REGION Network 12: HMI BA3 SET GOOD PART
   RUNG wire#powerrail
      Contact( "DB2001_MODES_GENERAL".BA.BA3_SELECTED )
      I_Contact( "DB1201_PART_CYCLE_UNIT_01".RUNNING )
      Contact( "DB1018_SAFETY_TAGS".ENABLE_DEVICE_FROM_UNIT_01_MAIN_SAFETY_DOOR_AREA )
      Contact( "DB7224_HMI_AXES".BA3.SOFTKEYS.SET_GOOD_PART )
      wire#w1
      Contact( "DB4000_FIX_TABLE_POSITIONS".UNIT_01.FIXTURE_1.IN_CLADDING_STATION_3 )
      wire#w2
      S_Coil( "DB8000_PART_STATUS".UNIT_01.FIXTURE_1.PART_A.STATUS.OK )
   END_RUNG
   RUNG wire#w2
      R_Coil( "DB8000_PART_STATUS".UNIT_01.FIXTURE_1.PART_A.STATUS.PART_REJECTED )
   END_RUNG
   RUNG wire#w1
      Contact( "DB4000_FIX_TABLE_POSITIONS".UNIT_01.FIXTURE_2.IN_CLADDING_STATION_3 )
      wire#w3
      S_Coil( "DB8000_PART_STATUS".UNIT_01.FIXTURE_2.PART_A.STATUS.OK )
   END_RUNG
   RUNG wire#w3
      R_Coil( "DB8000_PART_STATUS".UNIT_01.FIXTURE_2.PART_A.STATUS.PART_REJECTED )
   END_RUNG
   RUNG wire#w1
      Contact( "DB4000_FIX_TABLE_POSITIONS".UNIT_01.FIXTURE_3.IN_CLADDING_STATION_3 )
      wire#w4
      S_Coil( "DB8000_PART_STATUS".UNIT_01.FIXTURE_3.PART_A.STATUS.OK )
   END_RUNG
   RUNG wire#w4
      R_Coil( "DB8000_PART_STATUS".UNIT_01.FIXTURE_3.PART_A.STATUS.PART_REJECTED )
   END_RUNG
   RUNG wire#w1
      Contact( "DB4000_FIX_TABLE_POSITIONS".UNIT_01.FIXTURE_4.IN_CLADDING_STATION_3 )
      wire#w5
      S_Coil( "DB8000_PART_STATUS".UNIT_01.FIXTURE_4.PART_A.STATUS.OK )
   END_RUNG
   RUNG wire#w5
      R_Coil( "DB8000_PART_STATUS".UNIT_01.FIXTURE_4.PART_A.STATUS.PART_REJECTED )
   END_RUNG
   // the same network as SCL:
   #_w1 := "DB2001_MODES_GENERAL".BA.BA3_SELECTED AND NOT "DB1201_PART_CYCLE_UNIT_01".RUNNING AND "DB1018_SAFETY_TAGS".ENABLE_DEVICE_FROM_UNIT_01_MAIN_SAFETY_DOOR_AREA AND "DB7224_HMI_AXES".BA3.SOFTKEYS.SET_GOOD_PART;
   IF #_w1 AND "DB4000_FIX_TABLE_POSITIONS".UNIT_01.FIXTURE_1.IN_CLADDING_STATION_3 THEN
       "DB8000_PART_STATUS".UNIT_01.FIXTURE_1.PART_A.STATUS.OK := TRUE;
       "DB8000_PART_STATUS".UNIT_01.FIXTURE_1.PART_A.STATUS.PART_REJECTED := FALSE;
   END_IF;
   IF #_w1 AND "DB4000_FIX_TABLE_POSITIONS".UNIT_01.FIXTURE_2.IN_CLADDING_STATION_3 THEN
       "DB8000_PART_STATUS".UNIT_01.FIXTURE_2.PART_A.STATUS.OK := TRUE;
       "DB8000_PART_STATUS".UNIT_01.FIXTURE_2.PART_A.STATUS.PART_REJECTED := FALSE;
   END_IF;
   IF #_w1 AND "DB4000_FIX_TABLE_POSITIONS".UNIT_01.FIXTURE_3.IN_CLADDING_STATION_3 THEN
       "DB8000_PART_STATUS".UNIT_01.FIXTURE_3.PART_A.STATUS.OK := TRUE;
       "DB8000_PART_STATUS".UNIT_01.FIXTURE_3.PART_A.STATUS.PART_REJECTED := FALSE;
   END_IF;
   IF #_w1 AND "DB4000_FIX_TABLE_POSITIONS".UNIT_01.FIXTURE_4.IN_CLADDING_STATION_3 THEN
       "DB8000_PART_STATUS".UNIT_01.FIXTURE_4.PART_A.STATUS.OK := TRUE;
       "DB8000_PART_STATUS".UNIT_01.FIXTURE_4.PART_A.STATUS.PART_REJECTED := FALSE;
   END_IF;
END_REGION

REGION Network 13: UNIT 01 STATION 1 PART A PRESENT
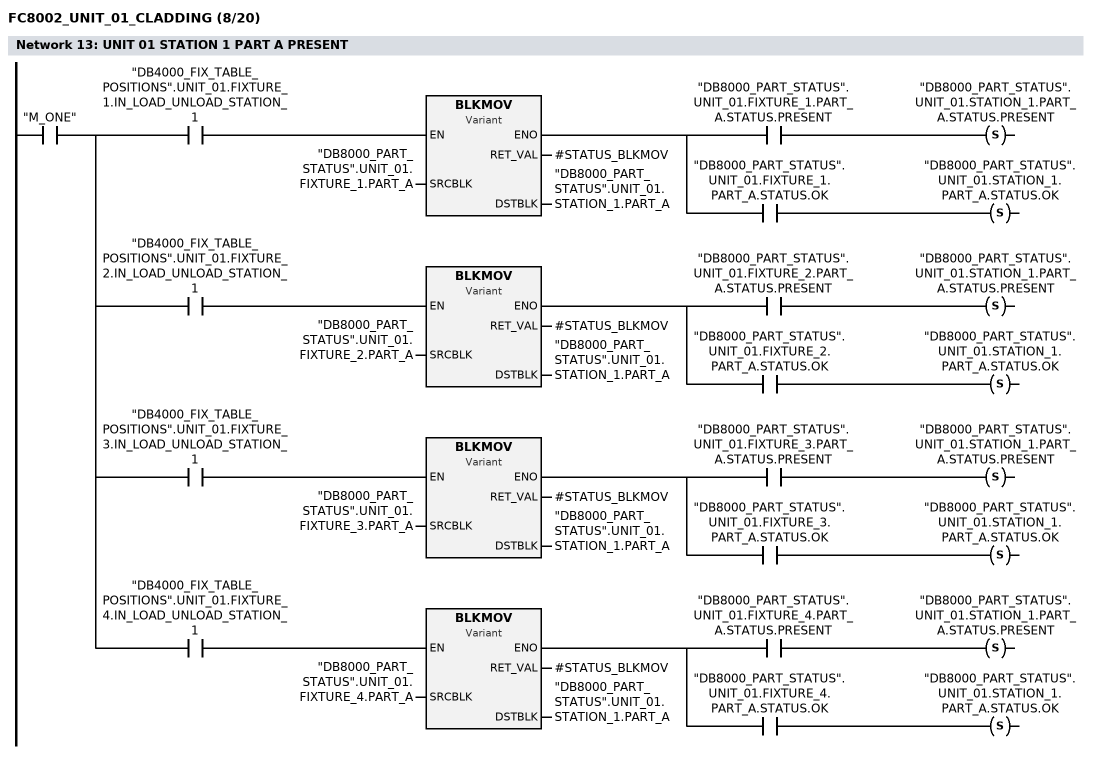
   RUNG wire#powerrail
      Contact( "M_ONE" )
      wire#w1
      Contact( "DB4000_FIX_TABLE_POSITIONS".UNIT_01.FIXTURE_1.IN_LOAD_UNLOAD_STATION_1 )
      { S7_Templates := "blk_type := Variant" } BLKMOV(SRCBLK := "DB8000_PART_STATUS".UNIT_01.FIXTURE_1.PART_A, RET_VAL => #STATUS_BLKMOV, DSTBLK => "DB8000_PART_STATUS".UNIT_01.STATION_1.PART_A)
      wire#w2
      Contact( "DB8000_PART_STATUS".UNIT_01.FIXTURE_1.PART_A.STATUS.PRESENT )
      S_Coil( "DB8000_PART_STATUS".UNIT_01.STATION_1.PART_A.STATUS.PRESENT )
   END_RUNG
   RUNG wire#w2
      Contact( "DB8000_PART_STATUS".UNIT_01.FIXTURE_1.PART_A.STATUS.OK )
      S_Coil( "DB8000_PART_STATUS".UNIT_01.STATION_1.PART_A.STATUS.OK )
   END_RUNG
   RUNG wire#w1
      Contact( "DB4000_FIX_TABLE_POSITIONS".UNIT_01.FIXTURE_2.IN_LOAD_UNLOAD_STATION_1 )
      { S7_Templates := "blk_type := Variant" } BLKMOV(SRCBLK := "DB8000_PART_STATUS".UNIT_01.FIXTURE_2.PART_A, RET_VAL => #STATUS_BLKMOV, DSTBLK => "DB8000_PART_STATUS".UNIT_01.STATION_1.PART_A)
      wire#w3
      Contact( "DB8000_PART_STATUS".UNIT_01.FIXTURE_2.PART_A.STATUS.PRESENT )
      S_Coil( "DB8000_PART_STATUS".UNIT_01.STATION_1.PART_A.STATUS.PRESENT )
   END_RUNG
   RUNG wire#w3
      Contact( "DB8000_PART_STATUS".UNIT_01.FIXTURE_2.PART_A.STATUS.OK )
      S_Coil( "DB8000_PART_STATUS".UNIT_01.STATION_1.PART_A.STATUS.OK )
   END_RUNG
   RUNG wire#w1
      Contact( "DB4000_FIX_TABLE_POSITIONS".UNIT_01.FIXTURE_3.IN_LOAD_UNLOAD_STATION_1 )
      { S7_Templates := "blk_type := Variant" } BLKMOV(SRCBLK := "DB8000_PART_STATUS".UNIT_01.FIXTURE_3.PART_A, RET_VAL => #STATUS_BLKMOV, DSTBLK => "DB8000_PART_STATUS".UNIT_01.STATION_1.PART_A)
      wire#w4
      Contact( "DB8000_PART_STATUS".UNIT_01.FIXTURE_3.PART_A.STATUS.PRESENT )
      S_Coil( "DB8000_PART_STATUS".UNIT_01.STATION_1.PART_A.STATUS.PRESENT )
   END_RUNG
   RUNG wire#w4
      Contact( "DB8000_PART_STATUS".UNIT_01.FIXTURE_3.PART_A.STATUS.OK )
      S_Coil( "DB8000_PART_STATUS".UNIT_01.STATION_1.PART_A.STATUS.OK )
   END_RUNG
   RUNG wire#w1
      Contact( "DB4000_FIX_TABLE_POSITIONS".UNIT_01.FIXTURE_4.IN_LOAD_UNLOAD_STATION_1 )
      { S7_Templates := "blk_type := Variant" } BLKMOV(SRCBLK := "DB8000_PART_STATUS".UNIT_01.FIXTURE_4.PART_A, RET_VAL => #STATUS_BLKMOV, DSTBLK => "DB8000_PART_STATUS".UNIT_01.STATION_1.PART_A)
      wire#w5
      Contact( "DB8000_PART_STATUS".UNIT_01.FIXTURE_4.PART_A.STATUS.PRESENT )
      S_Coil( "DB8000_PART_STATUS".UNIT_01.STATION_1.PART_A.STATUS.PRESENT )
   END_RUNG
   RUNG wire#w5
      Contact( "DB8000_PART_STATUS".UNIT_01.FIXTURE_4.PART_A.STATUS.OK )
      S_Coil( "DB8000_PART_STATUS".UNIT_01.STATION_1.PART_A.STATUS.OK )
   END_RUNG
   // the same network as SCL:
   #_w1 := "M_ONE" AND "DB4000_FIX_TABLE_POSITIONS".UNIT_01.FIXTURE_1.IN_LOAD_UNLOAD_STATION_1;
   #_w3 := "M_ONE";
   #STATUS_BLKMOV := BLKMOV(EN := #_w1,
                           SRCBLK := "DB8000_PART_STATUS".UNIT_01.FIXTURE_1.PART_A,
                           DSTBLK => "DB8000_PART_STATUS".UNIT_01.STATION_1.PART_A,
                           ENO => #_w2);
   IF #_w2 AND "DB8000_PART_STATUS".UNIT_01.FIXTURE_1.PART_A.STATUS.PRESENT THEN
       "DB8000_PART_STATUS".UNIT_01.STATION_1.PART_A.STATUS.PRESENT := TRUE;
   END_IF;
   IF #_w2 AND "DB8000_PART_STATUS".UNIT_01.FIXTURE_1.PART_A.STATUS.OK THEN
       "DB8000_PART_STATUS".UNIT_01.STATION_1.PART_A.STATUS.OK := TRUE;
   END_IF;
   #_w4 := #_w3 AND "DB4000_FIX_TABLE_POSITIONS".UNIT_01.FIXTURE_2.IN_LOAD_UNLOAD_STATION_1;
   #STATUS_BLKMOV := BLKMOV(EN := #_w4,
                           SRCBLK := "DB8000_PART_STATUS".UNIT_01.FIXTURE_2.PART_A,
                           DSTBLK => "DB8000_PART_STATUS".UNIT_01.STATION_1.PART_A,
                           ENO => #_w5);
   IF #_w5 AND "DB8000_PART_STATUS".UNIT_01.FIXTURE_2.PART_A.STATUS.PRESENT THEN
       "DB8000_PART_STATUS".UNIT_01.STATION_1.PART_A.STATUS.PRESENT := TRUE;
   END_IF;
   IF #_w5 AND "DB8000_PART_STATUS".UNIT_01.FIXTURE_2.PART_A.STATUS.OK THEN
       "DB8000_PART_STATUS".UNIT_01.STATION_1.PART_A.STATUS.OK := TRUE;
   END_IF;
   #_w6 := #_w3 AND "DB4000_FIX_TABLE_POSITIONS".UNIT_01.FIXTURE_3.IN_LOAD_UNLOAD_STATION_1;
   #STATUS_BLKMOV := BLKMOV(EN := #_w6,
                           SRCBLK := "DB8000_PART_STATUS".UNIT_01.FIXTURE_3.PART_A,
                           DSTBLK => "DB8000_PART_STATUS".UNIT_01.STATION_1.PART_A,
                           ENO => #_w7);
   IF #_w7 AND "DB8000_PART_STATUS".UNIT_01.FIXTURE_3.PART_A.STATUS.PRESENT THEN
       "DB8000_PART_STATUS".UNIT_01.STATION_1.PART_A.STATUS.PRESENT := TRUE;
   END_IF;
   IF #_w7 AND "DB8000_PART_STATUS".UNIT_01.FIXTURE_3.PART_A.STATUS.OK THEN
       "DB8000_PART_STATUS".UNIT_01.STATION_1.PART_A.STATUS.OK := TRUE;
   END_IF;
   #_w8 := #_w3 AND "DB4000_FIX_TABLE_POSITIONS".UNIT_01.FIXTURE_4.IN_LOAD_UNLOAD_STATION_1;
   #STATUS_BLKMOV := BLKMOV(EN := #_w8,
                           SRCBLK := "DB8000_PART_STATUS".UNIT_01.FIXTURE_4.PART_A,
                           DSTBLK => "DB8000_PART_STATUS".UNIT_01.STATION_1.PART_A,
                           ENO => #_w9);
   IF #_w9 AND "DB8000_PART_STATUS".UNIT_01.FIXTURE_4.PART_A.STATUS.PRESENT THEN
       "DB8000_PART_STATUS".UNIT_01.STATION_1.PART_A.STATUS.PRESENT := TRUE;
   END_IF;
   IF #_w9 AND "DB8000_PART_STATUS".UNIT_01.FIXTURE_4.PART_A.STATUS.OK THEN
       "DB8000_PART_STATUS".UNIT_01.STATION_1.PART_A.STATUS.OK := TRUE;
   END_IF;
END_REGION

REGION Network 14: UNIT 01 STATION 2 PART A PRESENT
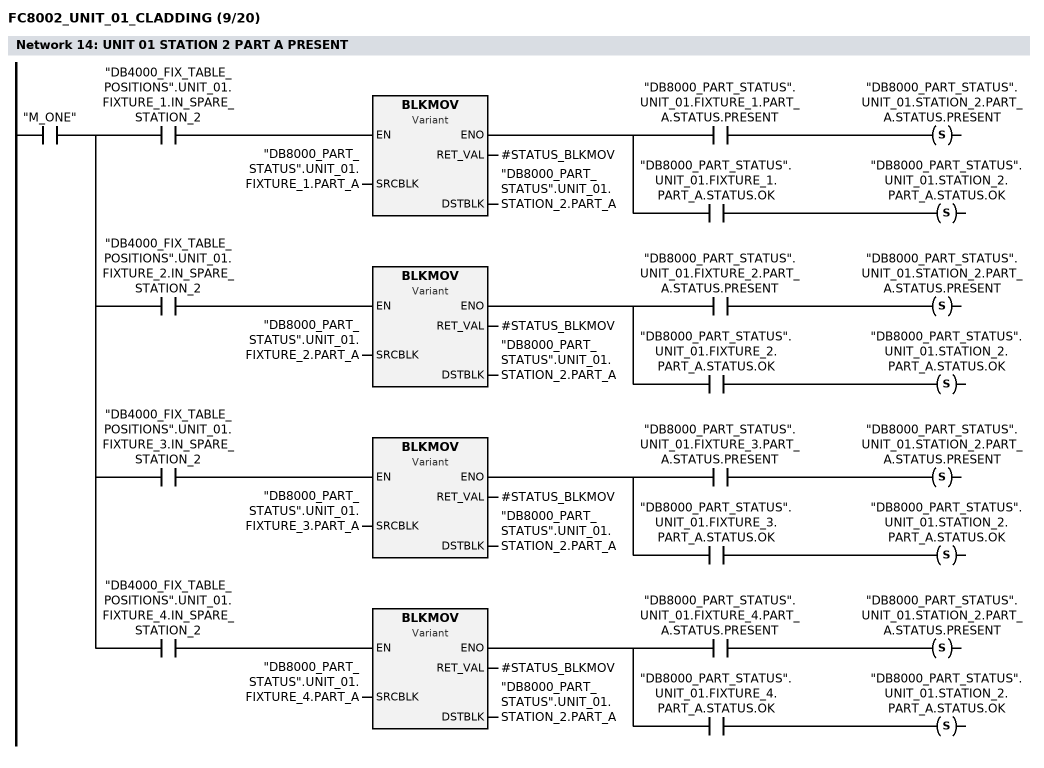
   RUNG wire#powerrail
      Contact( "M_ONE" )
      wire#w1
      Contact( "DB4000_FIX_TABLE_POSITIONS".UNIT_01.FIXTURE_1.IN_SPARE_STATION_2 )
      { S7_Templates := "blk_type := Variant" } BLKMOV(SRCBLK := "DB8000_PART_STATUS".UNIT_01.FIXTURE_1.PART_A, RET_VAL => #STATUS_BLKMOV, DSTBLK => "DB8000_PART_STATUS".UNIT_01.STATION_2.PART_A)
      wire#w2
      Contact( "DB8000_PART_STATUS".UNIT_01.FIXTURE_1.PART_A.STATUS.PRESENT )
      S_Coil( "DB8000_PART_STATUS".UNIT_01.STATION_2.PART_A.STATUS.PRESENT )
   END_RUNG
   RUNG wire#w2
      Contact( "DB8000_PART_STATUS".UNIT_01.FIXTURE_1.PART_A.STATUS.OK )
      S_Coil( "DB8000_PART_STATUS".UNIT_01.STATION_2.PART_A.STATUS.OK )
   END_RUNG
   RUNG wire#w1
      Contact( "DB4000_FIX_TABLE_POSITIONS".UNIT_01.FIXTURE_2.IN_SPARE_STATION_2 )
      { S7_Templates := "blk_type := Variant" } BLKMOV(SRCBLK := "DB8000_PART_STATUS".UNIT_01.FIXTURE_2.PART_A, RET_VAL => #STATUS_BLKMOV, DSTBLK => "DB8000_PART_STATUS".UNIT_01.STATION_2.PART_A)
      wire#w3
      Contact( "DB8000_PART_STATUS".UNIT_01.FIXTURE_2.PART_A.STATUS.PRESENT )
      S_Coil( "DB8000_PART_STATUS".UNIT_01.STATION_2.PART_A.STATUS.PRESENT )
   END_RUNG
   RUNG wire#w3
      Contact( "DB8000_PART_STATUS".UNIT_01.FIXTURE_2.PART_A.STATUS.OK )
      S_Coil( "DB8000_PART_STATUS".UNIT_01.STATION_2.PART_A.STATUS.OK )
   END_RUNG
   RUNG wire#w1
      Contact( "DB4000_FIX_TABLE_POSITIONS".UNIT_01.FIXTURE_3.IN_SPARE_STATION_2 )
      { S7_Templates := "blk_type := Variant" } BLKMOV(SRCBLK := "DB8000_PART_STATUS".UNIT_01.FIXTURE_3.PART_A, RET_VAL => #STATUS_BLKMOV, DSTBLK => "DB8000_PART_STATUS".UNIT_01.STATION_2.PART_A)
      wire#w4
      Contact( "DB8000_PART_STATUS".UNIT_01.FIXTURE_3.PART_A.STATUS.PRESENT )
      S_Coil( "DB8000_PART_STATUS".UNIT_01.STATION_2.PART_A.STATUS.PRESENT )
   END_RUNG
   RUNG wire#w4
      Contact( "DB8000_PART_STATUS".UNIT_01.FIXTURE_3.PART_A.STATUS.OK )
      S_Coil( "DB8000_PART_STATUS".UNIT_01.STATION_2.PART_A.STATUS.OK )
   END_RUNG
   RUNG wire#w1
      Contact( "DB4000_FIX_TABLE_POSITIONS".UNIT_01.FIXTURE_4.IN_SPARE_STATION_2 )
      { S7_Templates := "blk_type := Variant" } BLKMOV(SRCBLK := "DB8000_PART_STATUS".UNIT_01.FIXTURE_4.PART_A, RET_VAL => #STATUS_BLKMOV, DSTBLK => "DB8000_PART_STATUS".UNIT_01.STATION_2.PART_A)
      wire#w5
      Contact( "DB8000_PART_STATUS".UNIT_01.FIXTURE_4.PART_A.STATUS.PRESENT )
      S_Coil( "DB8000_PART_STATUS".UNIT_01.STATION_2.PART_A.STATUS.PRESENT )
   END_RUNG
   RUNG wire#w5
      Contact( "DB8000_PART_STATUS".UNIT_01.FIXTURE_4.PART_A.STATUS.OK )
      S_Coil( "DB8000_PART_STATUS".UNIT_01.STATION_2.PART_A.STATUS.OK )
   END_RUNG
   // the same network as SCL:
   #_w1 := "M_ONE" AND "DB4000_FIX_TABLE_POSITIONS".UNIT_01.FIXTURE_1.IN_SPARE_STATION_2;
   #_w3 := "M_ONE";
   #STATUS_BLKMOV := BLKMOV(EN := #_w1,
                           SRCBLK := "DB8000_PART_STATUS".UNIT_01.FIXTURE_1.PART_A,
                           DSTBLK => "DB8000_PART_STATUS".UNIT_01.STATION_2.PART_A,
                           ENO => #_w2);
   IF #_w2 AND "DB8000_PART_STATUS".UNIT_01.FIXTURE_1.PART_A.STATUS.PRESENT THEN
       "DB8000_PART_STATUS".UNIT_01.STATION_2.PART_A.STATUS.PRESENT := TRUE;
   END_IF;
   IF #_w2 AND "DB8000_PART_STATUS".UNIT_01.FIXTURE_1.PART_A.STATUS.OK THEN
       "DB8000_PART_STATUS".UNIT_01.STATION_2.PART_A.STATUS.OK := TRUE;
   END_IF;
   #_w4 := #_w3 AND "DB4000_FIX_TABLE_POSITIONS".UNIT_01.FIXTURE_2.IN_SPARE_STATION_2;
   #STATUS_BLKMOV := BLKMOV(EN := #_w4,
                           SRCBLK := "DB8000_PART_STATUS".UNIT_01.FIXTURE_2.PART_A,
                           DSTBLK => "DB8000_PART_STATUS".UNIT_01.STATION_2.PART_A,
                           ENO => #_w5);
   IF #_w5 AND "DB8000_PART_STATUS".UNIT_01.FIXTURE_2.PART_A.STATUS.PRESENT THEN
       "DB8000_PART_STATUS".UNIT_01.STATION_2.PART_A.STATUS.PRESENT := TRUE;
   END_IF;
   IF #_w5 AND "DB8000_PART_STATUS".UNIT_01.FIXTURE_2.PART_A.STATUS.OK THEN
       "DB8000_PART_STATUS".UNIT_01.STATION_2.PART_A.STATUS.OK := TRUE;
   END_IF;
   #_w6 := #_w3 AND "DB4000_FIX_TABLE_POSITIONS".UNIT_01.FIXTURE_3.IN_SPARE_STATION_2;
   #STATUS_BLKMOV := BLKMOV(EN := #_w6,
                           SRCBLK := "DB8000_PART_STATUS".UNIT_01.FIXTURE_3.PART_A,
                           DSTBLK => "DB8000_PART_STATUS".UNIT_01.STATION_2.PART_A,
                           ENO => #_w7);
   IF #_w7 AND "DB8000_PART_STATUS".UNIT_01.FIXTURE_3.PART_A.STATUS.PRESENT THEN
       "DB8000_PART_STATUS".UNIT_01.STATION_2.PART_A.STATUS.PRESENT := TRUE;
   END_IF;
   IF #_w7 AND "DB8000_PART_STATUS".UNIT_01.FIXTURE_3.PART_A.STATUS.OK THEN
       "DB8000_PART_STATUS".UNIT_01.STATION_2.PART_A.STATUS.OK := TRUE;
   END_IF;
   #_w8 := #_w3 AND "DB4000_FIX_TABLE_POSITIONS".UNIT_01.FIXTURE_4.IN_SPARE_STATION_2;
   #STATUS_BLKMOV := BLKMOV(EN := #_w8,
                           SRCBLK := "DB8000_PART_STATUS".UNIT_01.FIXTURE_4.PART_A,
                           DSTBLK => "DB8000_PART_STATUS".UNIT_01.STATION_2.PART_A,
                           ENO => #_w9);
   IF #_w9 AND "DB8000_PART_STATUS".UNIT_01.FIXTURE_4.PART_A.STATUS.PRESENT THEN
       "DB8000_PART_STATUS".UNIT_01.STATION_2.PART_A.STATUS.PRESENT := TRUE;
   END_IF;
   IF #_w9 AND "DB8000_PART_STATUS".UNIT_01.FIXTURE_4.PART_A.STATUS.OK THEN
       "DB8000_PART_STATUS".UNIT_01.STATION_2.PART_A.STATUS.OK := TRUE;
   END_IF;
END_REGION

REGION Network 15: UNIT 01 STATION 3 PART A PRESENT
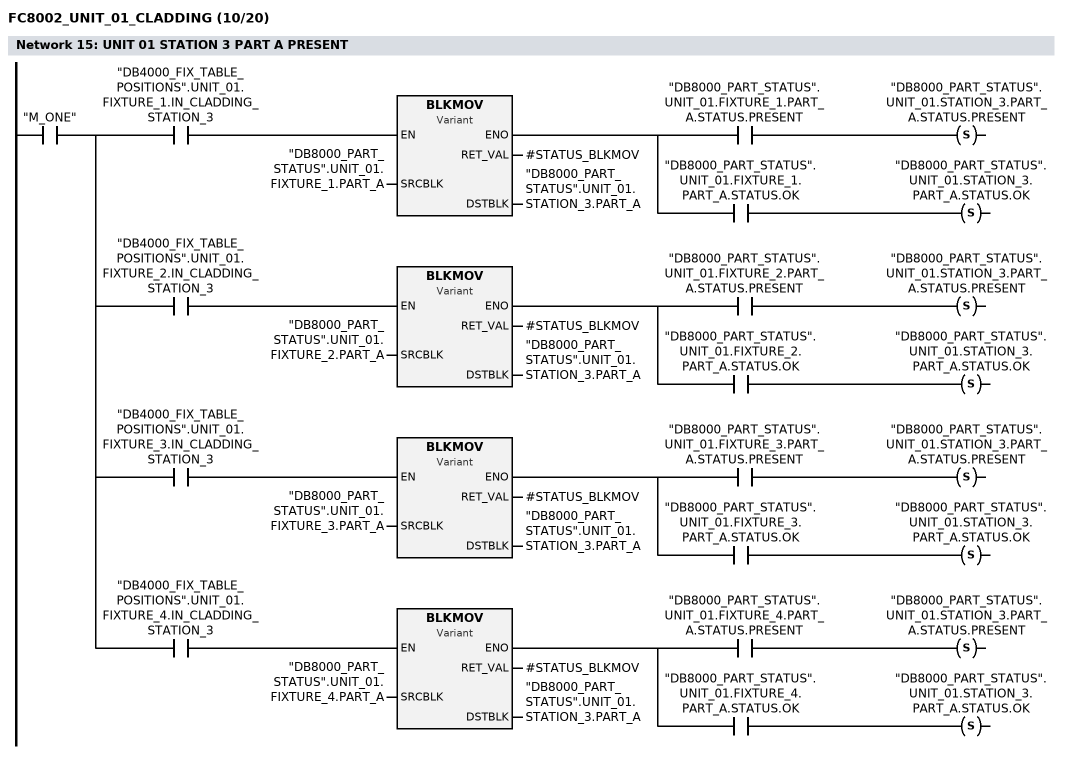
   RUNG wire#powerrail
      Contact( "M_ONE" )
      wire#w1
      Contact( "DB4000_FIX_TABLE_POSITIONS".UNIT_01.FIXTURE_1.IN_CLADDING_STATION_3 )
      { S7_Templates := "blk_type := Variant" } BLKMOV(SRCBLK := "DB8000_PART_STATUS".UNIT_01.FIXTURE_1.PART_A, RET_VAL => #STATUS_BLKMOV, DSTBLK => "DB8000_PART_STATUS".UNIT_01.STATION_3.PART_A)
      wire#w2
      Contact( "DB8000_PART_STATUS".UNIT_01.FIXTURE_1.PART_A.STATUS.PRESENT )
      S_Coil( "DB8000_PART_STATUS".UNIT_01.STATION_3.PART_A.STATUS.PRESENT )
   END_RUNG
   RUNG wire#w2
      Contact( "DB8000_PART_STATUS".UNIT_01.FIXTURE_1.PART_A.STATUS.OK )
      S_Coil( "DB8000_PART_STATUS".UNIT_01.STATION_3.PART_A.STATUS.OK )
   END_RUNG
   RUNG wire#w1
      Contact( "DB4000_FIX_TABLE_POSITIONS".UNIT_01.FIXTURE_2.IN_CLADDING_STATION_3 )
      { S7_Templates := "blk_type := Variant" } BLKMOV(SRCBLK := "DB8000_PART_STATUS".UNIT_01.FIXTURE_2.PART_A, RET_VAL => #STATUS_BLKMOV, DSTBLK => "DB8000_PART_STATUS".UNIT_01.STATION_3.PART_A)
      wire#w3
      Contact( "DB8000_PART_STATUS".UNIT_01.FIXTURE_2.PART_A.STATUS.PRESENT )
      S_Coil( "DB8000_PART_STATUS".UNIT_01.STATION_3.PART_A.STATUS.PRESENT )
   END_RUNG
   RUNG wire#w3
      Contact( "DB8000_PART_STATUS".UNIT_01.FIXTURE_2.PART_A.STATUS.OK )
      S_Coil( "DB8000_PART_STATUS".UNIT_01.STATION_3.PART_A.STATUS.OK )
   END_RUNG
   RUNG wire#w1
      Contact( "DB4000_FIX_TABLE_POSITIONS".UNIT_01.FIXTURE_3.IN_CLADDING_STATION_3 )
      { S7_Templates := "blk_type := Variant" } BLKMOV(SRCBLK := "DB8000_PART_STATUS".UNIT_01.FIXTURE_3.PART_A, RET_VAL => #STATUS_BLKMOV, DSTBLK => "DB8000_PART_STATUS".UNIT_01.STATION_3.PART_A)
      wire#w4
      Contact( "DB8000_PART_STATUS".UNIT_01.FIXTURE_3.PART_A.STATUS.PRESENT )
      S_Coil( "DB8000_PART_STATUS".UNIT_01.STATION_3.PART_A.STATUS.PRESENT )
   END_RUNG
   RUNG wire#w4
      Contact( "DB8000_PART_STATUS".UNIT_01.FIXTURE_3.PART_A.STATUS.OK )
      S_Coil( "DB8000_PART_STATUS".UNIT_01.STATION_3.PART_A.STATUS.OK )
   END_RUNG
   RUNG wire#w1
      Contact( "DB4000_FIX_TABLE_POSITIONS".UNIT_01.FIXTURE_4.IN_CLADDING_STATION_3 )
      { S7_Templates := "blk_type := Variant" } BLKMOV(SRCBLK := "DB8000_PART_STATUS".UNIT_01.FIXTURE_4.PART_A, RET_VAL => #STATUS_BLKMOV, DSTBLK => "DB8000_PART_STATUS".UNIT_01.STATION_3.PART_A)
      wire#w5
      Contact( "DB8000_PART_STATUS".UNIT_01.FIXTURE_4.PART_A.STATUS.PRESENT )
      S_Coil( "DB8000_PART_STATUS".UNIT_01.STATION_3.PART_A.STATUS.PRESENT )
   END_RUNG
   RUNG wire#w5
      Contact( "DB8000_PART_STATUS".UNIT_01.FIXTURE_4.PART_A.STATUS.OK )
      S_Coil( "DB8000_PART_STATUS".UNIT_01.STATION_3.PART_A.STATUS.OK )
   END_RUNG
   // the same network as SCL:
   #_w1 := "M_ONE" AND "DB4000_FIX_TABLE_POSITIONS".UNIT_01.FIXTURE_1.IN_CLADDING_STATION_3;
   #_w3 := "M_ONE";
   #STATUS_BLKMOV := BLKMOV(EN := #_w1,
                           SRCBLK := "DB8000_PART_STATUS".UNIT_01.FIXTURE_1.PART_A,
                           DSTBLK => "DB8000_PART_STATUS".UNIT_01.STATION_3.PART_A,
                           ENO => #_w2);
   IF #_w2 AND "DB8000_PART_STATUS".UNIT_01.FIXTURE_1.PART_A.STATUS.PRESENT THEN
       "DB8000_PART_STATUS".UNIT_01.STATION_3.PART_A.STATUS.PRESENT := TRUE;
   END_IF;
   IF #_w2 AND "DB8000_PART_STATUS".UNIT_01.FIXTURE_1.PART_A.STATUS.OK THEN
       "DB8000_PART_STATUS".UNIT_01.STATION_3.PART_A.STATUS.OK := TRUE;
   END_IF;
   #_w4 := #_w3 AND "DB4000_FIX_TABLE_POSITIONS".UNIT_01.FIXTURE_2.IN_CLADDING_STATION_3;
   #STATUS_BLKMOV := BLKMOV(EN := #_w4,
                           SRCBLK := "DB8000_PART_STATUS".UNIT_01.FIXTURE_2.PART_A,
                           DSTBLK => "DB8000_PART_STATUS".UNIT_01.STATION_3.PART_A,
                           ENO => #_w5);
   IF #_w5 AND "DB8000_PART_STATUS".UNIT_01.FIXTURE_2.PART_A.STATUS.PRESENT THEN
       "DB8000_PART_STATUS".UNIT_01.STATION_3.PART_A.STATUS.PRESENT := TRUE;
   END_IF;
   IF #_w5 AND "DB8000_PART_STATUS".UNIT_01.FIXTURE_2.PART_A.STATUS.OK THEN
       "DB8000_PART_STATUS".UNIT_01.STATION_3.PART_A.STATUS.OK := TRUE;
   END_IF;
   #_w6 := #_w3 AND "DB4000_FIX_TABLE_POSITIONS".UNIT_01.FIXTURE_3.IN_CLADDING_STATION_3;
   #STATUS_BLKMOV := BLKMOV(EN := #_w6,
                           SRCBLK := "DB8000_PART_STATUS".UNIT_01.FIXTURE_3.PART_A,
                           DSTBLK => "DB8000_PART_STATUS".UNIT_01.STATION_3.PART_A,
                           ENO => #_w7);
   IF #_w7 AND "DB8000_PART_STATUS".UNIT_01.FIXTURE_3.PART_A.STATUS.PRESENT THEN
       "DB8000_PART_STATUS".UNIT_01.STATION_3.PART_A.STATUS.PRESENT := TRUE;
   END_IF;
   IF #_w7 AND "DB8000_PART_STATUS".UNIT_01.FIXTURE_3.PART_A.STATUS.OK THEN
       "DB8000_PART_STATUS".UNIT_01.STATION_3.PART_A.STATUS.OK := TRUE;
   END_IF;
   #_w8 := #_w3 AND "DB4000_FIX_TABLE_POSITIONS".UNIT_01.FIXTURE_4.IN_CLADDING_STATION_3;
   #STATUS_BLKMOV := BLKMOV(EN := #_w8,
                           SRCBLK := "DB8000_PART_STATUS".UNIT_01.FIXTURE_4.PART_A,
                           DSTBLK => "DB8000_PART_STATUS".UNIT_01.STATION_3.PART_A,
                           ENO => #_w9);
   IF #_w9 AND "DB8000_PART_STATUS".UNIT_01.FIXTURE_4.PART_A.STATUS.PRESENT THEN
       "DB8000_PART_STATUS".UNIT_01.STATION_3.PART_A.STATUS.PRESENT := TRUE;
   END_IF;
   IF #_w9 AND "DB8000_PART_STATUS".UNIT_01.FIXTURE_4.PART_A.STATUS.OK THEN
       "DB8000_PART_STATUS".UNIT_01.STATION_3.PART_A.STATUS.OK := TRUE;
   END_IF;
END_REGION

REGION Network 16: UNIT 01 STATION 4 PART A PRESENT
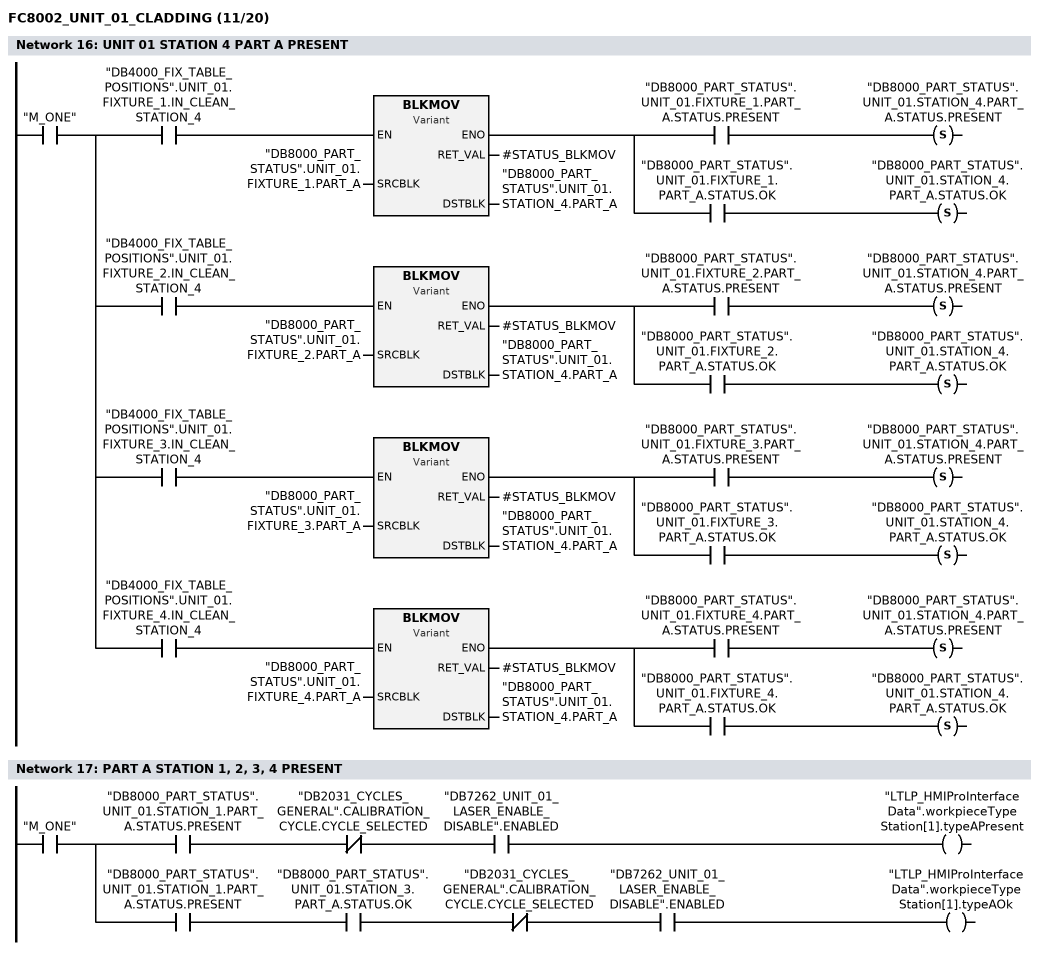
   RUNG wire#powerrail
      Contact( "M_ONE" )
      wire#w1
      Contact( "DB4000_FIX_TABLE_POSITIONS".UNIT_01.FIXTURE_1.IN_CLEAN_STATION_4 )
      { S7_Templates := "blk_type := Variant" } BLKMOV(SRCBLK := "DB8000_PART_STATUS".UNIT_01.FIXTURE_1.PART_A, RET_VAL => #STATUS_BLKMOV, DSTBLK => "DB8000_PART_STATUS".UNIT_01.STATION_4.PART_A)
      wire#w2
      Contact( "DB8000_PART_STATUS".UNIT_01.FIXTURE_1.PART_A.STATUS.PRESENT )
      S_Coil( "DB8000_PART_STATUS".UNIT_01.STATION_4.PART_A.STATUS.PRESENT )
   END_RUNG
   RUNG wire#w2
      Contact( "DB8000_PART_STATUS".UNIT_01.FIXTURE_1.PART_A.STATUS.OK )
      S_Coil( "DB8000_PART_STATUS".UNIT_01.STATION_4.PART_A.STATUS.OK )
   END_RUNG
   RUNG wire#w1
      Contact( "DB4000_FIX_TABLE_POSITIONS".UNIT_01.FIXTURE_2.IN_CLEAN_STATION_4 )
      { S7_Templates := "blk_type := Variant" } BLKMOV(SRCBLK := "DB8000_PART_STATUS".UNIT_01.FIXTURE_2.PART_A, RET_VAL => #STATUS_BLKMOV, DSTBLK => "DB8000_PART_STATUS".UNIT_01.STATION_4.PART_A)
      wire#w3
      Contact( "DB8000_PART_STATUS".UNIT_01.FIXTURE_2.PART_A.STATUS.PRESENT )
      S_Coil( "DB8000_PART_STATUS".UNIT_01.STATION_4.PART_A.STATUS.PRESENT )
   END_RUNG
   RUNG wire#w3
      Contact( "DB8000_PART_STATUS".UNIT_01.FIXTURE_2.PART_A.STATUS.OK )
      S_Coil( "DB8000_PART_STATUS".UNIT_01.STATION_4.PART_A.STATUS.OK )
   END_RUNG
   RUNG wire#w1
      Contact( "DB4000_FIX_TABLE_POSITIONS".UNIT_01.FIXTURE_3.IN_CLEAN_STATION_4 )
      { S7_Templates := "blk_type := Variant" } BLKMOV(SRCBLK := "DB8000_PART_STATUS".UNIT_01.FIXTURE_3.PART_A, RET_VAL => #STATUS_BLKMOV, DSTBLK => "DB8000_PART_STATUS".UNIT_01.STATION_4.PART_A)
      wire#w4
      Contact( "DB8000_PART_STATUS".UNIT_01.FIXTURE_3.PART_A.STATUS.PRESENT )
      S_Coil( "DB8000_PART_STATUS".UNIT_01.STATION_4.PART_A.STATUS.PRESENT )
   END_RUNG
   RUNG wire#w4
      Contact( "DB8000_PART_STATUS".UNIT_01.FIXTURE_3.PART_A.STATUS.OK )
      S_Coil( "DB8000_PART_STATUS".UNIT_01.STATION_4.PART_A.STATUS.OK )
   END_RUNG
   RUNG wire#w1
      Contact( "DB4000_FIX_TABLE_POSITIONS".UNIT_01.FIXTURE_4.IN_CLEAN_STATION_4 )
      { S7_Templates := "blk_type := Variant" } BLKMOV(SRCBLK := "DB8000_PART_STATUS".UNIT_01.FIXTURE_4.PART_A, RET_VAL => #STATUS_BLKMOV, DSTBLK => "DB8000_PART_STATUS".UNIT_01.STATION_4.PART_A)
      wire#w5
      Contact( "DB8000_PART_STATUS".UNIT_01.FIXTURE_4.PART_A.STATUS.PRESENT )
      S_Coil( "DB8000_PART_STATUS".UNIT_01.STATION_4.PART_A.STATUS.PRESENT )
   END_RUNG
   RUNG wire#w5
      Contact( "DB8000_PART_STATUS".UNIT_01.FIXTURE_4.PART_A.STATUS.OK )
      S_Coil( "DB8000_PART_STATUS".UNIT_01.STATION_4.PART_A.STATUS.OK )
   END_RUNG
   // the same network as SCL:
   #_w1 := "M_ONE" AND "DB4000_FIX_TABLE_POSITIONS".UNIT_01.FIXTURE_1.IN_CLEAN_STATION_4;
   #_w3 := "M_ONE";
   #STATUS_BLKMOV := BLKMOV(EN := #_w1,
                           SRCBLK := "DB8000_PART_STATUS".UNIT_01.FIXTURE_1.PART_A,
                           DSTBLK => "DB8000_PART_STATUS".UNIT_01.STATION_4.PART_A,
                           ENO => #_w2);
   IF #_w2 AND "DB8000_PART_STATUS".UNIT_01.FIXTURE_1.PART_A.STATUS.PRESENT THEN
       "DB8000_PART_STATUS".UNIT_01.STATION_4.PART_A.STATUS.PRESENT := TRUE;
   END_IF;
   IF #_w2 AND "DB8000_PART_STATUS".UNIT_01.FIXTURE_1.PART_A.STATUS.OK THEN
       "DB8000_PART_STATUS".UNIT_01.STATION_4.PART_A.STATUS.OK := TRUE;
   END_IF;
   #_w4 := #_w3 AND "DB4000_FIX_TABLE_POSITIONS".UNIT_01.FIXTURE_2.IN_CLEAN_STATION_4;
   #STATUS_BLKMOV := BLKMOV(EN := #_w4,
                           SRCBLK := "DB8000_PART_STATUS".UNIT_01.FIXTURE_2.PART_A,
                           DSTBLK => "DB8000_PART_STATUS".UNIT_01.STATION_4.PART_A,
                           ENO => #_w5);
   IF #_w5 AND "DB8000_PART_STATUS".UNIT_01.FIXTURE_2.PART_A.STATUS.PRESENT THEN
       "DB8000_PART_STATUS".UNIT_01.STATION_4.PART_A.STATUS.PRESENT := TRUE;
   END_IF;
   IF #_w5 AND "DB8000_PART_STATUS".UNIT_01.FIXTURE_2.PART_A.STATUS.OK THEN
       "DB8000_PART_STATUS".UNIT_01.STATION_4.PART_A.STATUS.OK := TRUE;
   END_IF;
   #_w6 := #_w3 AND "DB4000_FIX_TABLE_POSITIONS".UNIT_01.FIXTURE_3.IN_CLEAN_STATION_4;
   #STATUS_BLKMOV := BLKMOV(EN := #_w6,
                           SRCBLK := "DB8000_PART_STATUS".UNIT_01.FIXTURE_3.PART_A,
                           DSTBLK => "DB8000_PART_STATUS".UNIT_01.STATION_4.PART_A,
                           ENO => #_w7);
   IF #_w7 AND "DB8000_PART_STATUS".UNIT_01.FIXTURE_3.PART_A.STATUS.PRESENT THEN
       "DB8000_PART_STATUS".UNIT_01.STATION_4.PART_A.STATUS.PRESENT := TRUE;
   END_IF;
   IF #_w7 AND "DB8000_PART_STATUS".UNIT_01.FIXTURE_3.PART_A.STATUS.OK THEN
       "DB8000_PART_STATUS".UNIT_01.STATION_4.PART_A.STATUS.OK := TRUE;
   END_IF;
   #_w8 := #_w3 AND "DB4000_FIX_TABLE_POSITIONS".UNIT_01.FIXTURE_4.IN_CLEAN_STATION_4;
   #STATUS_BLKMOV := BLKMOV(EN := #_w8,
                           SRCBLK := "DB8000_PART_STATUS".UNIT_01.FIXTURE_4.PART_A,
                           DSTBLK => "DB8000_PART_STATUS".UNIT_01.STATION_4.PART_A,
                           ENO => #_w9);
   IF #_w9 AND "DB8000_PART_STATUS".UNIT_01.FIXTURE_4.PART_A.STATUS.PRESENT THEN
       "DB8000_PART_STATUS".UNIT_01.STATION_4.PART_A.STATUS.PRESENT := TRUE;
   END_IF;
   IF #_w9 AND "DB8000_PART_STATUS".UNIT_01.FIXTURE_4.PART_A.STATUS.OK THEN
       "DB8000_PART_STATUS".UNIT_01.STATION_4.PART_A.STATUS.OK := TRUE;
   END_IF;
END_REGION

REGION Network 17: PART A STATION 1, 2, 3, 4 PRESENT
   RUNG wire#powerrail
      Contact( "M_ONE" )
      wire#w1
      Contact( "DB8000_PART_STATUS".UNIT_01.STATION_1.PART_A.STATUS.PRESENT )
      I_Contact( "DB2031_CYCLES_GENERAL".CALIBRATION_CYCLE.CYCLE_SELECTED )
      Contact( "DB7262_UNIT_01_LASER_ENABLE_DISABLE".ENABLED )
      Coil( "LTLP_HMIProInterfaceData".workpieceTypeStation[1].typeAPresent )
   END_RUNG
   RUNG wire#w1
      Contact( "DB8000_PART_STATUS".UNIT_01.STATION_1.PART_A.STATUS.PRESENT )
      Contact( "DB8000_PART_STATUS".UNIT_01.STATION_3.PART_A.STATUS.OK )
      I_Contact( "DB2031_CYCLES_GENERAL".CALIBRATION_CYCLE.CYCLE_SELECTED )
      Contact( "DB7262_UNIT_01_LASER_ENABLE_DISABLE".ENABLED )
      Coil( "LTLP_HMIProInterfaceData".workpieceTypeStation[1].typeAOk )
   END_RUNG
   // the same network as SCL:
   "LTLP_HMIProInterfaceData".workpieceTypeStation[1].typeAPresent := "M_ONE" AND "DB8000_PART_STATUS".UNIT_01.STATION_1.PART_A.STATUS.PRESENT AND NOT "DB2031_CYCLES_GENERAL".CALIBRATION_CYCLE.CYCLE_SELECTED AND "DB7262_UNIT_01_LASER_ENABLE_DISABLE".ENABLED;
   "LTLP_HMIProInterfaceData".workpieceTypeStation[1].typeAOk := "M_ONE" AND "DB8000_PART_STATUS".UNIT_01.STATION_1.PART_A.STATUS.PRESENT AND "DB8000_PART_STATUS".UNIT_01.STATION_3.PART_A.STATUS.OK AND NOT "DB2031_CYCLES_GENERAL".CALIBRATION_CYCLE.CYCLE_SELECTED AND "DB7262_UNIT_01_LASER_ENABLE_DISABLE".ENABLED;
END_REGION

REGION Network 18: PART A FIXTURE 1, 2, 3, 4 RESET STATUS TO ZERO
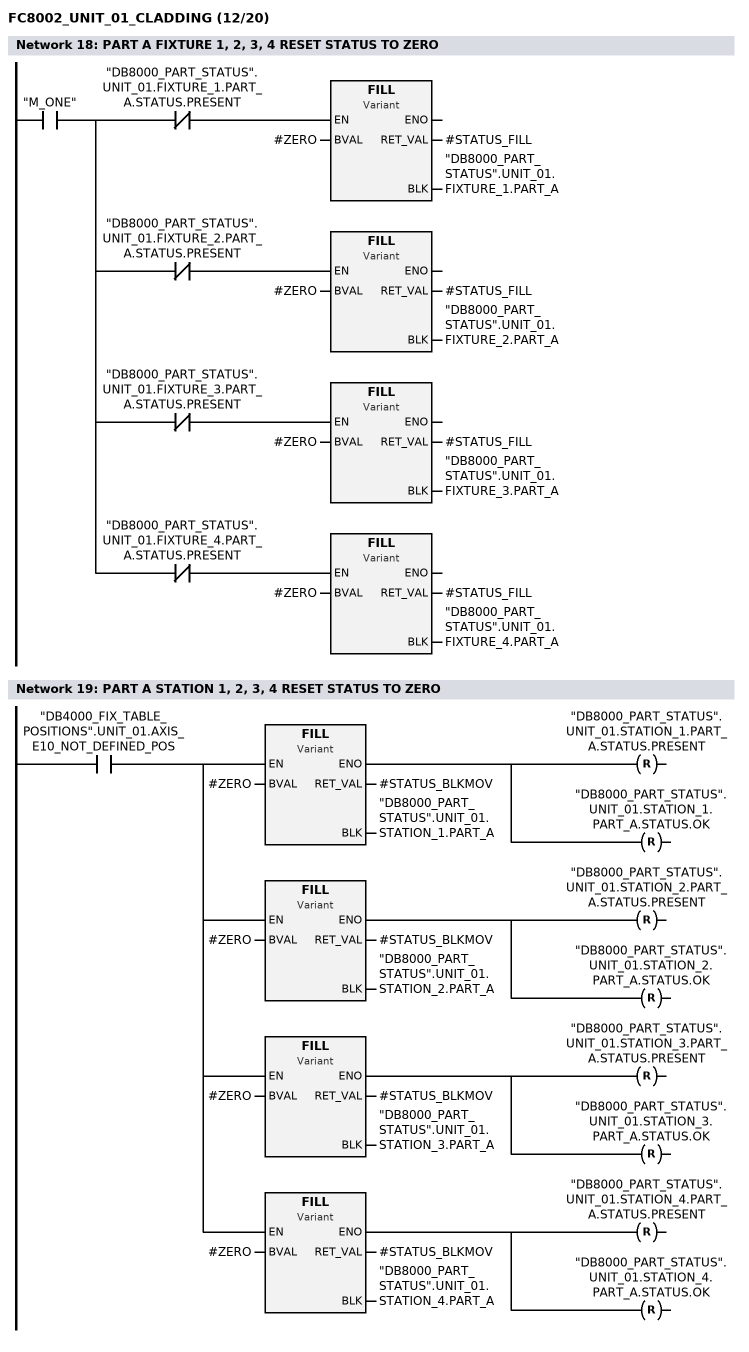
   RUNG wire#powerrail
      Contact( "M_ONE" )
      wire#w1
      I_Contact( "DB8000_PART_STATUS".UNIT_01.FIXTURE_1.PART_A.STATUS.PRESENT )
      { S7_Templates := "ptr_type := Variant" } FILL(BVAL := #ZERO, RET_VAL => #STATUS_FILL, BLK => "DB8000_PART_STATUS".UNIT_01.FIXTURE_1.PART_A)
   END_RUNG
   RUNG wire#w1
      I_Contact( "DB8000_PART_STATUS".UNIT_01.FIXTURE_2.PART_A.STATUS.PRESENT )
      { S7_Templates := "ptr_type := Variant" } FILL(BVAL := #ZERO, RET_VAL => #STATUS_FILL, BLK => "DB8000_PART_STATUS".UNIT_01.FIXTURE_2.PART_A)
   END_RUNG
   RUNG wire#w1
      I_Contact( "DB8000_PART_STATUS".UNIT_01.FIXTURE_3.PART_A.STATUS.PRESENT )
      { S7_Templates := "ptr_type := Variant" } FILL(BVAL := #ZERO, RET_VAL => #STATUS_FILL, BLK => "DB8000_PART_STATUS".UNIT_01.FIXTURE_3.PART_A)
   END_RUNG
   RUNG wire#w1
      I_Contact( "DB8000_PART_STATUS".UNIT_01.FIXTURE_4.PART_A.STATUS.PRESENT )
      { S7_Templates := "ptr_type := Variant" } FILL(BVAL := #ZERO, RET_VAL => #STATUS_FILL, BLK => "DB8000_PART_STATUS".UNIT_01.FIXTURE_4.PART_A)
   END_RUNG
   // the same network as SCL:
   #_w1 := "M_ONE";
   IF "M_ONE" AND NOT "DB8000_PART_STATUS".UNIT_01.FIXTURE_1.PART_A.STATUS.PRESENT THEN
       #STATUS_FILL := FILL(BVAL := #ZERO, BLK => "DB8000_PART_STATUS".UNIT_01.FIXTURE_1.PART_A);
   END_IF;
   IF #_w1 AND NOT "DB8000_PART_STATUS".UNIT_01.FIXTURE_2.PART_A.STATUS.PRESENT THEN
       #STATUS_FILL := FILL(BVAL := #ZERO, BLK => "DB8000_PART_STATUS".UNIT_01.FIXTURE_2.PART_A);
   END_IF;
   IF #_w1 AND NOT "DB8000_PART_STATUS".UNIT_01.FIXTURE_3.PART_A.STATUS.PRESENT THEN
       #STATUS_FILL := FILL(BVAL := #ZERO, BLK => "DB8000_PART_STATUS".UNIT_01.FIXTURE_3.PART_A);
   END_IF;
   IF #_w1 AND NOT "DB8000_PART_STATUS".UNIT_01.FIXTURE_4.PART_A.STATUS.PRESENT THEN
       #STATUS_FILL := FILL(BVAL := #ZERO, BLK => "DB8000_PART_STATUS".UNIT_01.FIXTURE_4.PART_A);
   END_IF;
END_REGION

REGION Network 19: PART A STATION 1, 2, 3, 4 RESET STATUS TO ZERO
   RUNG wire#powerrail
      Contact( "DB4000_FIX_TABLE_POSITIONS".UNIT_01.AXIS_E10_NOT_DEFINED_POS )
      wire#w1
      { S7_Templates := "ptr_type := Variant" } FILL(BVAL := #ZERO, RET_VAL => #STATUS_BLKMOV, BLK => "DB8000_PART_STATUS".UNIT_01.STATION_1.PART_A)
      wire#w2
      R_Coil( "DB8000_PART_STATUS".UNIT_01.STATION_1.PART_A.STATUS.PRESENT )
   END_RUNG
   RUNG wire#w2
      R_Coil( "DB8000_PART_STATUS".UNIT_01.STATION_1.PART_A.STATUS.OK )
   END_RUNG
   RUNG wire#w1
      { S7_Templates := "ptr_type := Variant" } FILL(BVAL := #ZERO, RET_VAL => #STATUS_BLKMOV, BLK => "DB8000_PART_STATUS".UNIT_01.STATION_2.PART_A)
      wire#w3
      R_Coil( "DB8000_PART_STATUS".UNIT_01.STATION_2.PART_A.STATUS.PRESENT )
   END_RUNG
   RUNG wire#w3
      R_Coil( "DB8000_PART_STATUS".UNIT_01.STATION_2.PART_A.STATUS.OK )
   END_RUNG
   RUNG wire#w1
      { S7_Templates := "ptr_type := Variant" } FILL(BVAL := #ZERO, RET_VAL => #STATUS_BLKMOV, BLK => "DB8000_PART_STATUS".UNIT_01.STATION_3.PART_A)
      wire#w4
      R_Coil( "DB8000_PART_STATUS".UNIT_01.STATION_3.PART_A.STATUS.PRESENT )
   END_RUNG
   RUNG wire#w4
      R_Coil( "DB8000_PART_STATUS".UNIT_01.STATION_3.PART_A.STATUS.OK )
   END_RUNG
   RUNG wire#w1
      { S7_Templates := "ptr_type := Variant" } FILL(BVAL := #ZERO, RET_VAL => #STATUS_BLKMOV, BLK => "DB8000_PART_STATUS".UNIT_01.STATION_4.PART_A)
      wire#w5
      R_Coil( "DB8000_PART_STATUS".UNIT_01.STATION_4.PART_A.STATUS.PRESENT )
   END_RUNG
   RUNG wire#w5
      R_Coil( "DB8000_PART_STATUS".UNIT_01.STATION_4.PART_A.STATUS.OK )
   END_RUNG
   // the same network as SCL:
   #_w2 := "DB4000_FIX_TABLE_POSITIONS".UNIT_01.AXIS_E10_NOT_DEFINED_POS;
   #STATUS_BLKMOV := FILL(EN := "DB4000_FIX_TABLE_POSITIONS".UNIT_01.AXIS_E10_NOT_DEFINED_POS,
                          BVAL := #ZERO,
                          BLK => "DB8000_PART_STATUS".UNIT_01.STATION_1.PART_A,
                          ENO => #_w1);
   IF #_w1 THEN
       "DB8000_PART_STATUS".UNIT_01.STATION_1.PART_A.STATUS.PRESENT := FALSE;
       "DB8000_PART_STATUS".UNIT_01.STATION_1.PART_A.STATUS.OK := FALSE;
   END_IF;
   #STATUS_BLKMOV := FILL(EN := #_w2,
                          BVAL := #ZERO,
                          BLK => "DB8000_PART_STATUS".UNIT_01.STATION_2.PART_A,
                          ENO => #_w3);
   IF #_w3 THEN
       "DB8000_PART_STATUS".UNIT_01.STATION_2.PART_A.STATUS.PRESENT := FALSE;
       "DB8000_PART_STATUS".UNIT_01.STATION_2.PART_A.STATUS.OK := FALSE;
   END_IF;
   #STATUS_BLKMOV := FILL(EN := #_w2,
                          BVAL := #ZERO,
                          BLK => "DB8000_PART_STATUS".UNIT_01.STATION_3.PART_A,
                          ENO => #_w4);
   IF #_w4 THEN
       "DB8000_PART_STATUS".UNIT_01.STATION_3.PART_A.STATUS.PRESENT := FALSE;
       "DB8000_PART_STATUS".UNIT_01.STATION_3.PART_A.STATUS.OK := FALSE;
   END_IF;
   #STATUS_BLKMOV := FILL(EN := #_w2,
                          BVAL := #ZERO,
                          BLK => "DB8000_PART_STATUS".UNIT_01.STATION_4.PART_A,
                          ENO => #_w5);
   IF #_w5 THEN
       "DB8000_PART_STATUS".UNIT_01.STATION_4.PART_A.STATUS.PRESENT := FALSE;
       "DB8000_PART_STATUS".UNIT_01.STATION_4.PART_A.STATUS.OK := FALSE;
   END_IF;
END_REGION

REGION Network 20: PART A FIXTURE 1 COLOR STATUS
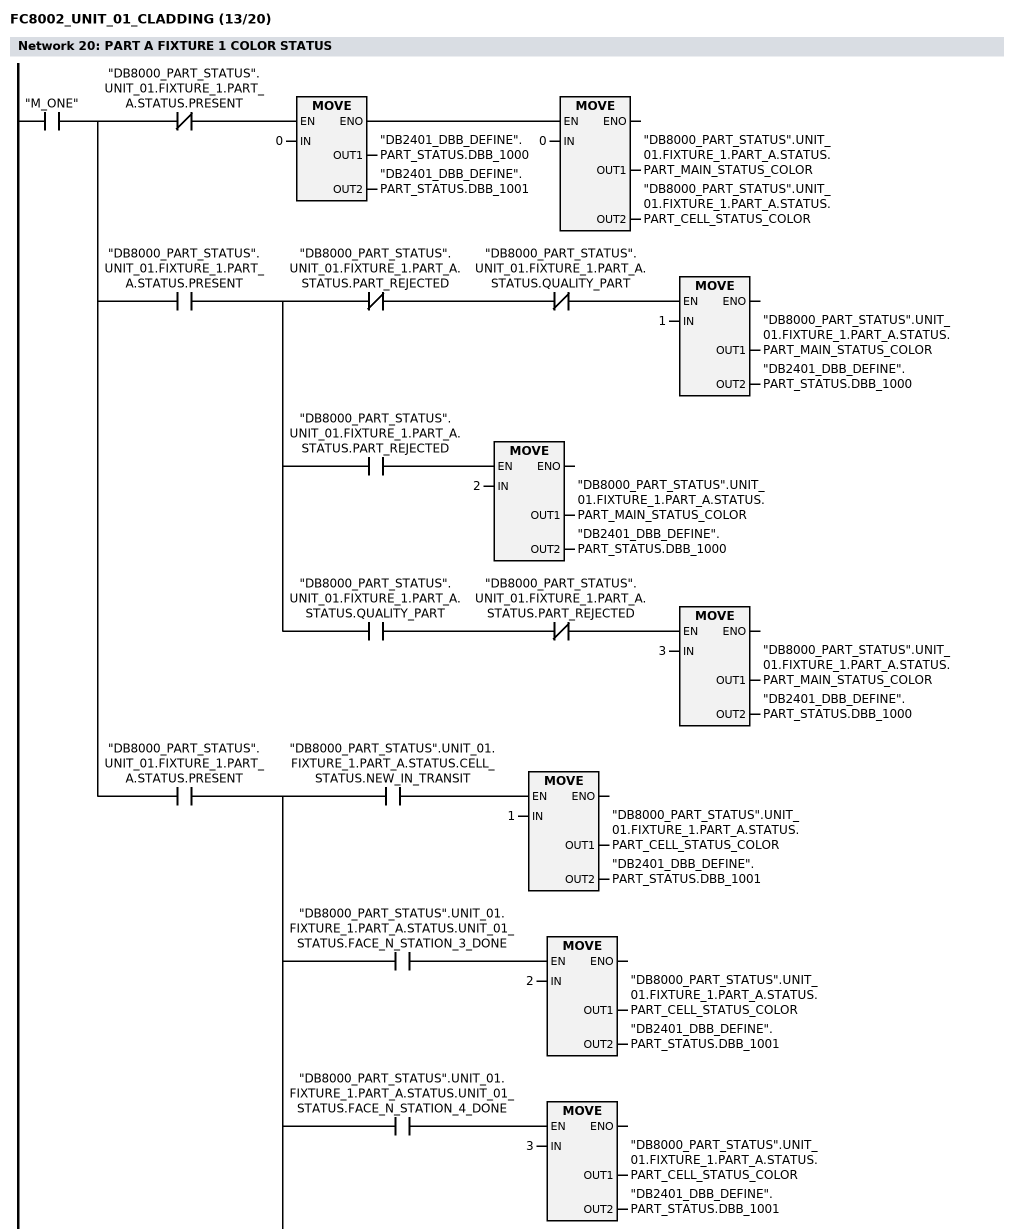
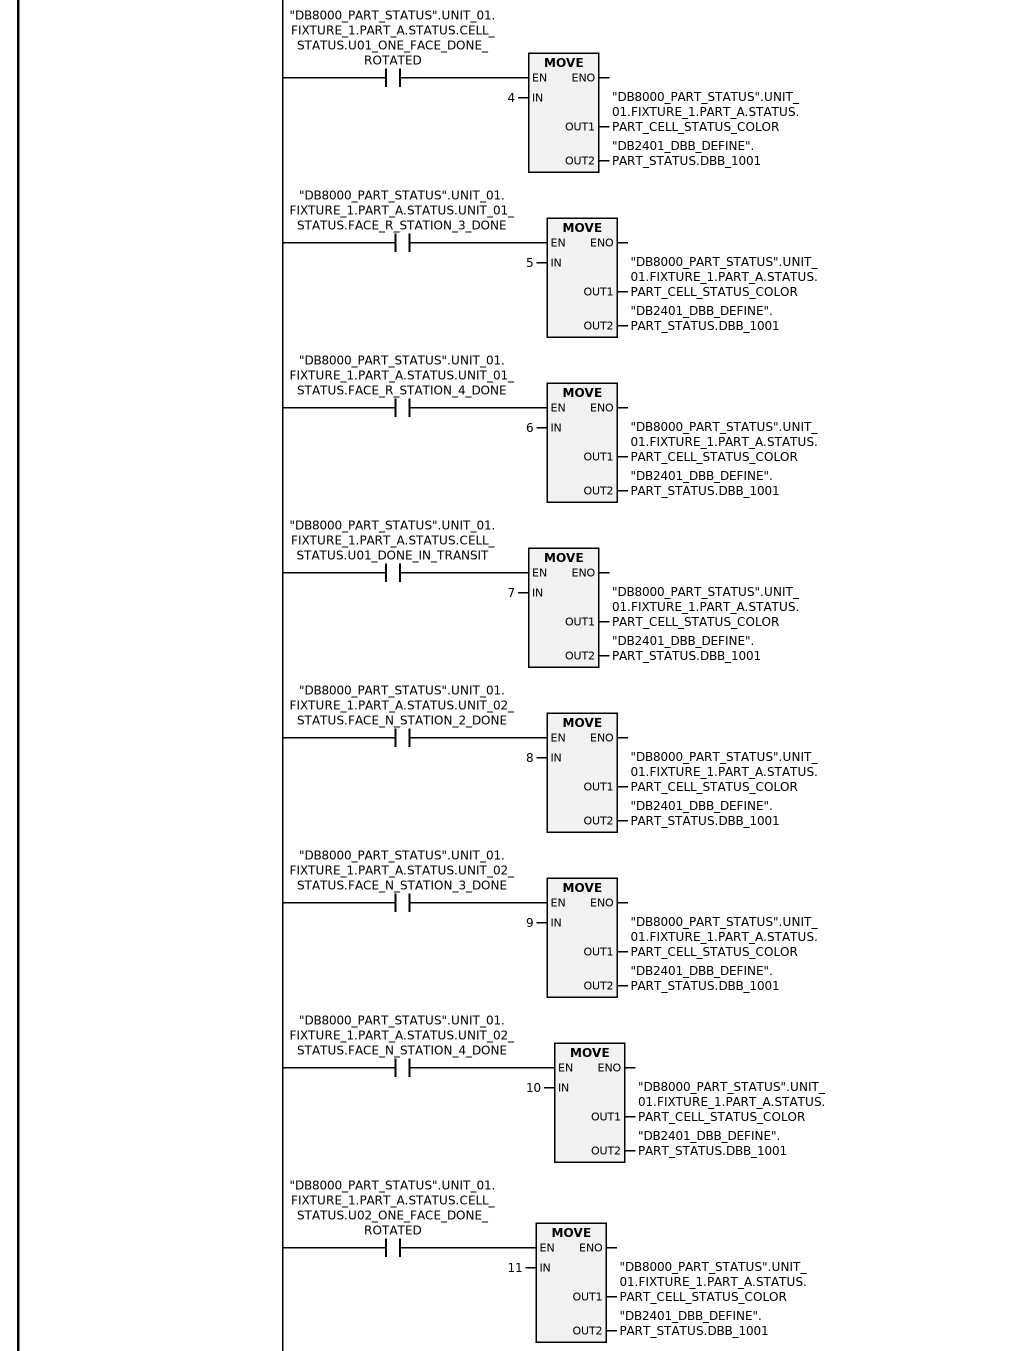
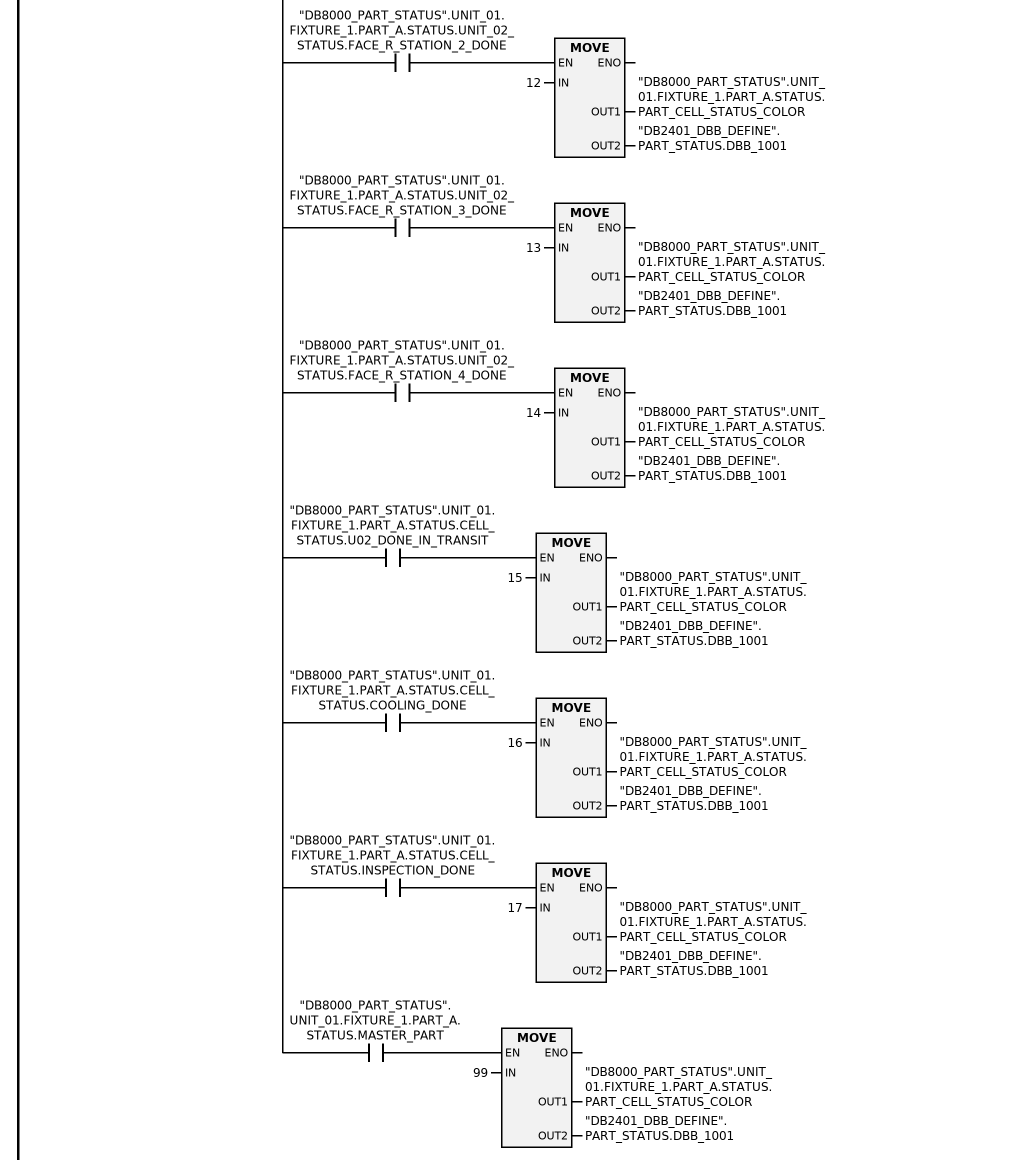
   RUNG wire#powerrail
      Contact( "M_ONE" )
      wire#w1
      I_Contact( "DB8000_PART_STATUS".UNIT_01.FIXTURE_1.PART_A.STATUS.PRESENT )
      { S7_GenerateENO := "TRUE" } Move(in := 0, out1 => "DB2401_DBB_DEFINE".PART_STATUS.DBB_1000, out2 => "DB2401_DBB_DEFINE".PART_STATUS.DBB_1001)
      { S7_GenerateENO := "TRUE" } Move(in := 0, out1 => "DB8000_PART_STATUS".UNIT_01.FIXTURE_1.PART_A.STATUS.PART_MAIN_STATUS_COLOR, out2 => "DB8000_PART_STATUS".UNIT_01.FIXTURE_1.PART_A.STATUS.PART_CELL_STATUS_COLOR)
   END_RUNG
   RUNG wire#w1
      Contact( "DB8000_PART_STATUS".UNIT_01.FIXTURE_1.PART_A.STATUS.PRESENT )
      wire#w2
      I_Contact( "DB8000_PART_STATUS".UNIT_01.FIXTURE_1.PART_A.STATUS.PART_REJECTED )
      I_Contact( "DB8000_PART_STATUS".UNIT_01.FIXTURE_1.PART_A.STATUS.QUALITY_PART )
      { S7_GenerateENO := "TRUE" } Move(in := 1, out1 => "DB8000_PART_STATUS".UNIT_01.FIXTURE_1.PART_A.STATUS.PART_MAIN_STATUS_COLOR, out2 => "DB2401_DBB_DEFINE".PART_STATUS.DBB_1000)
   END_RUNG
   RUNG wire#w2
      Contact( "DB8000_PART_STATUS".UNIT_01.FIXTURE_1.PART_A.STATUS.PART_REJECTED )
      { S7_GenerateENO := "TRUE" } Move(in := 2, out1 => "DB8000_PART_STATUS".UNIT_01.FIXTURE_1.PART_A.STATUS.PART_MAIN_STATUS_COLOR, out2 => "DB2401_DBB_DEFINE".PART_STATUS.DBB_1000)
   END_RUNG
   RUNG wire#w2
      Contact( "DB8000_PART_STATUS".UNIT_01.FIXTURE_1.PART_A.STATUS.QUALITY_PART )
      I_Contact( "DB8000_PART_STATUS".UNIT_01.FIXTURE_1.PART_A.STATUS.PART_REJECTED )
      { S7_GenerateENO := "TRUE" } Move(in := 3, out1 => "DB8000_PART_STATUS".UNIT_01.FIXTURE_1.PART_A.STATUS.PART_MAIN_STATUS_COLOR, out2 => "DB2401_DBB_DEFINE".PART_STATUS.DBB_1000)
   END_RUNG
   RUNG wire#w1
      Contact( "DB8000_PART_STATUS".UNIT_01.FIXTURE_1.PART_A.STATUS.PRESENT )
      wire#w3
      Contact( "DB8000_PART_STATUS".UNIT_01.FIXTURE_1.PART_A.STATUS.CELL_STATUS.NEW_IN_TRANSIT )
      { S7_GenerateENO := "TRUE" } Move(in := 1, out1 => "DB8000_PART_STATUS".UNIT_01.FIXTURE_1.PART_A.STATUS.PART_CELL_STATUS_COLOR, out2 => "DB2401_DBB_DEFINE".PART_STATUS.DBB_1001)
   END_RUNG
   RUNG wire#w3
      Contact( "DB8000_PART_STATUS".UNIT_01.FIXTURE_1.PART_A.STATUS.UNIT_01_STATUS.FACE_N_STATION_3_DONE )
      { S7_GenerateENO := "TRUE" } Move(in := 2, out1 => "DB8000_PART_STATUS".UNIT_01.FIXTURE_1.PART_A.STATUS.PART_CELL_STATUS_COLOR, out2 => "DB2401_DBB_DEFINE".PART_STATUS.DBB_1001)
   END_RUNG
   RUNG wire#w3
      Contact( "DB8000_PART_STATUS".UNIT_01.FIXTURE_1.PART_A.STATUS.UNIT_01_STATUS.FACE_N_STATION_4_DONE )
      { S7_GenerateENO := "TRUE" } Move(in := 3, out1 => "DB8000_PART_STATUS".UNIT_01.FIXTURE_1.PART_A.STATUS.PART_CELL_STATUS_COLOR, out2 => "DB2401_DBB_DEFINE".PART_STATUS.DBB_1001)
   END_RUNG
   RUNG wire#w3
      Contact( "DB8000_PART_STATUS".UNIT_01.FIXTURE_1.PART_A.STATUS.CELL_STATUS.U01_ONE_FACE_DONE_ROTATED )
      { S7_GenerateENO := "TRUE" } Move(in := 4, out1 => "DB8000_PART_STATUS".UNIT_01.FIXTURE_1.PART_A.STATUS.PART_CELL_STATUS_COLOR, out2 => "DB2401_DBB_DEFINE".PART_STATUS.DBB_1001)
   END_RUNG
   RUNG wire#w3
      Contact( "DB8000_PART_STATUS".UNIT_01.FIXTURE_1.PART_A.STATUS.UNIT_01_STATUS.FACE_R_STATION_3_DONE )
      { S7_GenerateENO := "TRUE" } Move(in := 5, out1 => "DB8000_PART_STATUS".UNIT_01.FIXTURE_1.PART_A.STATUS.PART_CELL_STATUS_COLOR, out2 => "DB2401_DBB_DEFINE".PART_STATUS.DBB_1001)
   END_RUNG
   RUNG wire#w3
      Contact( "DB8000_PART_STATUS".UNIT_01.FIXTURE_1.PART_A.STATUS.UNIT_01_STATUS.FACE_R_STATION_4_DONE )
      { S7_GenerateENO := "TRUE" } Move(in := 6, out1 => "DB8000_PART_STATUS".UNIT_01.FIXTURE_1.PART_A.STATUS.PART_CELL_STATUS_COLOR, out2 => "DB2401_DBB_DEFINE".PART_STATUS.DBB_1001)
   END_RUNG
   RUNG wire#w3
      Contact( "DB8000_PART_STATUS".UNIT_01.FIXTURE_1.PART_A.STATUS.CELL_STATUS.U01_DONE_IN_TRANSIT )
      { S7_GenerateENO := "TRUE" } Move(in := 7, out1 => "DB8000_PART_STATUS".UNIT_01.FIXTURE_1.PART_A.STATUS.PART_CELL_STATUS_COLOR, out2 => "DB2401_DBB_DEFINE".PART_STATUS.DBB_1001)
   END_RUNG
   RUNG wire#w3
      Contact( "DB8000_PART_STATUS".UNIT_01.FIXTURE_1.PART_A.STATUS.UNIT_02_STATUS.FACE_N_STATION_2_DONE )
      { S7_GenerateENO := "TRUE" } Move(in := 8, out1 => "DB8000_PART_STATUS".UNIT_01.FIXTURE_1.PART_A.STATUS.PART_CELL_STATUS_COLOR, out2 => "DB2401_DBB_DEFINE".PART_STATUS.DBB_1001)
   END_RUNG
   RUNG wire#w3
      Contact( "DB8000_PART_STATUS".UNIT_01.FIXTURE_1.PART_A.STATUS.UNIT_02_STATUS.FACE_N_STATION_3_DONE )
      { S7_GenerateENO := "TRUE" } Move(in := 9, out1 => "DB8000_PART_STATUS".UNIT_01.FIXTURE_1.PART_A.STATUS.PART_CELL_STATUS_COLOR, out2 => "DB2401_DBB_DEFINE".PART_STATUS.DBB_1001)
   END_RUNG
   RUNG wire#w3
      Contact( "DB8000_PART_STATUS".UNIT_01.FIXTURE_1.PART_A.STATUS.UNIT_02_STATUS.FACE_N_STATION_4_DONE )
      { S7_GenerateENO := "TRUE" } Move(in := 10, out1 => "DB8000_PART_STATUS".UNIT_01.FIXTURE_1.PART_A.STATUS.PART_CELL_STATUS_COLOR, out2 => "DB2401_DBB_DEFINE".PART_STATUS.DBB_1001)
   END_RUNG
   RUNG wire#w3
      Contact( "DB8000_PART_STATUS".UNIT_01.FIXTURE_1.PART_A.STATUS.CELL_STATUS.U02_ONE_FACE_DONE_ROTATED )
      { S7_GenerateENO := "TRUE" } Move(in := 11, out1 => "DB8000_PART_STATUS".UNIT_01.FIXTURE_1.PART_A.STATUS.PART_CELL_STATUS_COLOR, out2 => "DB2401_DBB_DEFINE".PART_STATUS.DBB_1001)
   END_RUNG
   RUNG wire#w3
      Contact( "DB8000_PART_STATUS".UNIT_01.FIXTURE_1.PART_A.STATUS.UNIT_02_STATUS.FACE_R_STATION_2_DONE )
      { S7_GenerateENO := "TRUE" } Move(in := 12, out1 => "DB8000_PART_STATUS".UNIT_01.FIXTURE_1.PART_A.STATUS.PART_CELL_STATUS_COLOR, out2 => "DB2401_DBB_DEFINE".PART_STATUS.DBB_1001)
   END_RUNG
   RUNG wire#w3
      Contact( "DB8000_PART_STATUS".UNIT_01.FIXTURE_1.PART_A.STATUS.UNIT_02_STATUS.FACE_R_STATION_3_DONE )
      Move(in := 13, out1 => "DB8000_PART_STATUS".UNIT_01.FIXTURE_1.PART_A.STATUS.PART_CELL_STATUS_COLOR, out2 => "DB2401_DBB_DEFINE".PART_STATUS.DBB_1001)
   END_RUNG
   RUNG wire#w3
      Contact( "DB8000_PART_STATUS".UNIT_01.FIXTURE_1.PART_A.STATUS.UNIT_02_STATUS.FACE_R_STATION_4_DONE )
      Move(in := 14, out1 => "DB8000_PART_STATUS".UNIT_01.FIXTURE_1.PART_A.STATUS.PART_CELL_STATUS_COLOR, out2 => "DB2401_DBB_DEFINE".PART_STATUS.DBB_1001)
   END_RUNG
   RUNG wire#w3
      Contact( "DB8000_PART_STATUS".UNIT_01.FIXTURE_1.PART_A.STATUS.CELL_STATUS.U02_DONE_IN_TRANSIT )
      Move(in := 15, out1 => "DB8000_PART_STATUS".UNIT_01.FIXTURE_1.PART_A.STATUS.PART_CELL_STATUS_COLOR, out2 => "DB2401_DBB_DEFINE".PART_STATUS.DBB_1001)
   END_RUNG
   RUNG wire#w3
      Contact( "DB8000_PART_STATUS".UNIT_01.FIXTURE_1.PART_A.STATUS.CELL_STATUS.COOLING_DONE )
      Move(in := 16, out1 => "DB8000_PART_STATUS".UNIT_01.FIXTURE_1.PART_A.STATUS.PART_CELL_STATUS_COLOR, out2 => "DB2401_DBB_DEFINE".PART_STATUS.DBB_1001)
   END_RUNG
   RUNG wire#w3
      Contact( "DB8000_PART_STATUS".UNIT_01.FIXTURE_1.PART_A.STATUS.CELL_STATUS.INSPECTION_DONE )
      Move(in := 17, out1 => "DB8000_PART_STATUS".UNIT_01.FIXTURE_1.PART_A.STATUS.PART_CELL_STATUS_COLOR, out2 => "DB2401_DBB_DEFINE".PART_STATUS.DBB_1001)
   END_RUNG
   RUNG wire#w3
      Contact( "DB8000_PART_STATUS".UNIT_01.FIXTURE_1.PART_A.STATUS.MASTER_PART )
      Move(in := 99, out1 => "DB8000_PART_STATUS".UNIT_01.FIXTURE_1.PART_A.STATUS.PART_CELL_STATUS_COLOR, out2 => "DB2401_DBB_DEFINE".PART_STATUS.DBB_1001)
   END_RUNG
   // the same network as SCL:
   // ENO of a box is taken as its EN; it also drops when the box reports an error
   IF "M_ONE" AND NOT "DB8000_PART_STATUS".UNIT_01.FIXTURE_1.PART_A.STATUS.PRESENT THEN
       "DB2401_DBB_DEFINE".PART_STATUS.DBB_1000 := 0;
       "DB2401_DBB_DEFINE".PART_STATUS.DBB_1001 := 0;
       "DB8000_PART_STATUS".UNIT_01.FIXTURE_1.PART_A.STATUS.PART_MAIN_STATUS_COLOR := 0;
       "DB8000_PART_STATUS".UNIT_01.FIXTURE_1.PART_A.STATUS.PART_CELL_STATUS_COLOR := 0;
   END_IF;
   #_w1 := "M_ONE" AND "DB8000_PART_STATUS".UNIT_01.FIXTURE_1.PART_A.STATUS.PRESENT;
   IF #_w1 AND NOT "DB8000_PART_STATUS".UNIT_01.FIXTURE_1.PART_A.STATUS.PART_REJECTED AND NOT "DB8000_PART_STATUS".UNIT_01.FIXTURE_1.PART_A.STATUS.QUALITY_PART THEN
       "DB8000_PART_STATUS".UNIT_01.FIXTURE_1.PART_A.STATUS.PART_MAIN_STATUS_COLOR := 1;
       "DB2401_DBB_DEFINE".PART_STATUS.DBB_1000 := 1;
   END_IF;
   IF #_w1 AND "DB8000_PART_STATUS".UNIT_01.FIXTURE_1.PART_A.STATUS.PART_REJECTED THEN
       "DB8000_PART_STATUS".UNIT_01.FIXTURE_1.PART_A.STATUS.PART_MAIN_STATUS_COLOR := 2;
       "DB2401_DBB_DEFINE".PART_STATUS.DBB_1000 := 2;
   END_IF;
   IF #_w1 AND "DB8000_PART_STATUS".UNIT_01.FIXTURE_1.PART_A.STATUS.QUALITY_PART AND NOT "DB8000_PART_STATUS".UNIT_01.FIXTURE_1.PART_A.STATUS.PART_REJECTED THEN
       "DB8000_PART_STATUS".UNIT_01.FIXTURE_1.PART_A.STATUS.PART_MAIN_STATUS_COLOR := 3;
       "DB2401_DBB_DEFINE".PART_STATUS.DBB_1000 := 3;
   END_IF;
   #_w2 := "M_ONE" AND "DB8000_PART_STATUS".UNIT_01.FIXTURE_1.PART_A.STATUS.PRESENT;
   IF #_w2 AND "DB8000_PART_STATUS".UNIT_01.FIXTURE_1.PART_A.STATUS.CELL_STATUS.NEW_IN_TRANSIT THEN
       "DB8000_PART_STATUS".UNIT_01.FIXTURE_1.PART_A.STATUS.PART_CELL_STATUS_COLOR := 1;
       "DB2401_DBB_DEFINE".PART_STATUS.DBB_1001 := 1;
   END_IF;
   IF #_w2 AND "DB8000_PART_STATUS".UNIT_01.FIXTURE_1.PART_A.STATUS.UNIT_01_STATUS.FACE_N_STATION_3_DONE THEN
       "DB8000_PART_STATUS".UNIT_01.FIXTURE_1.PART_A.STATUS.PART_CELL_STATUS_COLOR := 2;
       "DB2401_DBB_DEFINE".PART_STATUS.DBB_1001 := 2;
   END_IF;
   IF #_w2 AND "DB8000_PART_STATUS".UNIT_01.FIXTURE_1.PART_A.STATUS.UNIT_01_STATUS.FACE_N_STATION_4_DONE THEN
       "DB8000_PART_STATUS".UNIT_01.FIXTURE_1.PART_A.STATUS.PART_CELL_STATUS_COLOR := 3;
       "DB2401_DBB_DEFINE".PART_STATUS.DBB_1001 := 3;
   END_IF;
   IF #_w2 AND "DB8000_PART_STATUS".UNIT_01.FIXTURE_1.PART_A.STATUS.CELL_STATUS.U01_ONE_FACE_DONE_ROTATED THEN
       "DB8000_PART_STATUS".UNIT_01.FIXTURE_1.PART_A.STATUS.PART_CELL_STATUS_COLOR := 4;
       "DB2401_DBB_DEFINE".PART_STATUS.DBB_1001 := 4;
   END_IF;
   IF #_w2 AND "DB8000_PART_STATUS".UNIT_01.FIXTURE_1.PART_A.STATUS.UNIT_01_STATUS.FACE_R_STATION_3_DONE THEN
       "DB8000_PART_STATUS".UNIT_01.FIXTURE_1.PART_A.STATUS.PART_CELL_STATUS_COLOR := 5;
       "DB2401_DBB_DEFINE".PART_STATUS.DBB_1001 := 5;
   END_IF;
   IF #_w2 AND "DB8000_PART_STATUS".UNIT_01.FIXTURE_1.PART_A.STATUS.UNIT_01_STATUS.FACE_R_STATION_4_DONE THEN
       "DB8000_PART_STATUS".UNIT_01.FIXTURE_1.PART_A.STATUS.PART_CELL_STATUS_COLOR := 6;
       "DB2401_DBB_DEFINE".PART_STATUS.DBB_1001 := 6;
   END_IF;
   IF #_w2 AND "DB8000_PART_STATUS".UNIT_01.FIXTURE_1.PART_A.STATUS.CELL_STATUS.U01_DONE_IN_TRANSIT THEN
       "DB8000_PART_STATUS".UNIT_01.FIXTURE_1.PART_A.STATUS.PART_CELL_STATUS_COLOR := 7;
       "DB2401_DBB_DEFINE".PART_STATUS.DBB_1001 := 7;
   END_IF;
   IF #_w2 AND "DB8000_PART_STATUS".UNIT_01.FIXTURE_1.PART_A.STATUS.UNIT_02_STATUS.FACE_N_STATION_2_DONE THEN
       "DB8000_PART_STATUS".UNIT_01.FIXTURE_1.PART_A.STATUS.PART_CELL_STATUS_COLOR := 8;
       "DB2401_DBB_DEFINE".PART_STATUS.DBB_1001 := 8;
   END_IF;
   IF #_w2 AND "DB8000_PART_STATUS".UNIT_01.FIXTURE_1.PART_A.STATUS.UNIT_02_STATUS.FACE_N_STATION_3_DONE THEN
       "DB8000_PART_STATUS".UNIT_01.FIXTURE_1.PART_A.STATUS.PART_CELL_STATUS_COLOR := 9;
       "DB2401_DBB_DEFINE".PART_STATUS.DBB_1001 := 9;
   END_IF;
   IF #_w2 AND "DB8000_PART_STATUS".UNIT_01.FIXTURE_1.PART_A.STATUS.UNIT_02_STATUS.FACE_N_STATION_4_DONE THEN
       "DB8000_PART_STATUS".UNIT_01.FIXTURE_1.PART_A.STATUS.PART_CELL_STATUS_COLOR := 10;
       "DB2401_DBB_DEFINE".PART_STATUS.DBB_1001 := 10;
   END_IF;
   IF #_w2 AND "DB8000_PART_STATUS".UNIT_01.FIXTURE_1.PART_A.STATUS.CELL_STATUS.U02_ONE_FACE_DONE_ROTATED THEN
       "DB8000_PART_STATUS".UNIT_01.FIXTURE_1.PART_A.STATUS.PART_CELL_STATUS_COLOR := 11;
       "DB2401_DBB_DEFINE".PART_STATUS.DBB_1001 := 11;
   END_IF;
   IF #_w2 AND "DB8000_PART_STATUS".UNIT_01.FIXTURE_1.PART_A.STATUS.UNIT_02_STATUS.FACE_R_STATION_2_DONE THEN
       "DB8000_PART_STATUS".UNIT_01.FIXTURE_1.PART_A.STATUS.PART_CELL_STATUS_COLOR := 12;
       "DB2401_DBB_DEFINE".PART_STATUS.DBB_1001 := 12;
   END_IF;
   IF #_w2 AND "DB8000_PART_STATUS".UNIT_01.FIXTURE_1.PART_A.STATUS.UNIT_02_STATUS.FACE_R_STATION_3_DONE THEN
       "DB8000_PART_STATUS".UNIT_01.FIXTURE_1.PART_A.STATUS.PART_CELL_STATUS_COLOR := 13;
       "DB2401_DBB_DEFINE".PART_STATUS.DBB_1001 := 13;
   END_IF;
   IF #_w2 AND "DB8000_PART_STATUS".UNIT_01.FIXTURE_1.PART_A.STATUS.UNIT_02_STATUS.FACE_R_STATION_4_DONE THEN
       "DB8000_PART_STATUS".UNIT_01.FIXTURE_1.PART_A.STATUS.PART_CELL_STATUS_COLOR := 14;
       "DB2401_DBB_DEFINE".PART_STATUS.DBB_1001 := 14;
   END_IF;
   IF #_w2 AND "DB8000_PART_STATUS".UNIT_01.FIXTURE_1.PART_A.STATUS.CELL_STATUS.U02_DONE_IN_TRANSIT THEN
       "DB8000_PART_STATUS".UNIT_01.FIXTURE_1.PART_A.STATUS.PART_CELL_STATUS_COLOR := 15;
       "DB2401_DBB_DEFINE".PART_STATUS.DBB_1001 := 15;
   END_IF;
   IF #_w2 AND "DB8000_PART_STATUS".UNIT_01.FIXTURE_1.PART_A.STATUS.CELL_STATUS.COOLING_DONE THEN
       "DB8000_PART_STATUS".UNIT_01.FIXTURE_1.PART_A.STATUS.PART_CELL_STATUS_COLOR := 16;
       "DB2401_DBB_DEFINE".PART_STATUS.DBB_1001 := 16;
   END_IF;
   IF #_w2 AND "DB8000_PART_STATUS".UNIT_01.FIXTURE_1.PART_A.STATUS.CELL_STATUS.INSPECTION_DONE THEN
       "DB8000_PART_STATUS".UNIT_01.FIXTURE_1.PART_A.STATUS.PART_CELL_STATUS_COLOR := 17;
       "DB2401_DBB_DEFINE".PART_STATUS.DBB_1001 := 17;
   END_IF;
   IF #_w2 AND "DB8000_PART_STATUS".UNIT_01.FIXTURE_1.PART_A.STATUS.MASTER_PART THEN
       "DB8000_PART_STATUS".UNIT_01.FIXTURE_1.PART_A.STATUS.PART_CELL_STATUS_COLOR := 99;
       "DB2401_DBB_DEFINE".PART_STATUS.DBB_1001 := 99;
   END_IF;
END_REGION

REGION Network 21: PART A FIXTURE 2 COLOR STATUS
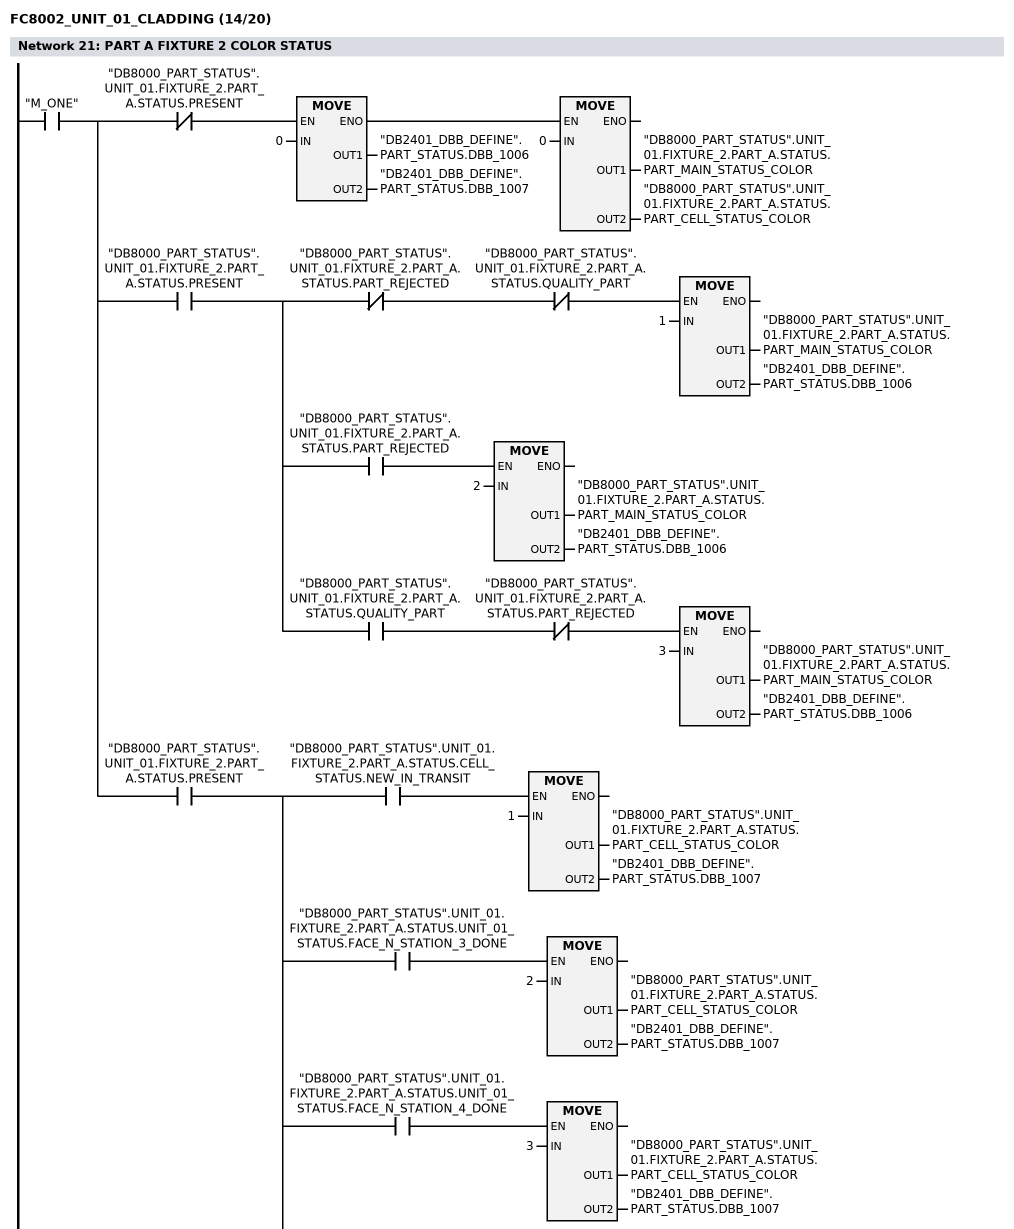
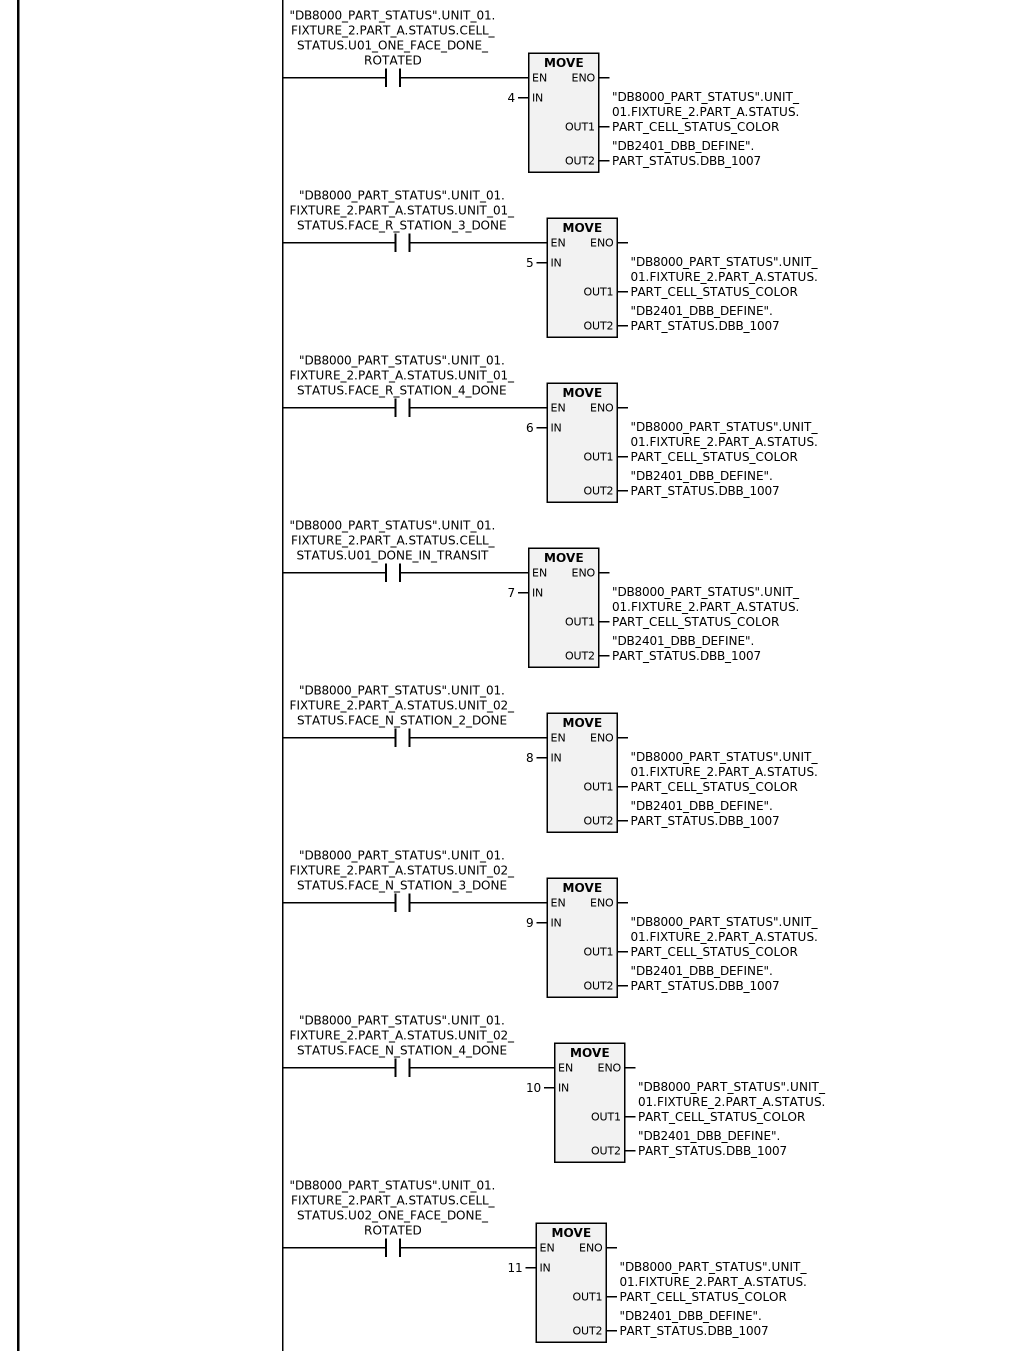
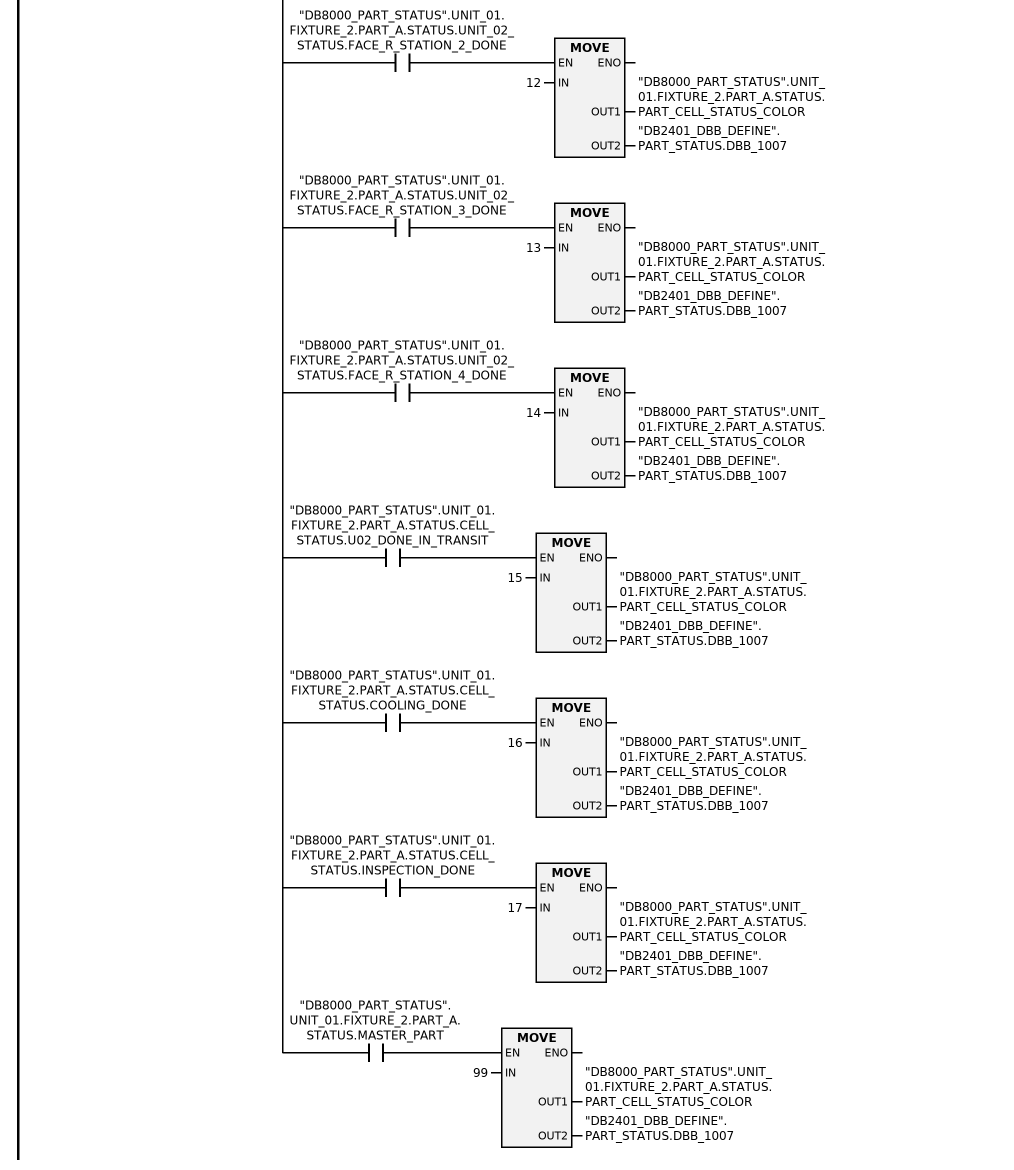
   RUNG wire#powerrail
      Contact( "M_ONE" )
      wire#w1
      I_Contact( "DB8000_PART_STATUS".UNIT_01.FIXTURE_2.PART_A.STATUS.PRESENT )
      { S7_GenerateENO := "TRUE" } Move(in := 0, out1 => "DB2401_DBB_DEFINE".PART_STATUS.DBB_1006, out2 => "DB2401_DBB_DEFINE".PART_STATUS.DBB_1007)
      { S7_GenerateENO := "TRUE" } Move(in := 0, out1 => "DB8000_PART_STATUS".UNIT_01.FIXTURE_2.PART_A.STATUS.PART_MAIN_STATUS_COLOR, out2 => "DB8000_PART_STATUS".UNIT_01.FIXTURE_2.PART_A.STATUS.PART_CELL_STATUS_COLOR)
   END_RUNG
   RUNG wire#w1
      Contact( "DB8000_PART_STATUS".UNIT_01.FIXTURE_2.PART_A.STATUS.PRESENT )
      wire#w2
      I_Contact( "DB8000_PART_STATUS".UNIT_01.FIXTURE_2.PART_A.STATUS.PART_REJECTED )
      I_Contact( "DB8000_PART_STATUS".UNIT_01.FIXTURE_2.PART_A.STATUS.QUALITY_PART )
      { S7_GenerateENO := "TRUE" } Move(in := 1, out1 => "DB8000_PART_STATUS".UNIT_01.FIXTURE_2.PART_A.STATUS.PART_MAIN_STATUS_COLOR, out2 => "DB2401_DBB_DEFINE".PART_STATUS.DBB_1006)
   END_RUNG
   RUNG wire#w2
      Contact( "DB8000_PART_STATUS".UNIT_01.FIXTURE_2.PART_A.STATUS.PART_REJECTED )
      { S7_GenerateENO := "TRUE" } Move(in := 2, out1 => "DB8000_PART_STATUS".UNIT_01.FIXTURE_2.PART_A.STATUS.PART_MAIN_STATUS_COLOR, out2 => "DB2401_DBB_DEFINE".PART_STATUS.DBB_1006)
   END_RUNG
   RUNG wire#w2
      Contact( "DB8000_PART_STATUS".UNIT_01.FIXTURE_2.PART_A.STATUS.QUALITY_PART )
      I_Contact( "DB8000_PART_STATUS".UNIT_01.FIXTURE_2.PART_A.STATUS.PART_REJECTED )
      { S7_GenerateENO := "TRUE" } Move(in := 3, out1 => "DB8000_PART_STATUS".UNIT_01.FIXTURE_2.PART_A.STATUS.PART_MAIN_STATUS_COLOR, out2 => "DB2401_DBB_DEFINE".PART_STATUS.DBB_1006)
   END_RUNG
   RUNG wire#w1
      Contact( "DB8000_PART_STATUS".UNIT_01.FIXTURE_2.PART_A.STATUS.PRESENT )
      wire#w3
      Contact( "DB8000_PART_STATUS".UNIT_01.FIXTURE_2.PART_A.STATUS.CELL_STATUS.NEW_IN_TRANSIT )
      { S7_GenerateENO := "TRUE" } Move(in := 1, out1 => "DB8000_PART_STATUS".UNIT_01.FIXTURE_2.PART_A.STATUS.PART_CELL_STATUS_COLOR, out2 => "DB2401_DBB_DEFINE".PART_STATUS.DBB_1007)
   END_RUNG
   RUNG wire#w3
      Contact( "DB8000_PART_STATUS".UNIT_01.FIXTURE_2.PART_A.STATUS.UNIT_01_STATUS.FACE_N_STATION_3_DONE )
      { S7_GenerateENO := "TRUE" } Move(in := 2, out1 => "DB8000_PART_STATUS".UNIT_01.FIXTURE_2.PART_A.STATUS.PART_CELL_STATUS_COLOR, out2 => "DB2401_DBB_DEFINE".PART_STATUS.DBB_1007)
   END_RUNG
   RUNG wire#w3
      Contact( "DB8000_PART_STATUS".UNIT_01.FIXTURE_2.PART_A.STATUS.UNIT_01_STATUS.FACE_N_STATION_4_DONE )
      { S7_GenerateENO := "TRUE" } Move(in := 3, out1 => "DB8000_PART_STATUS".UNIT_01.FIXTURE_2.PART_A.STATUS.PART_CELL_STATUS_COLOR, out2 => "DB2401_DBB_DEFINE".PART_STATUS.DBB_1007)
   END_RUNG
   RUNG wire#w3
      Contact( "DB8000_PART_STATUS".UNIT_01.FIXTURE_2.PART_A.STATUS.CELL_STATUS.U01_ONE_FACE_DONE_ROTATED )
      { S7_GenerateENO := "TRUE" } Move(in := 4, out1 => "DB8000_PART_STATUS".UNIT_01.FIXTURE_2.PART_A.STATUS.PART_CELL_STATUS_COLOR, out2 => "DB2401_DBB_DEFINE".PART_STATUS.DBB_1007)
   END_RUNG
   RUNG wire#w3
      Contact( "DB8000_PART_STATUS".UNIT_01.FIXTURE_2.PART_A.STATUS.UNIT_01_STATUS.FACE_R_STATION_3_DONE )
      { S7_GenerateENO := "TRUE" } Move(in := 5, out1 => "DB8000_PART_STATUS".UNIT_01.FIXTURE_2.PART_A.STATUS.PART_CELL_STATUS_COLOR, out2 => "DB2401_DBB_DEFINE".PART_STATUS.DBB_1007)
   END_RUNG
   RUNG wire#w3
      Contact( "DB8000_PART_STATUS".UNIT_01.FIXTURE_2.PART_A.STATUS.UNIT_01_STATUS.FACE_R_STATION_4_DONE )
      { S7_GenerateENO := "TRUE" } Move(in := 6, out1 => "DB8000_PART_STATUS".UNIT_01.FIXTURE_2.PART_A.STATUS.PART_CELL_STATUS_COLOR, out2 => "DB2401_DBB_DEFINE".PART_STATUS.DBB_1007)
   END_RUNG
   RUNG wire#w3
      Contact( "DB8000_PART_STATUS".UNIT_01.FIXTURE_2.PART_A.STATUS.CELL_STATUS.U01_DONE_IN_TRANSIT )
      { S7_GenerateENO := "TRUE" } Move(in := 7, out1 => "DB8000_PART_STATUS".UNIT_01.FIXTURE_2.PART_A.STATUS.PART_CELL_STATUS_COLOR, out2 => "DB2401_DBB_DEFINE".PART_STATUS.DBB_1007)
   END_RUNG
   RUNG wire#w3
      Contact( "DB8000_PART_STATUS".UNIT_01.FIXTURE_2.PART_A.STATUS.UNIT_02_STATUS.FACE_N_STATION_2_DONE )
      { S7_GenerateENO := "TRUE" } Move(in := 8, out1 => "DB8000_PART_STATUS".UNIT_01.FIXTURE_2.PART_A.STATUS.PART_CELL_STATUS_COLOR, out2 => "DB2401_DBB_DEFINE".PART_STATUS.DBB_1007)
   END_RUNG
   RUNG wire#w3
      Contact( "DB8000_PART_STATUS".UNIT_01.FIXTURE_2.PART_A.STATUS.UNIT_02_STATUS.FACE_N_STATION_3_DONE )
      { S7_GenerateENO := "TRUE" } Move(in := 9, out1 => "DB8000_PART_STATUS".UNIT_01.FIXTURE_2.PART_A.STATUS.PART_CELL_STATUS_COLOR, out2 => "DB2401_DBB_DEFINE".PART_STATUS.DBB_1007)
   END_RUNG
   RUNG wire#w3
      Contact( "DB8000_PART_STATUS".UNIT_01.FIXTURE_2.PART_A.STATUS.UNIT_02_STATUS.FACE_N_STATION_4_DONE )
      { S7_GenerateENO := "TRUE" } Move(in := 10, out1 => "DB8000_PART_STATUS".UNIT_01.FIXTURE_2.PART_A.STATUS.PART_CELL_STATUS_COLOR, out2 => "DB2401_DBB_DEFINE".PART_STATUS.DBB_1007)
   END_RUNG
   RUNG wire#w3
      Contact( "DB8000_PART_STATUS".UNIT_01.FIXTURE_2.PART_A.STATUS.CELL_STATUS.U02_ONE_FACE_DONE_ROTATED )
      { S7_GenerateENO := "TRUE" } Move(in := 11, out1 => "DB8000_PART_STATUS".UNIT_01.FIXTURE_2.PART_A.STATUS.PART_CELL_STATUS_COLOR, out2 => "DB2401_DBB_DEFINE".PART_STATUS.DBB_1007)
   END_RUNG
   RUNG wire#w3
      Contact( "DB8000_PART_STATUS".UNIT_01.FIXTURE_2.PART_A.STATUS.UNIT_02_STATUS.FACE_R_STATION_2_DONE )
      { S7_GenerateENO := "TRUE" } Move(in := 12, out1 => "DB8000_PART_STATUS".UNIT_01.FIXTURE_2.PART_A.STATUS.PART_CELL_STATUS_COLOR, out2 => "DB2401_DBB_DEFINE".PART_STATUS.DBB_1007)
   END_RUNG
   RUNG wire#w3
      Contact( "DB8000_PART_STATUS".UNIT_01.FIXTURE_2.PART_A.STATUS.UNIT_02_STATUS.FACE_R_STATION_3_DONE )
      Move(in := 13, out1 => "DB8000_PART_STATUS".UNIT_01.FIXTURE_2.PART_A.STATUS.PART_CELL_STATUS_COLOR, out2 => "DB2401_DBB_DEFINE".PART_STATUS.DBB_1007)
   END_RUNG
   RUNG wire#w3
      Contact( "DB8000_PART_STATUS".UNIT_01.FIXTURE_2.PART_A.STATUS.UNIT_02_STATUS.FACE_R_STATION_4_DONE )
      Move(in := 14, out1 => "DB8000_PART_STATUS".UNIT_01.FIXTURE_2.PART_A.STATUS.PART_CELL_STATUS_COLOR, out2 => "DB2401_DBB_DEFINE".PART_STATUS.DBB_1007)
   END_RUNG
   RUNG wire#w3
      Contact( "DB8000_PART_STATUS".UNIT_01.FIXTURE_2.PART_A.STATUS.CELL_STATUS.U02_DONE_IN_TRANSIT )
      Move(in := 15, out1 => "DB8000_PART_STATUS".UNIT_01.FIXTURE_2.PART_A.STATUS.PART_CELL_STATUS_COLOR, out2 => "DB2401_DBB_DEFINE".PART_STATUS.DBB_1007)
   END_RUNG
   RUNG wire#w3
      Contact( "DB8000_PART_STATUS".UNIT_01.FIXTURE_2.PART_A.STATUS.CELL_STATUS.COOLING_DONE )
      Move(in := 16, out1 => "DB8000_PART_STATUS".UNIT_01.FIXTURE_2.PART_A.STATUS.PART_CELL_STATUS_COLOR, out2 => "DB2401_DBB_DEFINE".PART_STATUS.DBB_1007)
   END_RUNG
   RUNG wire#w3
      Contact( "DB8000_PART_STATUS".UNIT_01.FIXTURE_2.PART_A.STATUS.CELL_STATUS.INSPECTION_DONE )
      Move(in := 17, out1 => "DB8000_PART_STATUS".UNIT_01.FIXTURE_2.PART_A.STATUS.PART_CELL_STATUS_COLOR, out2 => "DB2401_DBB_DEFINE".PART_STATUS.DBB_1007)
   END_RUNG
   RUNG wire#w3
      Contact( "DB8000_PART_STATUS".UNIT_01.FIXTURE_2.PART_A.STATUS.MASTER_PART )
      Move(in := 99, out1 => "DB8000_PART_STATUS".UNIT_01.FIXTURE_2.PART_A.STATUS.PART_CELL_STATUS_COLOR, out2 => "DB2401_DBB_DEFINE".PART_STATUS.DBB_1007)
   END_RUNG
   // the same network as SCL:
   // ENO of a box is taken as its EN; it also drops when the box reports an error
   IF "M_ONE" AND NOT "DB8000_PART_STATUS".UNIT_01.FIXTURE_2.PART_A.STATUS.PRESENT THEN
       "DB2401_DBB_DEFINE".PART_STATUS.DBB_1006 := 0;
       "DB2401_DBB_DEFINE".PART_STATUS.DBB_1007 := 0;
       "DB8000_PART_STATUS".UNIT_01.FIXTURE_2.PART_A.STATUS.PART_MAIN_STATUS_COLOR := 0;
       "DB8000_PART_STATUS".UNIT_01.FIXTURE_2.PART_A.STATUS.PART_CELL_STATUS_COLOR := 0;
   END_IF;
   #_w1 := "M_ONE" AND "DB8000_PART_STATUS".UNIT_01.FIXTURE_2.PART_A.STATUS.PRESENT;
   IF #_w1 AND NOT "DB8000_PART_STATUS".UNIT_01.FIXTURE_2.PART_A.STATUS.PART_REJECTED AND NOT "DB8000_PART_STATUS".UNIT_01.FIXTURE_2.PART_A.STATUS.QUALITY_PART THEN
       "DB8000_PART_STATUS".UNIT_01.FIXTURE_2.PART_A.STATUS.PART_MAIN_STATUS_COLOR := 1;
       "DB2401_DBB_DEFINE".PART_STATUS.DBB_1006 := 1;
   END_IF;
   IF #_w1 AND "DB8000_PART_STATUS".UNIT_01.FIXTURE_2.PART_A.STATUS.PART_REJECTED THEN
       "DB8000_PART_STATUS".UNIT_01.FIXTURE_2.PART_A.STATUS.PART_MAIN_STATUS_COLOR := 2;
       "DB2401_DBB_DEFINE".PART_STATUS.DBB_1006 := 2;
   END_IF;
   IF #_w1 AND "DB8000_PART_STATUS".UNIT_01.FIXTURE_2.PART_A.STATUS.QUALITY_PART AND NOT "DB8000_PART_STATUS".UNIT_01.FIXTURE_2.PART_A.STATUS.PART_REJECTED THEN
       "DB8000_PART_STATUS".UNIT_01.FIXTURE_2.PART_A.STATUS.PART_MAIN_STATUS_COLOR := 3;
       "DB2401_DBB_DEFINE".PART_STATUS.DBB_1006 := 3;
   END_IF;
   #_w2 := "M_ONE" AND "DB8000_PART_STATUS".UNIT_01.FIXTURE_2.PART_A.STATUS.PRESENT;
   IF #_w2 AND "DB8000_PART_STATUS".UNIT_01.FIXTURE_2.PART_A.STATUS.CELL_STATUS.NEW_IN_TRANSIT THEN
       "DB8000_PART_STATUS".UNIT_01.FIXTURE_2.PART_A.STATUS.PART_CELL_STATUS_COLOR := 1;
       "DB2401_DBB_DEFINE".PART_STATUS.DBB_1007 := 1;
   END_IF;
   IF #_w2 AND "DB8000_PART_STATUS".UNIT_01.FIXTURE_2.PART_A.STATUS.UNIT_01_STATUS.FACE_N_STATION_3_DONE THEN
       "DB8000_PART_STATUS".UNIT_01.FIXTURE_2.PART_A.STATUS.PART_CELL_STATUS_COLOR := 2;
       "DB2401_DBB_DEFINE".PART_STATUS.DBB_1007 := 2;
   END_IF;
   IF #_w2 AND "DB8000_PART_STATUS".UNIT_01.FIXTURE_2.PART_A.STATUS.UNIT_01_STATUS.FACE_N_STATION_4_DONE THEN
       "DB8000_PART_STATUS".UNIT_01.FIXTURE_2.PART_A.STATUS.PART_CELL_STATUS_COLOR := 3;
       "DB2401_DBB_DEFINE".PART_STATUS.DBB_1007 := 3;
   END_IF;
   IF #_w2 AND "DB8000_PART_STATUS".UNIT_01.FIXTURE_2.PART_A.STATUS.CELL_STATUS.U01_ONE_FACE_DONE_ROTATED THEN
       "DB8000_PART_STATUS".UNIT_01.FIXTURE_2.PART_A.STATUS.PART_CELL_STATUS_COLOR := 4;
       "DB2401_DBB_DEFINE".PART_STATUS.DBB_1007 := 4;
   END_IF;
   IF #_w2 AND "DB8000_PART_STATUS".UNIT_01.FIXTURE_2.PART_A.STATUS.UNIT_01_STATUS.FACE_R_STATION_3_DONE THEN
       "DB8000_PART_STATUS".UNIT_01.FIXTURE_2.PART_A.STATUS.PART_CELL_STATUS_COLOR := 5;
       "DB2401_DBB_DEFINE".PART_STATUS.DBB_1007 := 5;
   END_IF;
   IF #_w2 AND "DB8000_PART_STATUS".UNIT_01.FIXTURE_2.PART_A.STATUS.UNIT_01_STATUS.FACE_R_STATION_4_DONE THEN
       "DB8000_PART_STATUS".UNIT_01.FIXTURE_2.PART_A.STATUS.PART_CELL_STATUS_COLOR := 6;
       "DB2401_DBB_DEFINE".PART_STATUS.DBB_1007 := 6;
   END_IF;
   IF #_w2 AND "DB8000_PART_STATUS".UNIT_01.FIXTURE_2.PART_A.STATUS.CELL_STATUS.U01_DONE_IN_TRANSIT THEN
       "DB8000_PART_STATUS".UNIT_01.FIXTURE_2.PART_A.STATUS.PART_CELL_STATUS_COLOR := 7;
       "DB2401_DBB_DEFINE".PART_STATUS.DBB_1007 := 7;
   END_IF;
   IF #_w2 AND "DB8000_PART_STATUS".UNIT_01.FIXTURE_2.PART_A.STATUS.UNIT_02_STATUS.FACE_N_STATION_2_DONE THEN
       "DB8000_PART_STATUS".UNIT_01.FIXTURE_2.PART_A.STATUS.PART_CELL_STATUS_COLOR := 8;
       "DB2401_DBB_DEFINE".PART_STATUS.DBB_1007 := 8;
   END_IF;
   IF #_w2 AND "DB8000_PART_STATUS".UNIT_01.FIXTURE_2.PART_A.STATUS.UNIT_02_STATUS.FACE_N_STATION_3_DONE THEN
       "DB8000_PART_STATUS".UNIT_01.FIXTURE_2.PART_A.STATUS.PART_CELL_STATUS_COLOR := 9;
       "DB2401_DBB_DEFINE".PART_STATUS.DBB_1007 := 9;
   END_IF;
   IF #_w2 AND "DB8000_PART_STATUS".UNIT_01.FIXTURE_2.PART_A.STATUS.UNIT_02_STATUS.FACE_N_STATION_4_DONE THEN
       "DB8000_PART_STATUS".UNIT_01.FIXTURE_2.PART_A.STATUS.PART_CELL_STATUS_COLOR := 10;
       "DB2401_DBB_DEFINE".PART_STATUS.DBB_1007 := 10;
   END_IF;
   IF #_w2 AND "DB8000_PART_STATUS".UNIT_01.FIXTURE_2.PART_A.STATUS.CELL_STATUS.U02_ONE_FACE_DONE_ROTATED THEN
       "DB8000_PART_STATUS".UNIT_01.FIXTURE_2.PART_A.STATUS.PART_CELL_STATUS_COLOR := 11;
       "DB2401_DBB_DEFINE".PART_STATUS.DBB_1007 := 11;
   END_IF;
   IF #_w2 AND "DB8000_PART_STATUS".UNIT_01.FIXTURE_2.PART_A.STATUS.UNIT_02_STATUS.FACE_R_STATION_2_DONE THEN
       "DB8000_PART_STATUS".UNIT_01.FIXTURE_2.PART_A.STATUS.PART_CELL_STATUS_COLOR := 12;
       "DB2401_DBB_DEFINE".PART_STATUS.DBB_1007 := 12;
   END_IF;
   IF #_w2 AND "DB8000_PART_STATUS".UNIT_01.FIXTURE_2.PART_A.STATUS.UNIT_02_STATUS.FACE_R_STATION_3_DONE THEN
       "DB8000_PART_STATUS".UNIT_01.FIXTURE_2.PART_A.STATUS.PART_CELL_STATUS_COLOR := 13;
       "DB2401_DBB_DEFINE".PART_STATUS.DBB_1007 := 13;
   END_IF;
   IF #_w2 AND "DB8000_PART_STATUS".UNIT_01.FIXTURE_2.PART_A.STATUS.UNIT_02_STATUS.FACE_R_STATION_4_DONE THEN
       "DB8000_PART_STATUS".UNIT_01.FIXTURE_2.PART_A.STATUS.PART_CELL_STATUS_COLOR := 14;
       "DB2401_DBB_DEFINE".PART_STATUS.DBB_1007 := 14;
   END_IF;
   IF #_w2 AND "DB8000_PART_STATUS".UNIT_01.FIXTURE_2.PART_A.STATUS.CELL_STATUS.U02_DONE_IN_TRANSIT THEN
       "DB8000_PART_STATUS".UNIT_01.FIXTURE_2.PART_A.STATUS.PART_CELL_STATUS_COLOR := 15;
       "DB2401_DBB_DEFINE".PART_STATUS.DBB_1007 := 15;
   END_IF;
   IF #_w2 AND "DB8000_PART_STATUS".UNIT_01.FIXTURE_2.PART_A.STATUS.CELL_STATUS.COOLING_DONE THEN
       "DB8000_PART_STATUS".UNIT_01.FIXTURE_2.PART_A.STATUS.PART_CELL_STATUS_COLOR := 16;
       "DB2401_DBB_DEFINE".PART_STATUS.DBB_1007 := 16;
   END_IF;
   IF #_w2 AND "DB8000_PART_STATUS".UNIT_01.FIXTURE_2.PART_A.STATUS.CELL_STATUS.INSPECTION_DONE THEN
       "DB8000_PART_STATUS".UNIT_01.FIXTURE_2.PART_A.STATUS.PART_CELL_STATUS_COLOR := 17;
       "DB2401_DBB_DEFINE".PART_STATUS.DBB_1007 := 17;
   END_IF;
   IF #_w2 AND "DB8000_PART_STATUS".UNIT_01.FIXTURE_2.PART_A.STATUS.MASTER_PART THEN
       "DB8000_PART_STATUS".UNIT_01.FIXTURE_2.PART_A.STATUS.PART_CELL_STATUS_COLOR := 99;
       "DB2401_DBB_DEFINE".PART_STATUS.DBB_1007 := 99;
   END_IF;
END_REGION

REGION Network 22: PART A FIXTURE 3 COLOR STATUS
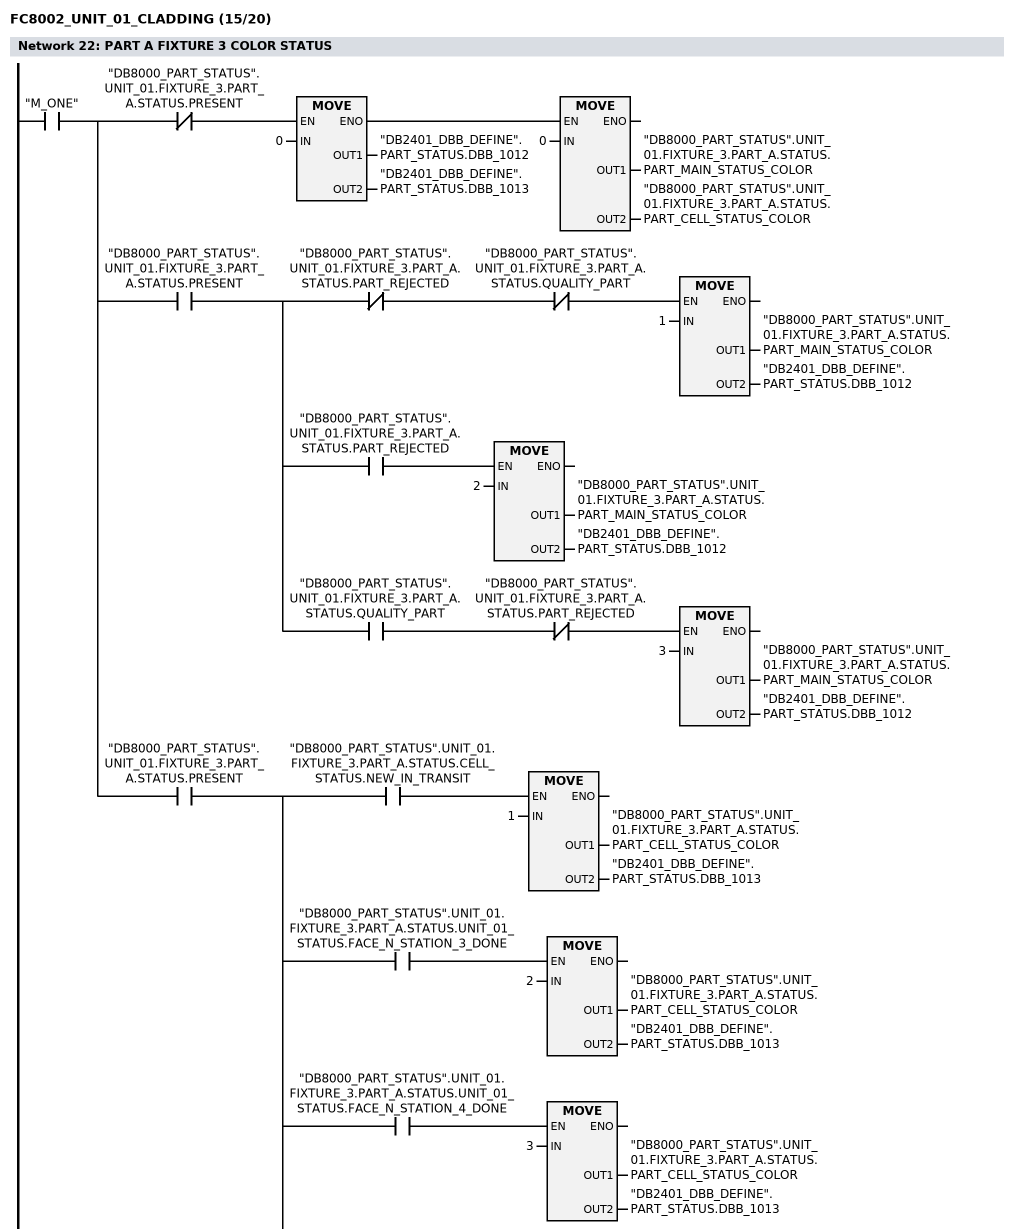
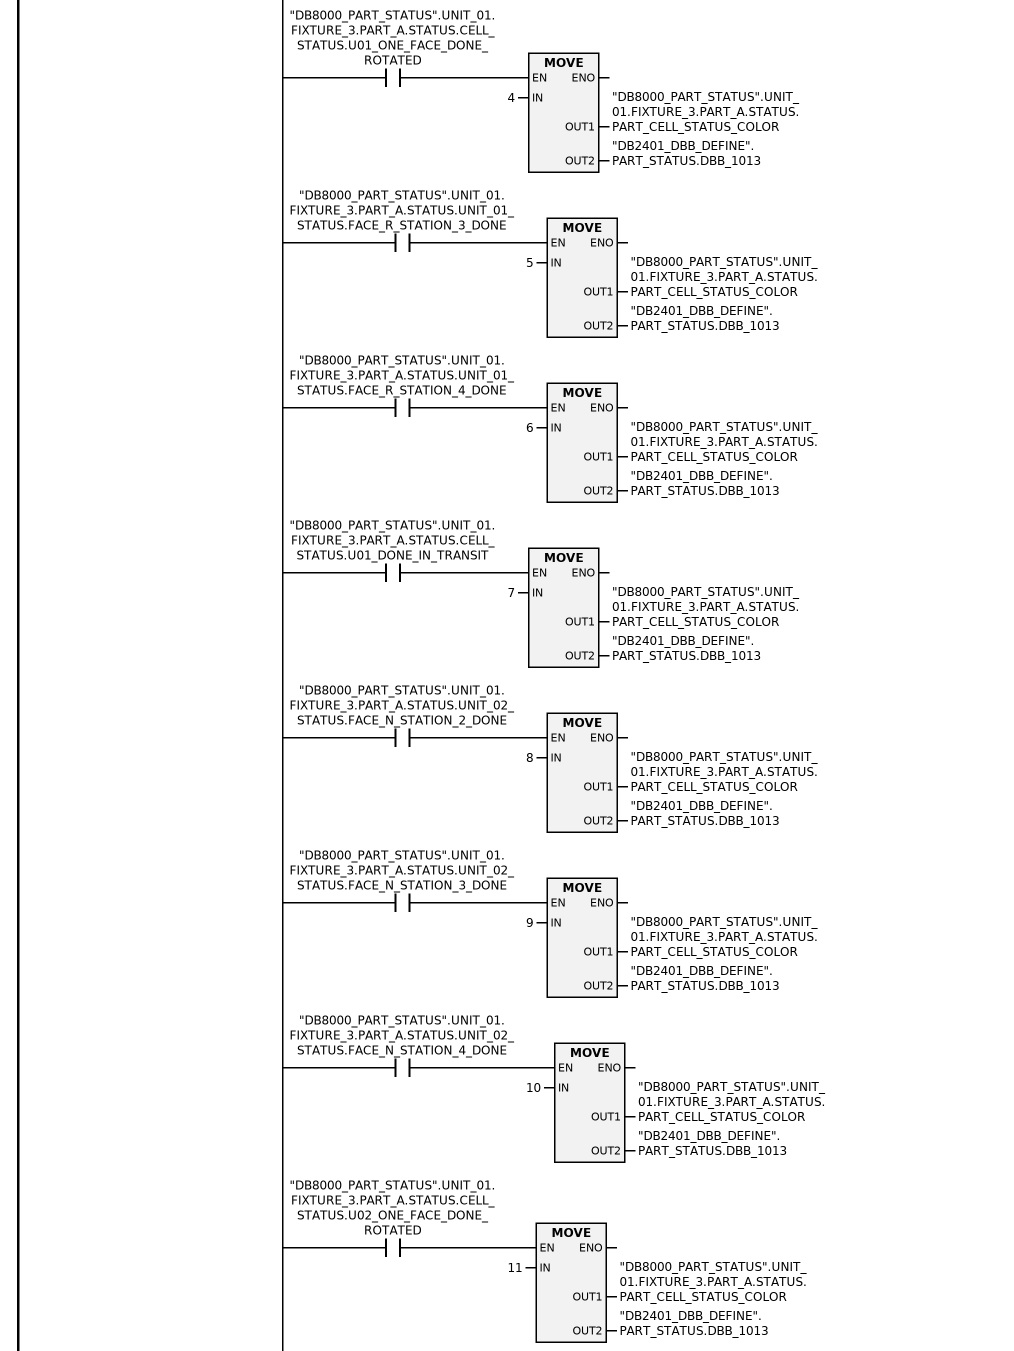
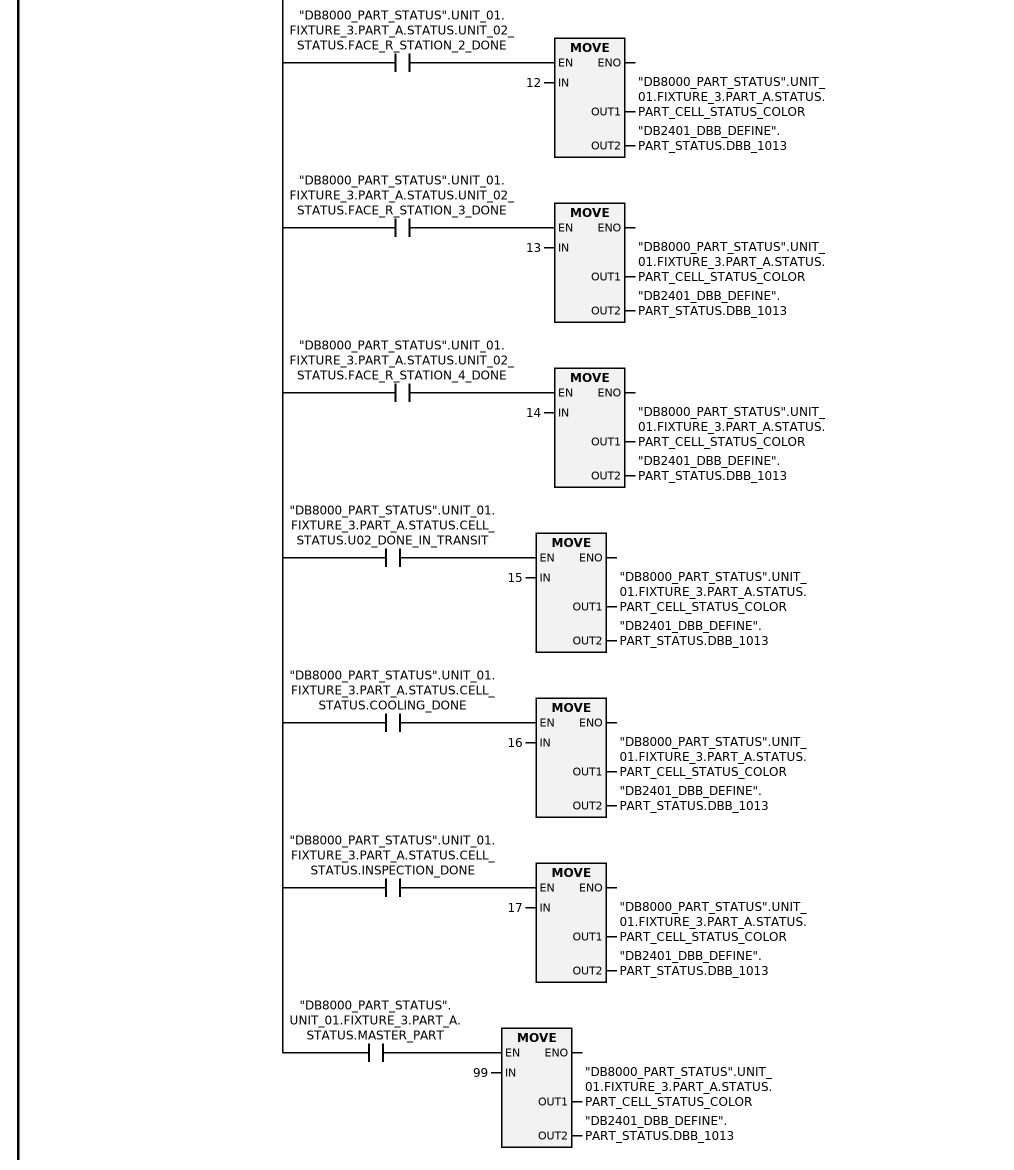
   RUNG wire#powerrail
      Contact( "M_ONE" )
      wire#w1
      I_Contact( "DB8000_PART_STATUS".UNIT_01.FIXTURE_3.PART_A.STATUS.PRESENT )
      { S7_GenerateENO := "TRUE" } Move(in := 0, out1 => "DB2401_DBB_DEFINE".PART_STATUS.DBB_1012, out2 => "DB2401_DBB_DEFINE".PART_STATUS.DBB_1013)
      { S7_GenerateENO := "TRUE" } Move(in := 0, out1 => "DB8000_PART_STATUS".UNIT_01.FIXTURE_3.PART_A.STATUS.PART_MAIN_STATUS_COLOR, out2 => "DB8000_PART_STATUS".UNIT_01.FIXTURE_3.PART_A.STATUS.PART_CELL_STATUS_COLOR)
   END_RUNG
   RUNG wire#w1
      Contact( "DB8000_PART_STATUS".UNIT_01.FIXTURE_3.PART_A.STATUS.PRESENT )
      wire#w2
      I_Contact( "DB8000_PART_STATUS".UNIT_01.FIXTURE_3.PART_A.STATUS.PART_REJECTED )
      I_Contact( "DB8000_PART_STATUS".UNIT_01.FIXTURE_3.PART_A.STATUS.QUALITY_PART )
      { S7_GenerateENO := "TRUE" } Move(in := 1, out1 => "DB8000_PART_STATUS".UNIT_01.FIXTURE_3.PART_A.STATUS.PART_MAIN_STATUS_COLOR, out2 => "DB2401_DBB_DEFINE".PART_STATUS.DBB_1012)
   END_RUNG
   RUNG wire#w2
      Contact( "DB8000_PART_STATUS".UNIT_01.FIXTURE_3.PART_A.STATUS.PART_REJECTED )
      { S7_GenerateENO := "TRUE" } Move(in := 2, out1 => "DB8000_PART_STATUS".UNIT_01.FIXTURE_3.PART_A.STATUS.PART_MAIN_STATUS_COLOR, out2 => "DB2401_DBB_DEFINE".PART_STATUS.DBB_1012)
   END_RUNG
   RUNG wire#w2
      Contact( "DB8000_PART_STATUS".UNIT_01.FIXTURE_3.PART_A.STATUS.QUALITY_PART )
      I_Contact( "DB8000_PART_STATUS".UNIT_01.FIXTURE_3.PART_A.STATUS.PART_REJECTED )
      { S7_GenerateENO := "TRUE" } Move(in := 3, out1 => "DB8000_PART_STATUS".UNIT_01.FIXTURE_3.PART_A.STATUS.PART_MAIN_STATUS_COLOR, out2 => "DB2401_DBB_DEFINE".PART_STATUS.DBB_1012)
   END_RUNG
   RUNG wire#w1
      Contact( "DB8000_PART_STATUS".UNIT_01.FIXTURE_3.PART_A.STATUS.PRESENT )
      wire#w3
      Contact( "DB8000_PART_STATUS".UNIT_01.FIXTURE_3.PART_A.STATUS.CELL_STATUS.NEW_IN_TRANSIT )
      { S7_GenerateENO := "TRUE" } Move(in := 1, out1 => "DB8000_PART_STATUS".UNIT_01.FIXTURE_3.PART_A.STATUS.PART_CELL_STATUS_COLOR, out2 => "DB2401_DBB_DEFINE".PART_STATUS.DBB_1013)
   END_RUNG
   RUNG wire#w3
      Contact( "DB8000_PART_STATUS".UNIT_01.FIXTURE_3.PART_A.STATUS.UNIT_01_STATUS.FACE_N_STATION_3_DONE )
      { S7_GenerateENO := "TRUE" } Move(in := 2, out1 => "DB8000_PART_STATUS".UNIT_01.FIXTURE_3.PART_A.STATUS.PART_CELL_STATUS_COLOR, out2 => "DB2401_DBB_DEFINE".PART_STATUS.DBB_1013)
   END_RUNG
   RUNG wire#w3
      Contact( "DB8000_PART_STATUS".UNIT_01.FIXTURE_3.PART_A.STATUS.UNIT_01_STATUS.FACE_N_STATION_4_DONE )
      { S7_GenerateENO := "TRUE" } Move(in := 3, out1 => "DB8000_PART_STATUS".UNIT_01.FIXTURE_3.PART_A.STATUS.PART_CELL_STATUS_COLOR, out2 => "DB2401_DBB_DEFINE".PART_STATUS.DBB_1013)
   END_RUNG
   RUNG wire#w3
      Contact( "DB8000_PART_STATUS".UNIT_01.FIXTURE_3.PART_A.STATUS.CELL_STATUS.U01_ONE_FACE_DONE_ROTATED )
      { S7_GenerateENO := "TRUE" } Move(in := 4, out1 => "DB8000_PART_STATUS".UNIT_01.FIXTURE_3.PART_A.STATUS.PART_CELL_STATUS_COLOR, out2 => "DB2401_DBB_DEFINE".PART_STATUS.DBB_1013)
   END_RUNG
   RUNG wire#w3
      Contact( "DB8000_PART_STATUS".UNIT_01.FIXTURE_3.PART_A.STATUS.UNIT_01_STATUS.FACE_R_STATION_3_DONE )
      { S7_GenerateENO := "TRUE" } Move(in := 5, out1 => "DB8000_PART_STATUS".UNIT_01.FIXTURE_3.PART_A.STATUS.PART_CELL_STATUS_COLOR, out2 => "DB2401_DBB_DEFINE".PART_STATUS.DBB_1013)
   END_RUNG
   RUNG wire#w3
      Contact( "DB8000_PART_STATUS".UNIT_01.FIXTURE_3.PART_A.STATUS.UNIT_01_STATUS.FACE_R_STATION_4_DONE )
      { S7_GenerateENO := "TRUE" } Move(in := 6, out1 => "DB8000_PART_STATUS".UNIT_01.FIXTURE_3.PART_A.STATUS.PART_CELL_STATUS_COLOR, out2 => "DB2401_DBB_DEFINE".PART_STATUS.DBB_1013)
   END_RUNG
   RUNG wire#w3
      Contact( "DB8000_PART_STATUS".UNIT_01.FIXTURE_3.PART_A.STATUS.CELL_STATUS.U01_DONE_IN_TRANSIT )
      { S7_GenerateENO := "TRUE" } Move(in := 7, out1 => "DB8000_PART_STATUS".UNIT_01.FIXTURE_3.PART_A.STATUS.PART_CELL_STATUS_COLOR, out2 => "DB2401_DBB_DEFINE".PART_STATUS.DBB_1013)
   END_RUNG
   RUNG wire#w3
      Contact( "DB8000_PART_STATUS".UNIT_01.FIXTURE_3.PART_A.STATUS.UNIT_02_STATUS.FACE_N_STATION_2_DONE )
      { S7_GenerateENO := "TRUE" } Move(in := 8, out1 => "DB8000_PART_STATUS".UNIT_01.FIXTURE_3.PART_A.STATUS.PART_CELL_STATUS_COLOR, out2 => "DB2401_DBB_DEFINE".PART_STATUS.DBB_1013)
   END_RUNG
   RUNG wire#w3
      Contact( "DB8000_PART_STATUS".UNIT_01.FIXTURE_3.PART_A.STATUS.UNIT_02_STATUS.FACE_N_STATION_3_DONE )
      { S7_GenerateENO := "TRUE" } Move(in := 9, out1 => "DB8000_PART_STATUS".UNIT_01.FIXTURE_3.PART_A.STATUS.PART_CELL_STATUS_COLOR, out2 => "DB2401_DBB_DEFINE".PART_STATUS.DBB_1013)
   END_RUNG
   RUNG wire#w3
      Contact( "DB8000_PART_STATUS".UNIT_01.FIXTURE_3.PART_A.STATUS.UNIT_02_STATUS.FACE_N_STATION_4_DONE )
      { S7_GenerateENO := "TRUE" } Move(in := 10, out1 => "DB8000_PART_STATUS".UNIT_01.FIXTURE_3.PART_A.STATUS.PART_CELL_STATUS_COLOR, out2 => "DB2401_DBB_DEFINE".PART_STATUS.DBB_1013)
   END_RUNG
   RUNG wire#w3
      Contact( "DB8000_PART_STATUS".UNIT_01.FIXTURE_3.PART_A.STATUS.CELL_STATUS.U02_ONE_FACE_DONE_ROTATED )
      { S7_GenerateENO := "TRUE" } Move(in := 11, out1 => "DB8000_PART_STATUS".UNIT_01.FIXTURE_3.PART_A.STATUS.PART_CELL_STATUS_COLOR, out2 => "DB2401_DBB_DEFINE".PART_STATUS.DBB_1013)
   END_RUNG
   RUNG wire#w3
      Contact( "DB8000_PART_STATUS".UNIT_01.FIXTURE_3.PART_A.STATUS.UNIT_02_STATUS.FACE_R_STATION_2_DONE )
      { S7_GenerateENO := "TRUE" } Move(in := 12, out1 => "DB8000_PART_STATUS".UNIT_01.FIXTURE_3.PART_A.STATUS.PART_CELL_STATUS_COLOR, out2 => "DB2401_DBB_DEFINE".PART_STATUS.DBB_1013)
   END_RUNG
   RUNG wire#w3
      Contact( "DB8000_PART_STATUS".UNIT_01.FIXTURE_3.PART_A.STATUS.UNIT_02_STATUS.FACE_R_STATION_3_DONE )
      Move(in := 13, out1 => "DB8000_PART_STATUS".UNIT_01.FIXTURE_3.PART_A.STATUS.PART_CELL_STATUS_COLOR, out2 => "DB2401_DBB_DEFINE".PART_STATUS.DBB_1013)
   END_RUNG
   RUNG wire#w3
      Contact( "DB8000_PART_STATUS".UNIT_01.FIXTURE_3.PART_A.STATUS.UNIT_02_STATUS.FACE_R_STATION_4_DONE )
      Move(in := 14, out1 => "DB8000_PART_STATUS".UNIT_01.FIXTURE_3.PART_A.STATUS.PART_CELL_STATUS_COLOR, out2 => "DB2401_DBB_DEFINE".PART_STATUS.DBB_1013)
   END_RUNG
   RUNG wire#w3
      Contact( "DB8000_PART_STATUS".UNIT_01.FIXTURE_3.PART_A.STATUS.CELL_STATUS.U02_DONE_IN_TRANSIT )
      Move(in := 15, out1 => "DB8000_PART_STATUS".UNIT_01.FIXTURE_3.PART_A.STATUS.PART_CELL_STATUS_COLOR, out2 => "DB2401_DBB_DEFINE".PART_STATUS.DBB_1013)
   END_RUNG
   RUNG wire#w3
      Contact( "DB8000_PART_STATUS".UNIT_01.FIXTURE_3.PART_A.STATUS.CELL_STATUS.COOLING_DONE )
      Move(in := 16, out1 => "DB8000_PART_STATUS".UNIT_01.FIXTURE_3.PART_A.STATUS.PART_CELL_STATUS_COLOR, out2 => "DB2401_DBB_DEFINE".PART_STATUS.DBB_1013)
   END_RUNG
   RUNG wire#w3
      Contact( "DB8000_PART_STATUS".UNIT_01.FIXTURE_3.PART_A.STATUS.CELL_STATUS.INSPECTION_DONE )
      Move(in := 17, out1 => "DB8000_PART_STATUS".UNIT_01.FIXTURE_3.PART_A.STATUS.PART_CELL_STATUS_COLOR, out2 => "DB2401_DBB_DEFINE".PART_STATUS.DBB_1013)
   END_RUNG
   RUNG wire#w3
      Contact( "DB8000_PART_STATUS".UNIT_01.FIXTURE_3.PART_A.STATUS.MASTER_PART )
      Move(in := 99, out1 => "DB8000_PART_STATUS".UNIT_01.FIXTURE_3.PART_A.STATUS.PART_CELL_STATUS_COLOR, out2 => "DB2401_DBB_DEFINE".PART_STATUS.DBB_1013)
   END_RUNG
   // the same network as SCL:
   // ENO of a box is taken as its EN; it also drops when the box reports an error
   IF "M_ONE" AND NOT "DB8000_PART_STATUS".UNIT_01.FIXTURE_3.PART_A.STATUS.PRESENT THEN
       "DB2401_DBB_DEFINE".PART_STATUS.DBB_1012 := 0;
       "DB2401_DBB_DEFINE".PART_STATUS.DBB_1013 := 0;
       "DB8000_PART_STATUS".UNIT_01.FIXTURE_3.PART_A.STATUS.PART_MAIN_STATUS_COLOR := 0;
       "DB8000_PART_STATUS".UNIT_01.FIXTURE_3.PART_A.STATUS.PART_CELL_STATUS_COLOR := 0;
   END_IF;
   #_w1 := "M_ONE" AND "DB8000_PART_STATUS".UNIT_01.FIXTURE_3.PART_A.STATUS.PRESENT;
   IF #_w1 AND NOT "DB8000_PART_STATUS".UNIT_01.FIXTURE_3.PART_A.STATUS.PART_REJECTED AND NOT "DB8000_PART_STATUS".UNIT_01.FIXTURE_3.PART_A.STATUS.QUALITY_PART THEN
       "DB8000_PART_STATUS".UNIT_01.FIXTURE_3.PART_A.STATUS.PART_MAIN_STATUS_COLOR := 1;
       "DB2401_DBB_DEFINE".PART_STATUS.DBB_1012 := 1;
   END_IF;
   IF #_w1 AND "DB8000_PART_STATUS".UNIT_01.FIXTURE_3.PART_A.STATUS.PART_REJECTED THEN
       "DB8000_PART_STATUS".UNIT_01.FIXTURE_3.PART_A.STATUS.PART_MAIN_STATUS_COLOR := 2;
       "DB2401_DBB_DEFINE".PART_STATUS.DBB_1012 := 2;
   END_IF;
   IF #_w1 AND "DB8000_PART_STATUS".UNIT_01.FIXTURE_3.PART_A.STATUS.QUALITY_PART AND NOT "DB8000_PART_STATUS".UNIT_01.FIXTURE_3.PART_A.STATUS.PART_REJECTED THEN
       "DB8000_PART_STATUS".UNIT_01.FIXTURE_3.PART_A.STATUS.PART_MAIN_STATUS_COLOR := 3;
       "DB2401_DBB_DEFINE".PART_STATUS.DBB_1012 := 3;
   END_IF;
   #_w2 := "M_ONE" AND "DB8000_PART_STATUS".UNIT_01.FIXTURE_3.PART_A.STATUS.PRESENT;
   IF #_w2 AND "DB8000_PART_STATUS".UNIT_01.FIXTURE_3.PART_A.STATUS.CELL_STATUS.NEW_IN_TRANSIT THEN
       "DB8000_PART_STATUS".UNIT_01.FIXTURE_3.PART_A.STATUS.PART_CELL_STATUS_COLOR := 1;
       "DB2401_DBB_DEFINE".PART_STATUS.DBB_1013 := 1;
   END_IF;
   IF #_w2 AND "DB8000_PART_STATUS".UNIT_01.FIXTURE_3.PART_A.STATUS.UNIT_01_STATUS.FACE_N_STATION_3_DONE THEN
       "DB8000_PART_STATUS".UNIT_01.FIXTURE_3.PART_A.STATUS.PART_CELL_STATUS_COLOR := 2;
       "DB2401_DBB_DEFINE".PART_STATUS.DBB_1013 := 2;
   END_IF;
   IF #_w2 AND "DB8000_PART_STATUS".UNIT_01.FIXTURE_3.PART_A.STATUS.UNIT_01_STATUS.FACE_N_STATION_4_DONE THEN
       "DB8000_PART_STATUS".UNIT_01.FIXTURE_3.PART_A.STATUS.PART_CELL_STATUS_COLOR := 3;
       "DB2401_DBB_DEFINE".PART_STATUS.DBB_1013 := 3;
   END_IF;
   IF #_w2 AND "DB8000_PART_STATUS".UNIT_01.FIXTURE_3.PART_A.STATUS.CELL_STATUS.U01_ONE_FACE_DONE_ROTATED THEN
       "DB8000_PART_STATUS".UNIT_01.FIXTURE_3.PART_A.STATUS.PART_CELL_STATUS_COLOR := 4;
       "DB2401_DBB_DEFINE".PART_STATUS.DBB_1013 := 4;
   END_IF;
   IF #_w2 AND "DB8000_PART_STATUS".UNIT_01.FIXTURE_3.PART_A.STATUS.UNIT_01_STATUS.FACE_R_STATION_3_DONE THEN
       "DB8000_PART_STATUS".UNIT_01.FIXTURE_3.PART_A.STATUS.PART_CELL_STATUS_COLOR := 5;
       "DB2401_DBB_DEFINE".PART_STATUS.DBB_1013 := 5;
   END_IF;
   IF #_w2 AND "DB8000_PART_STATUS".UNIT_01.FIXTURE_3.PART_A.STATUS.UNIT_01_STATUS.FACE_R_STATION_4_DONE THEN
       "DB8000_PART_STATUS".UNIT_01.FIXTURE_3.PART_A.STATUS.PART_CELL_STATUS_COLOR := 6;
       "DB2401_DBB_DEFINE".PART_STATUS.DBB_1013 := 6;
   END_IF;
   IF #_w2 AND "DB8000_PART_STATUS".UNIT_01.FIXTURE_3.PART_A.STATUS.CELL_STATUS.U01_DONE_IN_TRANSIT THEN
       "DB8000_PART_STATUS".UNIT_01.FIXTURE_3.PART_A.STATUS.PART_CELL_STATUS_COLOR := 7;
       "DB2401_DBB_DEFINE".PART_STATUS.DBB_1013 := 7;
   END_IF;
   IF #_w2 AND "DB8000_PART_STATUS".UNIT_01.FIXTURE_3.PART_A.STATUS.UNIT_02_STATUS.FACE_N_STATION_2_DONE THEN
       "DB8000_PART_STATUS".UNIT_01.FIXTURE_3.PART_A.STATUS.PART_CELL_STATUS_COLOR := 8;
       "DB2401_DBB_DEFINE".PART_STATUS.DBB_1013 := 8;
   END_IF;
   IF #_w2 AND "DB8000_PART_STATUS".UNIT_01.FIXTURE_3.PART_A.STATUS.UNIT_02_STATUS.FACE_N_STATION_3_DONE THEN
       "DB8000_PART_STATUS".UNIT_01.FIXTURE_3.PART_A.STATUS.PART_CELL_STATUS_COLOR := 9;
       "DB2401_DBB_DEFINE".PART_STATUS.DBB_1013 := 9;
   END_IF;
   IF #_w2 AND "DB8000_PART_STATUS".UNIT_01.FIXTURE_3.PART_A.STATUS.UNIT_02_STATUS.FACE_N_STATION_4_DONE THEN
       "DB8000_PART_STATUS".UNIT_01.FIXTURE_3.PART_A.STATUS.PART_CELL_STATUS_COLOR := 10;
       "DB2401_DBB_DEFINE".PART_STATUS.DBB_1013 := 10;
   END_IF;
   IF #_w2 AND "DB8000_PART_STATUS".UNIT_01.FIXTURE_3.PART_A.STATUS.CELL_STATUS.U02_ONE_FACE_DONE_ROTATED THEN
       "DB8000_PART_STATUS".UNIT_01.FIXTURE_3.PART_A.STATUS.PART_CELL_STATUS_COLOR := 11;
       "DB2401_DBB_DEFINE".PART_STATUS.DBB_1013 := 11;
   END_IF;
   IF #_w2 AND "DB8000_PART_STATUS".UNIT_01.FIXTURE_3.PART_A.STATUS.UNIT_02_STATUS.FACE_R_STATION_2_DONE THEN
       "DB8000_PART_STATUS".UNIT_01.FIXTURE_3.PART_A.STATUS.PART_CELL_STATUS_COLOR := 12;
       "DB2401_DBB_DEFINE".PART_STATUS.DBB_1013 := 12;
   END_IF;
   IF #_w2 AND "DB8000_PART_STATUS".UNIT_01.FIXTURE_3.PART_A.STATUS.UNIT_02_STATUS.FACE_R_STATION_3_DONE THEN
       "DB8000_PART_STATUS".UNIT_01.FIXTURE_3.PART_A.STATUS.PART_CELL_STATUS_COLOR := 13;
       "DB2401_DBB_DEFINE".PART_STATUS.DBB_1013 := 13;
   END_IF;
   IF #_w2 AND "DB8000_PART_STATUS".UNIT_01.FIXTURE_3.PART_A.STATUS.UNIT_02_STATUS.FACE_R_STATION_4_DONE THEN
       "DB8000_PART_STATUS".UNIT_01.FIXTURE_3.PART_A.STATUS.PART_CELL_STATUS_COLOR := 14;
       "DB2401_DBB_DEFINE".PART_STATUS.DBB_1013 := 14;
   END_IF;
   IF #_w2 AND "DB8000_PART_STATUS".UNIT_01.FIXTURE_3.PART_A.STATUS.CELL_STATUS.U02_DONE_IN_TRANSIT THEN
       "DB8000_PART_STATUS".UNIT_01.FIXTURE_3.PART_A.STATUS.PART_CELL_STATUS_COLOR := 15;
       "DB2401_DBB_DEFINE".PART_STATUS.DBB_1013 := 15;
   END_IF;
   IF #_w2 AND "DB8000_PART_STATUS".UNIT_01.FIXTURE_3.PART_A.STATUS.CELL_STATUS.COOLING_DONE THEN
       "DB8000_PART_STATUS".UNIT_01.FIXTURE_3.PART_A.STATUS.PART_CELL_STATUS_COLOR := 16;
       "DB2401_DBB_DEFINE".PART_STATUS.DBB_1013 := 16;
   END_IF;
   IF #_w2 AND "DB8000_PART_STATUS".UNIT_01.FIXTURE_3.PART_A.STATUS.CELL_STATUS.INSPECTION_DONE THEN
       "DB8000_PART_STATUS".UNIT_01.FIXTURE_3.PART_A.STATUS.PART_CELL_STATUS_COLOR := 17;
       "DB2401_DBB_DEFINE".PART_STATUS.DBB_1013 := 17;
   END_IF;
   IF #_w2 AND "DB8000_PART_STATUS".UNIT_01.FIXTURE_3.PART_A.STATUS.MASTER_PART THEN
       "DB8000_PART_STATUS".UNIT_01.FIXTURE_3.PART_A.STATUS.PART_CELL_STATUS_COLOR := 99;
       "DB2401_DBB_DEFINE".PART_STATUS.DBB_1013 := 99;
   END_IF;
END_REGION

REGION Network 23: PART A FIXTURE 4 COLOR STATUS
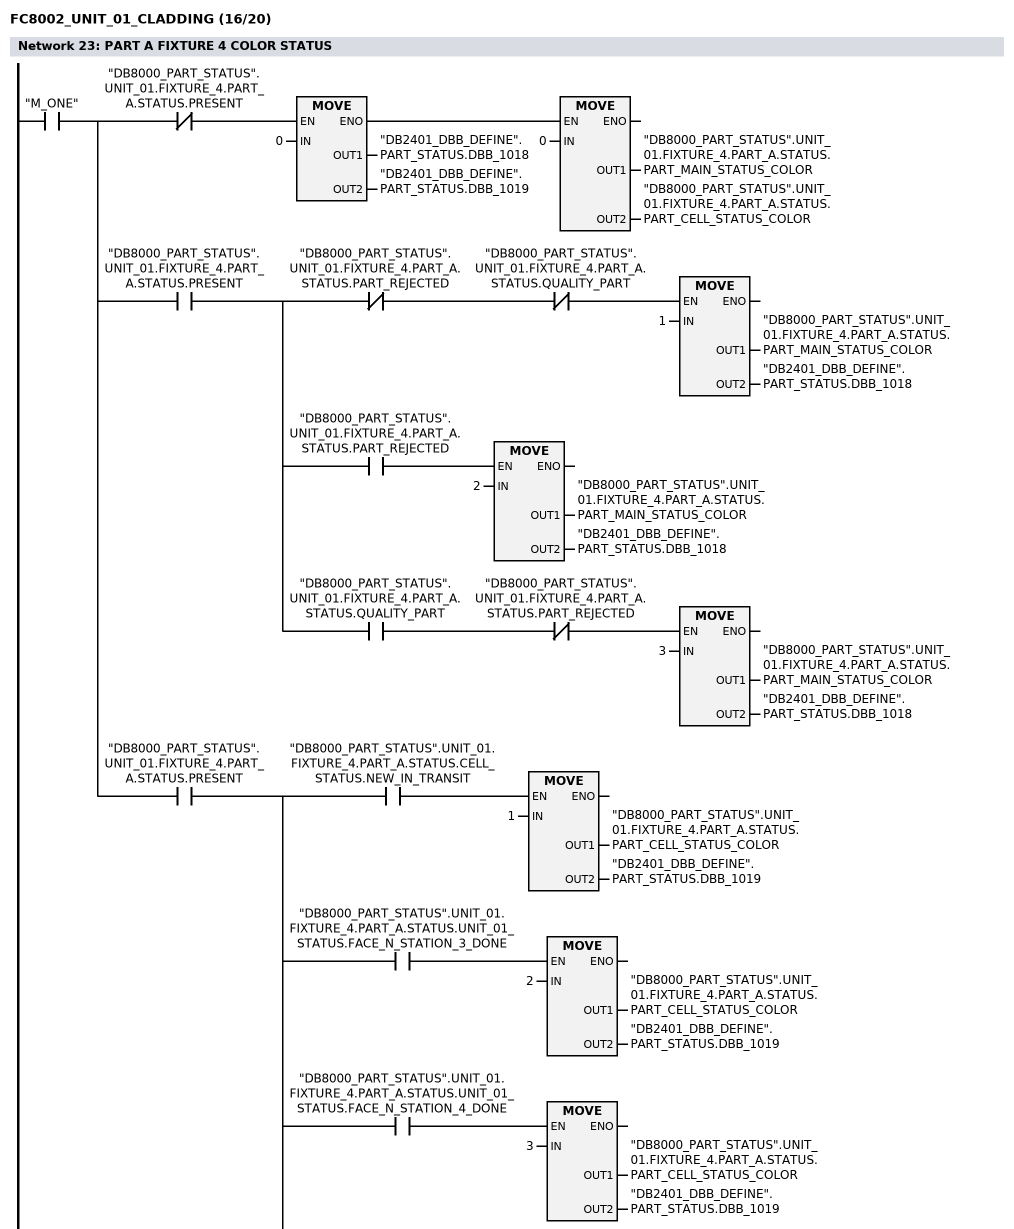
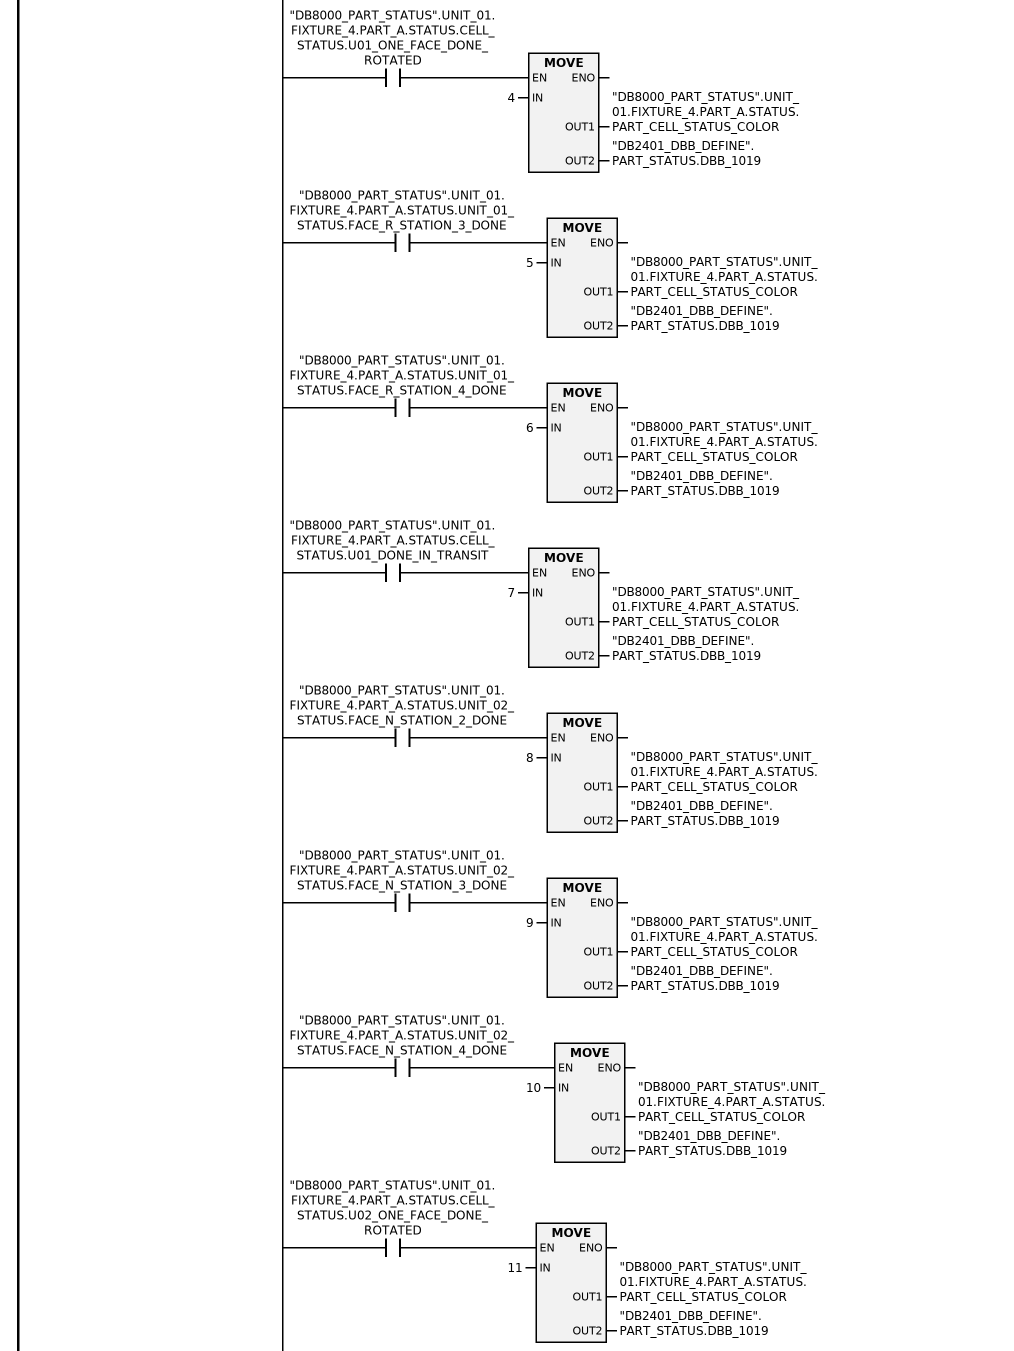
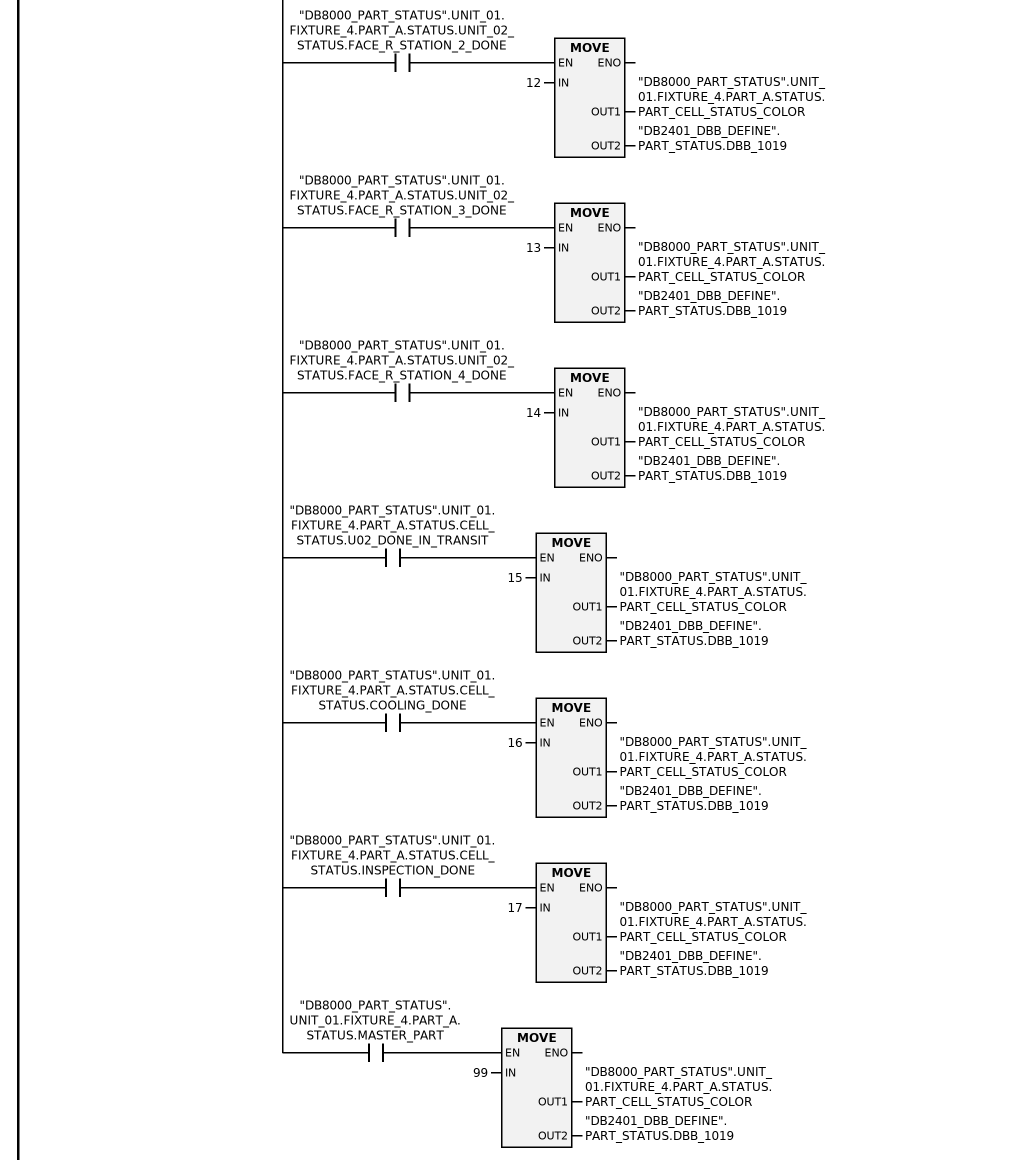
   RUNG wire#powerrail
      Contact( "M_ONE" )
      wire#w1
      I_Contact( "DB8000_PART_STATUS".UNIT_01.FIXTURE_4.PART_A.STATUS.PRESENT )
      { S7_GenerateENO := "TRUE" } Move(in := 0, out1 => "DB2401_DBB_DEFINE".PART_STATUS.DBB_1018, out2 => "DB2401_DBB_DEFINE".PART_STATUS.DBB_1019)
      { S7_GenerateENO := "TRUE" } Move(in := 0, out1 => "DB8000_PART_STATUS".UNIT_01.FIXTURE_4.PART_A.STATUS.PART_MAIN_STATUS_COLOR, out2 => "DB8000_PART_STATUS".UNIT_01.FIXTURE_4.PART_A.STATUS.PART_CELL_STATUS_COLOR)
   END_RUNG
   RUNG wire#w1
      Contact( "DB8000_PART_STATUS".UNIT_01.FIXTURE_4.PART_A.STATUS.PRESENT )
      wire#w2
      I_Contact( "DB8000_PART_STATUS".UNIT_01.FIXTURE_4.PART_A.STATUS.PART_REJECTED )
      I_Contact( "DB8000_PART_STATUS".UNIT_01.FIXTURE_4.PART_A.STATUS.QUALITY_PART )
      { S7_GenerateENO := "TRUE" } Move(in := 1, out1 => "DB8000_PART_STATUS".UNIT_01.FIXTURE_4.PART_A.STATUS.PART_MAIN_STATUS_COLOR, out2 => "DB2401_DBB_DEFINE".PART_STATUS.DBB_1018)
   END_RUNG
   RUNG wire#w2
      Contact( "DB8000_PART_STATUS".UNIT_01.FIXTURE_4.PART_A.STATUS.PART_REJECTED )
      { S7_GenerateENO := "TRUE" } Move(in := 2, out1 => "DB8000_PART_STATUS".UNIT_01.FIXTURE_4.PART_A.STATUS.PART_MAIN_STATUS_COLOR, out2 => "DB2401_DBB_DEFINE".PART_STATUS.DBB_1018)
   END_RUNG
   RUNG wire#w2
      Contact( "DB8000_PART_STATUS".UNIT_01.FIXTURE_4.PART_A.STATUS.QUALITY_PART )
      I_Contact( "DB8000_PART_STATUS".UNIT_01.FIXTURE_4.PART_A.STATUS.PART_REJECTED )
      { S7_GenerateENO := "TRUE" } Move(in := 3, out1 => "DB8000_PART_STATUS".UNIT_01.FIXTURE_4.PART_A.STATUS.PART_MAIN_STATUS_COLOR, out2 => "DB2401_DBB_DEFINE".PART_STATUS.DBB_1018)
   END_RUNG
   RUNG wire#w1
      Contact( "DB8000_PART_STATUS".UNIT_01.FIXTURE_4.PART_A.STATUS.PRESENT )
      wire#w3
      Contact( "DB8000_PART_STATUS".UNIT_01.FIXTURE_4.PART_A.STATUS.CELL_STATUS.NEW_IN_TRANSIT )
      { S7_GenerateENO := "TRUE" } Move(in := 1, out1 => "DB8000_PART_STATUS".UNIT_01.FIXTURE_4.PART_A.STATUS.PART_CELL_STATUS_COLOR, out2 => "DB2401_DBB_DEFINE".PART_STATUS.DBB_1019)
   END_RUNG
   RUNG wire#w3
      Contact( "DB8000_PART_STATUS".UNIT_01.FIXTURE_4.PART_A.STATUS.UNIT_01_STATUS.FACE_N_STATION_3_DONE )
      { S7_GenerateENO := "TRUE" } Move(in := 2, out1 => "DB8000_PART_STATUS".UNIT_01.FIXTURE_4.PART_A.STATUS.PART_CELL_STATUS_COLOR, out2 => "DB2401_DBB_DEFINE".PART_STATUS.DBB_1019)
   END_RUNG
   RUNG wire#w3
      Contact( "DB8000_PART_STATUS".UNIT_01.FIXTURE_4.PART_A.STATUS.UNIT_01_STATUS.FACE_N_STATION_4_DONE )
      { S7_GenerateENO := "TRUE" } Move(in := 3, out1 => "DB8000_PART_STATUS".UNIT_01.FIXTURE_4.PART_A.STATUS.PART_CELL_STATUS_COLOR, out2 => "DB2401_DBB_DEFINE".PART_STATUS.DBB_1019)
   END_RUNG
   RUNG wire#w3
      Contact( "DB8000_PART_STATUS".UNIT_01.FIXTURE_4.PART_A.STATUS.CELL_STATUS.U01_ONE_FACE_DONE_ROTATED )
      { S7_GenerateENO := "TRUE" } Move(in := 4, out1 => "DB8000_PART_STATUS".UNIT_01.FIXTURE_4.PART_A.STATUS.PART_CELL_STATUS_COLOR, out2 => "DB2401_DBB_DEFINE".PART_STATUS.DBB_1019)
   END_RUNG
   RUNG wire#w3
      Contact( "DB8000_PART_STATUS".UNIT_01.FIXTURE_4.PART_A.STATUS.UNIT_01_STATUS.FACE_R_STATION_3_DONE )
      { S7_GenerateENO := "TRUE" } Move(in := 5, out1 => "DB8000_PART_STATUS".UNIT_01.FIXTURE_4.PART_A.STATUS.PART_CELL_STATUS_COLOR, out2 => "DB2401_DBB_DEFINE".PART_STATUS.DBB_1019)
   END_RUNG
   RUNG wire#w3
      Contact( "DB8000_PART_STATUS".UNIT_01.FIXTURE_4.PART_A.STATUS.UNIT_01_STATUS.FACE_R_STATION_4_DONE )
      { S7_GenerateENO := "TRUE" } Move(in := 6, out1 => "DB8000_PART_STATUS".UNIT_01.FIXTURE_4.PART_A.STATUS.PART_CELL_STATUS_COLOR, out2 => "DB2401_DBB_DEFINE".PART_STATUS.DBB_1019)
   END_RUNG
   RUNG wire#w3
      Contact( "DB8000_PART_STATUS".UNIT_01.FIXTURE_4.PART_A.STATUS.CELL_STATUS.U01_DONE_IN_TRANSIT )
      { S7_GenerateENO := "TRUE" } Move(in := 7, out1 => "DB8000_PART_STATUS".UNIT_01.FIXTURE_4.PART_A.STATUS.PART_CELL_STATUS_COLOR, out2 => "DB2401_DBB_DEFINE".PART_STATUS.DBB_1019)
   END_RUNG
   RUNG wire#w3
      Contact( "DB8000_PART_STATUS".UNIT_01.FIXTURE_4.PART_A.STATUS.UNIT_02_STATUS.FACE_N_STATION_2_DONE )
      { S7_GenerateENO := "TRUE" } Move(in := 8, out1 => "DB8000_PART_STATUS".UNIT_01.FIXTURE_4.PART_A.STATUS.PART_CELL_STATUS_COLOR, out2 => "DB2401_DBB_DEFINE".PART_STATUS.DBB_1019)
   END_RUNG
   RUNG wire#w3
      Contact( "DB8000_PART_STATUS".UNIT_01.FIXTURE_4.PART_A.STATUS.UNIT_02_STATUS.FACE_N_STATION_3_DONE )
      { S7_GenerateENO := "TRUE" } Move(in := 9, out1 => "DB8000_PART_STATUS".UNIT_01.FIXTURE_4.PART_A.STATUS.PART_CELL_STATUS_COLOR, out2 => "DB2401_DBB_DEFINE".PART_STATUS.DBB_1019)
   END_RUNG
   RUNG wire#w3
      Contact( "DB8000_PART_STATUS".UNIT_01.FIXTURE_4.PART_A.STATUS.UNIT_02_STATUS.FACE_N_STATION_4_DONE )
      { S7_GenerateENO := "TRUE" } Move(in := 10, out1 => "DB8000_PART_STATUS".UNIT_01.FIXTURE_4.PART_A.STATUS.PART_CELL_STATUS_COLOR, out2 => "DB2401_DBB_DEFINE".PART_STATUS.DBB_1019)
   END_RUNG
   RUNG wire#w3
      Contact( "DB8000_PART_STATUS".UNIT_01.FIXTURE_4.PART_A.STATUS.CELL_STATUS.U02_ONE_FACE_DONE_ROTATED )
      { S7_GenerateENO := "TRUE" } Move(in := 11, out1 => "DB8000_PART_STATUS".UNIT_01.FIXTURE_4.PART_A.STATUS.PART_CELL_STATUS_COLOR, out2 => "DB2401_DBB_DEFINE".PART_STATUS.DBB_1019)
   END_RUNG
   RUNG wire#w3
      Contact( "DB8000_PART_STATUS".UNIT_01.FIXTURE_4.PART_A.STATUS.UNIT_02_STATUS.FACE_R_STATION_2_DONE )
      { S7_GenerateENO := "TRUE" } Move(in := 12, out1 => "DB8000_PART_STATUS".UNIT_01.FIXTURE_4.PART_A.STATUS.PART_CELL_STATUS_COLOR, out2 => "DB2401_DBB_DEFINE".PART_STATUS.DBB_1019)
   END_RUNG
   RUNG wire#w3
      Contact( "DB8000_PART_STATUS".UNIT_01.FIXTURE_4.PART_A.STATUS.UNIT_02_STATUS.FACE_R_STATION_3_DONE )
      Move(in := 13, out1 => "DB8000_PART_STATUS".UNIT_01.FIXTURE_4.PART_A.STATUS.PART_CELL_STATUS_COLOR, out2 => "DB2401_DBB_DEFINE".PART_STATUS.DBB_1019)
   END_RUNG
   RUNG wire#w3
      Contact( "DB8000_PART_STATUS".UNIT_01.FIXTURE_4.PART_A.STATUS.UNIT_02_STATUS.FACE_R_STATION_4_DONE )
      Move(in := 14, out1 => "DB8000_PART_STATUS".UNIT_01.FIXTURE_4.PART_A.STATUS.PART_CELL_STATUS_COLOR, out2 => "DB2401_DBB_DEFINE".PART_STATUS.DBB_1019)
   END_RUNG
   RUNG wire#w3
      Contact( "DB8000_PART_STATUS".UNIT_01.FIXTURE_4.PART_A.STATUS.CELL_STATUS.U02_DONE_IN_TRANSIT )
      Move(in := 15, out1 => "DB8000_PART_STATUS".UNIT_01.FIXTURE_4.PART_A.STATUS.PART_CELL_STATUS_COLOR, out2 => "DB2401_DBB_DEFINE".PART_STATUS.DBB_1019)
   END_RUNG
   RUNG wire#w3
      Contact( "DB8000_PART_STATUS".UNIT_01.FIXTURE_4.PART_A.STATUS.CELL_STATUS.COOLING_DONE )
      Move(in := 16, out1 => "DB8000_PART_STATUS".UNIT_01.FIXTURE_4.PART_A.STATUS.PART_CELL_STATUS_COLOR, out2 => "DB2401_DBB_DEFINE".PART_STATUS.DBB_1019)
   END_RUNG
   RUNG wire#w3
      Contact( "DB8000_PART_STATUS".UNIT_01.FIXTURE_4.PART_A.STATUS.CELL_STATUS.INSPECTION_DONE )
      Move(in := 17, out1 => "DB8000_PART_STATUS".UNIT_01.FIXTURE_4.PART_A.STATUS.PART_CELL_STATUS_COLOR, out2 => "DB2401_DBB_DEFINE".PART_STATUS.DBB_1019)
   END_RUNG
   RUNG wire#w3
      Contact( "DB8000_PART_STATUS".UNIT_01.FIXTURE_4.PART_A.STATUS.MASTER_PART )
      Move(in := 99, out1 => "DB8000_PART_STATUS".UNIT_01.FIXTURE_4.PART_A.STATUS.PART_CELL_STATUS_COLOR, out2 => "DB2401_DBB_DEFINE".PART_STATUS.DBB_1019)
   END_RUNG
   // the same network as SCL:
   // ENO of a box is taken as its EN; it also drops when the box reports an error
   IF "M_ONE" AND NOT "DB8000_PART_STATUS".UNIT_01.FIXTURE_4.PART_A.STATUS.PRESENT THEN
       "DB2401_DBB_DEFINE".PART_STATUS.DBB_1018 := 0;
       "DB2401_DBB_DEFINE".PART_STATUS.DBB_1019 := 0;
       "DB8000_PART_STATUS".UNIT_01.FIXTURE_4.PART_A.STATUS.PART_MAIN_STATUS_COLOR := 0;
       "DB8000_PART_STATUS".UNIT_01.FIXTURE_4.PART_A.STATUS.PART_CELL_STATUS_COLOR := 0;
   END_IF;
   #_w1 := "M_ONE" AND "DB8000_PART_STATUS".UNIT_01.FIXTURE_4.PART_A.STATUS.PRESENT;
   IF #_w1 AND NOT "DB8000_PART_STATUS".UNIT_01.FIXTURE_4.PART_A.STATUS.PART_REJECTED AND NOT "DB8000_PART_STATUS".UNIT_01.FIXTURE_4.PART_A.STATUS.QUALITY_PART THEN
       "DB8000_PART_STATUS".UNIT_01.FIXTURE_4.PART_A.STATUS.PART_MAIN_STATUS_COLOR := 1;
       "DB2401_DBB_DEFINE".PART_STATUS.DBB_1018 := 1;
   END_IF;
   IF #_w1 AND "DB8000_PART_STATUS".UNIT_01.FIXTURE_4.PART_A.STATUS.PART_REJECTED THEN
       "DB8000_PART_STATUS".UNIT_01.FIXTURE_4.PART_A.STATUS.PART_MAIN_STATUS_COLOR := 2;
       "DB2401_DBB_DEFINE".PART_STATUS.DBB_1018 := 2;
   END_IF;
   IF #_w1 AND "DB8000_PART_STATUS".UNIT_01.FIXTURE_4.PART_A.STATUS.QUALITY_PART AND NOT "DB8000_PART_STATUS".UNIT_01.FIXTURE_4.PART_A.STATUS.PART_REJECTED THEN
       "DB8000_PART_STATUS".UNIT_01.FIXTURE_4.PART_A.STATUS.PART_MAIN_STATUS_COLOR := 3;
       "DB2401_DBB_DEFINE".PART_STATUS.DBB_1018 := 3;
   END_IF;
   #_w2 := "M_ONE" AND "DB8000_PART_STATUS".UNIT_01.FIXTURE_4.PART_A.STATUS.PRESENT;
   IF #_w2 AND "DB8000_PART_STATUS".UNIT_01.FIXTURE_4.PART_A.STATUS.CELL_STATUS.NEW_IN_TRANSIT THEN
       "DB8000_PART_STATUS".UNIT_01.FIXTURE_4.PART_A.STATUS.PART_CELL_STATUS_COLOR := 1;
       "DB2401_DBB_DEFINE".PART_STATUS.DBB_1019 := 1;
   END_IF;
   IF #_w2 AND "DB8000_PART_STATUS".UNIT_01.FIXTURE_4.PART_A.STATUS.UNIT_01_STATUS.FACE_N_STATION_3_DONE THEN
       "DB8000_PART_STATUS".UNIT_01.FIXTURE_4.PART_A.STATUS.PART_CELL_STATUS_COLOR := 2;
       "DB2401_DBB_DEFINE".PART_STATUS.DBB_1019 := 2;
   END_IF;
   IF #_w2 AND "DB8000_PART_STATUS".UNIT_01.FIXTURE_4.PART_A.STATUS.UNIT_01_STATUS.FACE_N_STATION_4_DONE THEN
       "DB8000_PART_STATUS".UNIT_01.FIXTURE_4.PART_A.STATUS.PART_CELL_STATUS_COLOR := 3;
       "DB2401_DBB_DEFINE".PART_STATUS.DBB_1019 := 3;
   END_IF;
   IF #_w2 AND "DB8000_PART_STATUS".UNIT_01.FIXTURE_4.PART_A.STATUS.CELL_STATUS.U01_ONE_FACE_DONE_ROTATED THEN
       "DB8000_PART_STATUS".UNIT_01.FIXTURE_4.PART_A.STATUS.PART_CELL_STATUS_COLOR := 4;
       "DB2401_DBB_DEFINE".PART_STATUS.DBB_1019 := 4;
   END_IF;
   IF #_w2 AND "DB8000_PART_STATUS".UNIT_01.FIXTURE_4.PART_A.STATUS.UNIT_01_STATUS.FACE_R_STATION_3_DONE THEN
       "DB8000_PART_STATUS".UNIT_01.FIXTURE_4.PART_A.STATUS.PART_CELL_STATUS_COLOR := 5;
       "DB2401_DBB_DEFINE".PART_STATUS.DBB_1019 := 5;
   END_IF;
   IF #_w2 AND "DB8000_PART_STATUS".UNIT_01.FIXTURE_4.PART_A.STATUS.UNIT_01_STATUS.FACE_R_STATION_4_DONE THEN
       "DB8000_PART_STATUS".UNIT_01.FIXTURE_4.PART_A.STATUS.PART_CELL_STATUS_COLOR := 6;
       "DB2401_DBB_DEFINE".PART_STATUS.DBB_1019 := 6;
   END_IF;
   IF #_w2 AND "DB8000_PART_STATUS".UNIT_01.FIXTURE_4.PART_A.STATUS.CELL_STATUS.U01_DONE_IN_TRANSIT THEN
       "DB8000_PART_STATUS".UNIT_01.FIXTURE_4.PART_A.STATUS.PART_CELL_STATUS_COLOR := 7;
       "DB2401_DBB_DEFINE".PART_STATUS.DBB_1019 := 7;
   END_IF;
   IF #_w2 AND "DB8000_PART_STATUS".UNIT_01.FIXTURE_4.PART_A.STATUS.UNIT_02_STATUS.FACE_N_STATION_2_DONE THEN
       "DB8000_PART_STATUS".UNIT_01.FIXTURE_4.PART_A.STATUS.PART_CELL_STATUS_COLOR := 8;
       "DB2401_DBB_DEFINE".PART_STATUS.DBB_1019 := 8;
   END_IF;
   IF #_w2 AND "DB8000_PART_STATUS".UNIT_01.FIXTURE_4.PART_A.STATUS.UNIT_02_STATUS.FACE_N_STATION_3_DONE THEN
       "DB8000_PART_STATUS".UNIT_01.FIXTURE_4.PART_A.STATUS.PART_CELL_STATUS_COLOR := 9;
       "DB2401_DBB_DEFINE".PART_STATUS.DBB_1019 := 9;
   END_IF;
   IF #_w2 AND "DB8000_PART_STATUS".UNIT_01.FIXTURE_4.PART_A.STATUS.UNIT_02_STATUS.FACE_N_STATION_4_DONE THEN
       "DB8000_PART_STATUS".UNIT_01.FIXTURE_4.PART_A.STATUS.PART_CELL_STATUS_COLOR := 10;
       "DB2401_DBB_DEFINE".PART_STATUS.DBB_1019 := 10;
   END_IF;
   IF #_w2 AND "DB8000_PART_STATUS".UNIT_01.FIXTURE_4.PART_A.STATUS.CELL_STATUS.U02_ONE_FACE_DONE_ROTATED THEN
       "DB8000_PART_STATUS".UNIT_01.FIXTURE_4.PART_A.STATUS.PART_CELL_STATUS_COLOR := 11;
       "DB2401_DBB_DEFINE".PART_STATUS.DBB_1019 := 11;
   END_IF;
   IF #_w2 AND "DB8000_PART_STATUS".UNIT_01.FIXTURE_4.PART_A.STATUS.UNIT_02_STATUS.FACE_R_STATION_2_DONE THEN
       "DB8000_PART_STATUS".UNIT_01.FIXTURE_4.PART_A.STATUS.PART_CELL_STATUS_COLOR := 12;
       "DB2401_DBB_DEFINE".PART_STATUS.DBB_1019 := 12;
   END_IF;
   IF #_w2 AND "DB8000_PART_STATUS".UNIT_01.FIXTURE_4.PART_A.STATUS.UNIT_02_STATUS.FACE_R_STATION_3_DONE THEN
       "DB8000_PART_STATUS".UNIT_01.FIXTURE_4.PART_A.STATUS.PART_CELL_STATUS_COLOR := 13;
       "DB2401_DBB_DEFINE".PART_STATUS.DBB_1019 := 13;
   END_IF;
   IF #_w2 AND "DB8000_PART_STATUS".UNIT_01.FIXTURE_4.PART_A.STATUS.UNIT_02_STATUS.FACE_R_STATION_4_DONE THEN
       "DB8000_PART_STATUS".UNIT_01.FIXTURE_4.PART_A.STATUS.PART_CELL_STATUS_COLOR := 14;
       "DB2401_DBB_DEFINE".PART_STATUS.DBB_1019 := 14;
   END_IF;
   IF #_w2 AND "DB8000_PART_STATUS".UNIT_01.FIXTURE_4.PART_A.STATUS.CELL_STATUS.U02_DONE_IN_TRANSIT THEN
       "DB8000_PART_STATUS".UNIT_01.FIXTURE_4.PART_A.STATUS.PART_CELL_STATUS_COLOR := 15;
       "DB2401_DBB_DEFINE".PART_STATUS.DBB_1019 := 15;
   END_IF;
   IF #_w2 AND "DB8000_PART_STATUS".UNIT_01.FIXTURE_4.PART_A.STATUS.CELL_STATUS.COOLING_DONE THEN
       "DB8000_PART_STATUS".UNIT_01.FIXTURE_4.PART_A.STATUS.PART_CELL_STATUS_COLOR := 16;
       "DB2401_DBB_DEFINE".PART_STATUS.DBB_1019 := 16;
   END_IF;
   IF #_w2 AND "DB8000_PART_STATUS".UNIT_01.FIXTURE_4.PART_A.STATUS.CELL_STATUS.INSPECTION_DONE THEN
       "DB8000_PART_STATUS".UNIT_01.FIXTURE_4.PART_A.STATUS.PART_CELL_STATUS_COLOR := 17;
       "DB2401_DBB_DEFINE".PART_STATUS.DBB_1019 := 17;
   END_IF;
   IF #_w2 AND "DB8000_PART_STATUS".UNIT_01.FIXTURE_4.PART_A.STATUS.MASTER_PART THEN
       "DB8000_PART_STATUS".UNIT_01.FIXTURE_4.PART_A.STATUS.PART_CELL_STATUS_COLOR := 99;
       "DB2401_DBB_DEFINE".PART_STATUS.DBB_1019 := 99;
   END_IF;
END_REGION

REGION Network 24: PART A STATION 1 COLOR STATUS
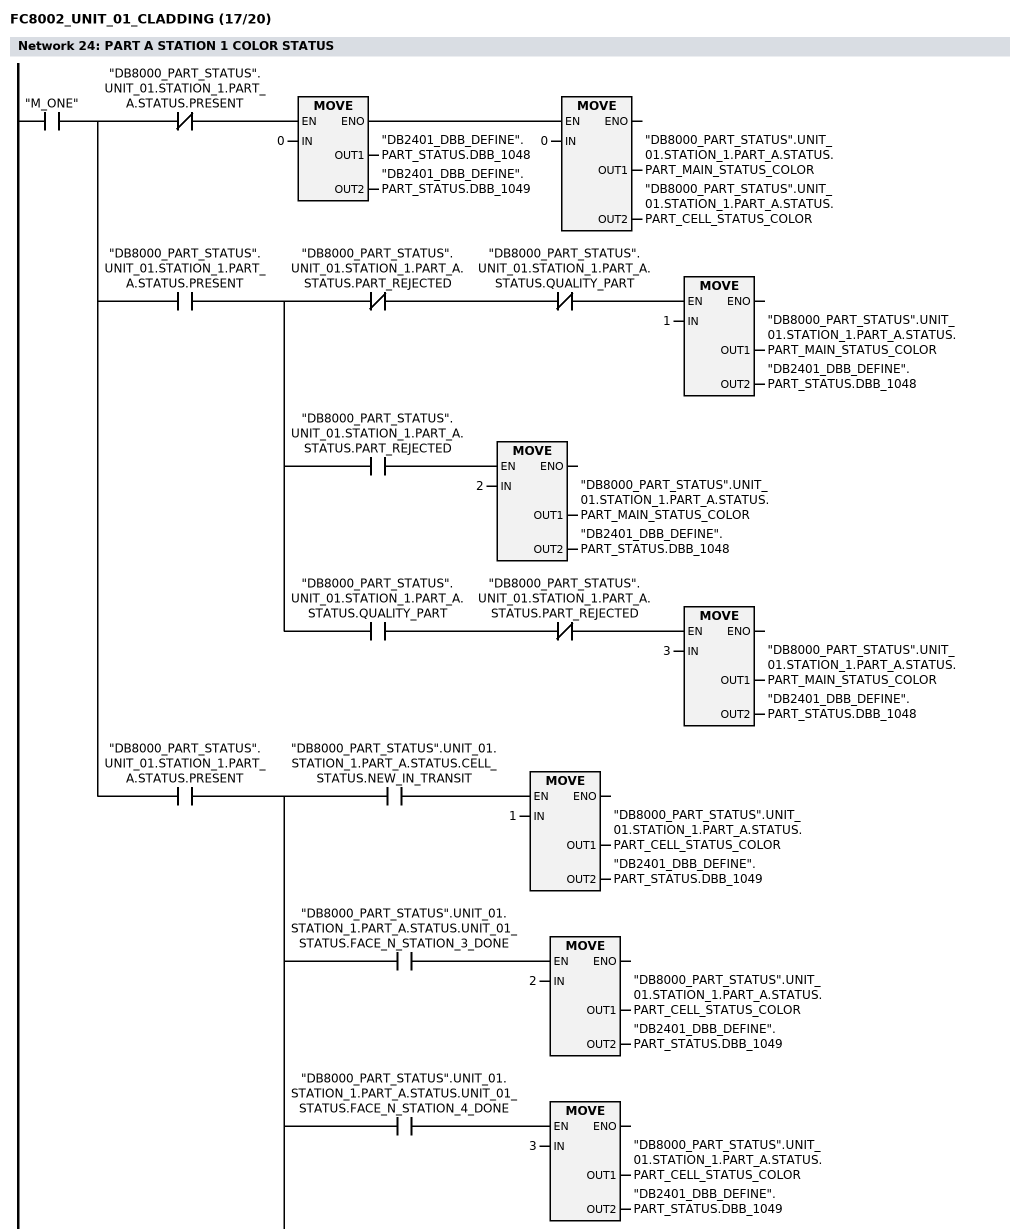
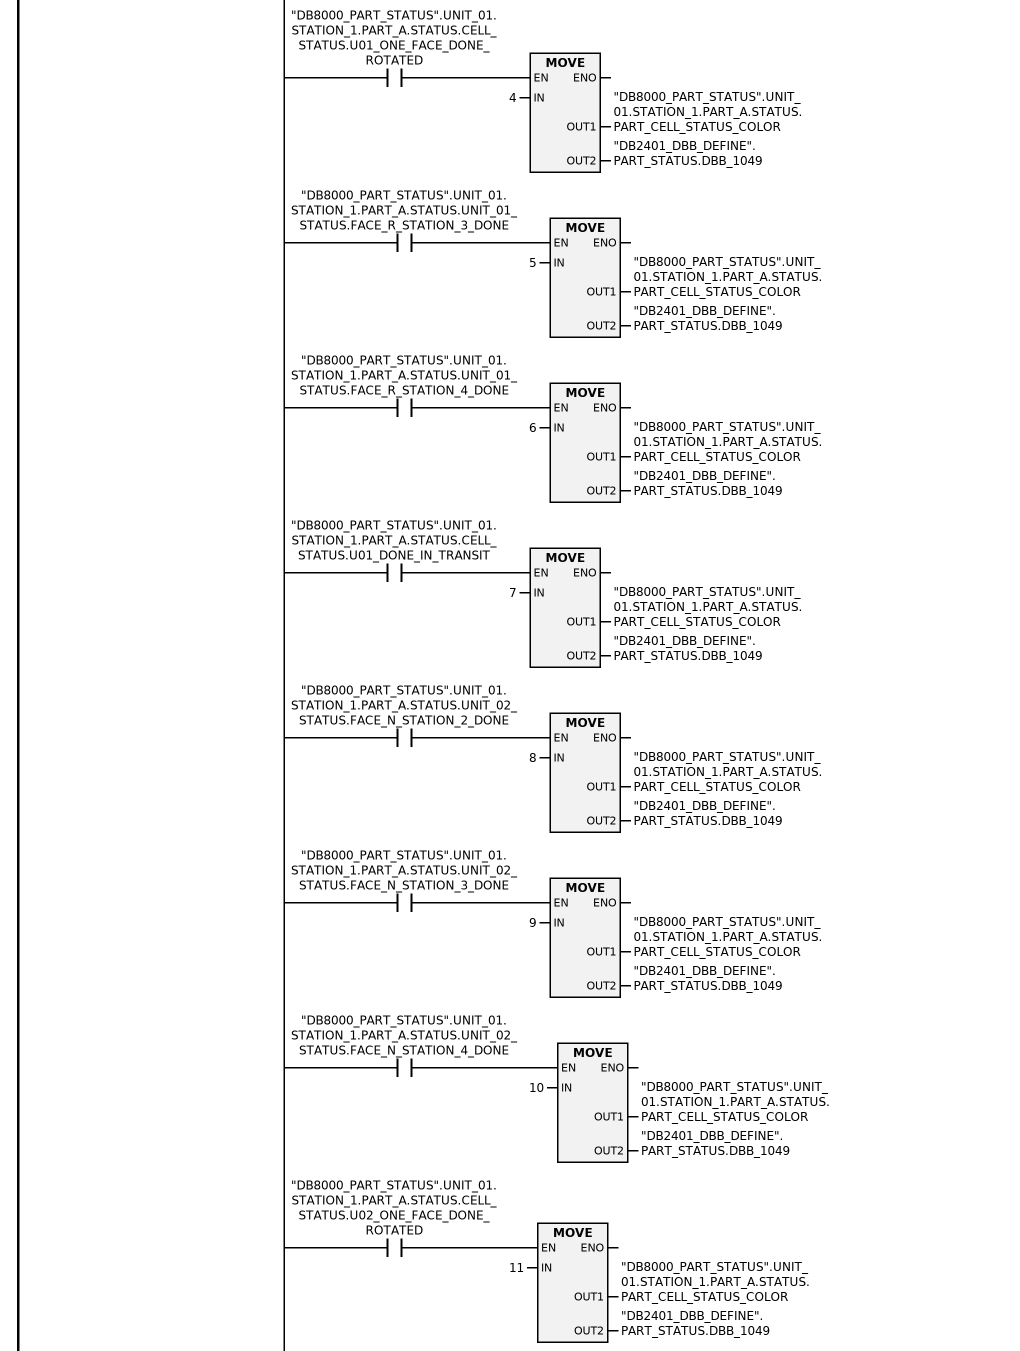
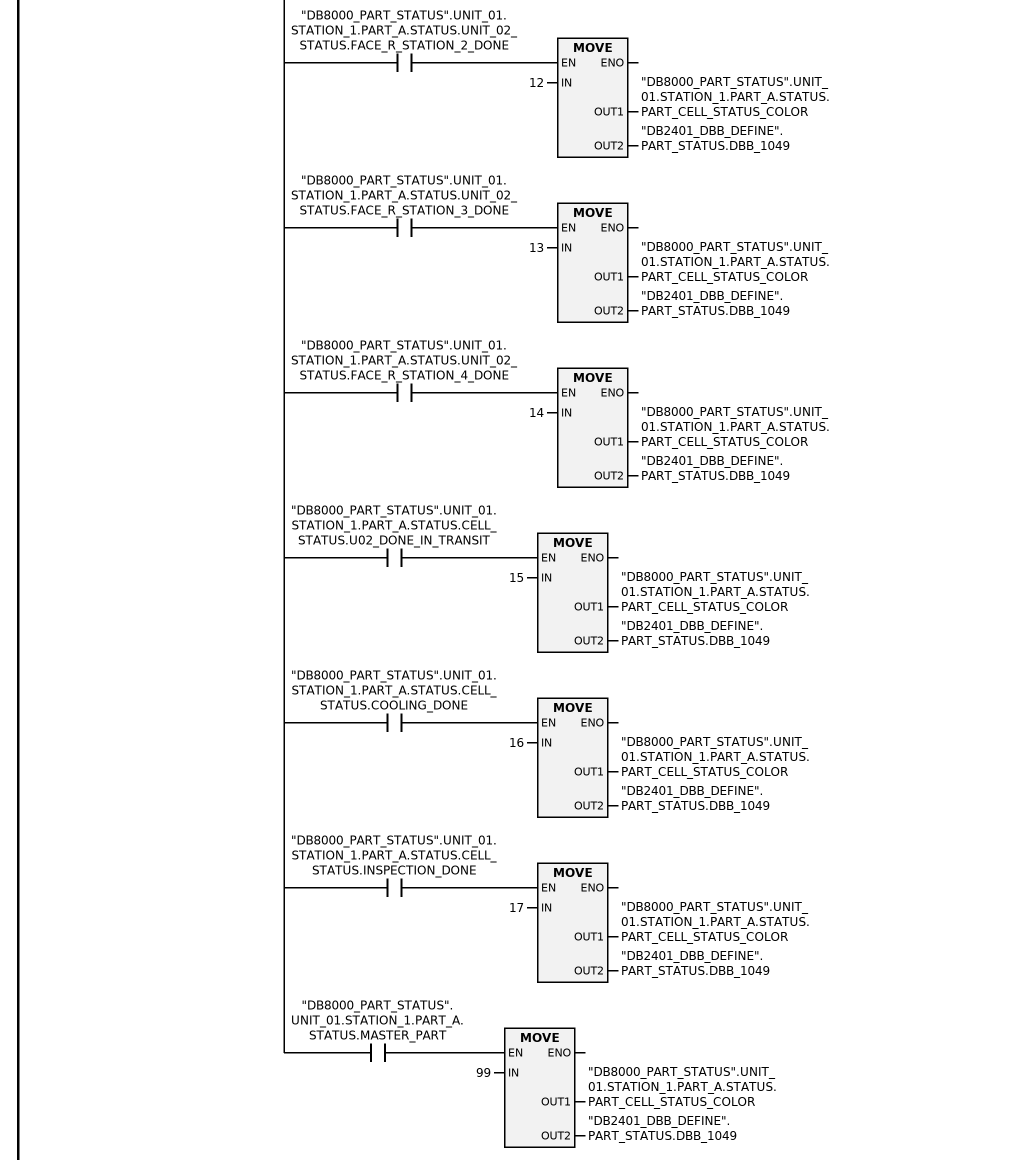
   RUNG wire#powerrail
      Contact( "M_ONE" )
      wire#w1
      I_Contact( "DB8000_PART_STATUS".UNIT_01.STATION_1.PART_A.STATUS.PRESENT )
      { S7_GenerateENO := "TRUE" } Move(in := 0, out1 => "DB2401_DBB_DEFINE".PART_STATUS.DBB_1048, out2 => "DB2401_DBB_DEFINE".PART_STATUS.DBB_1049)
      { S7_GenerateENO := "TRUE" } Move(in := 0, out1 => "DB8000_PART_STATUS".UNIT_01.STATION_1.PART_A.STATUS.PART_MAIN_STATUS_COLOR, out2 => "DB8000_PART_STATUS".UNIT_01.STATION_1.PART_A.STATUS.PART_CELL_STATUS_COLOR)
   END_RUNG
   RUNG wire#w1
      Contact( "DB8000_PART_STATUS".UNIT_01.STATION_1.PART_A.STATUS.PRESENT )
      wire#w2
      I_Contact( "DB8000_PART_STATUS".UNIT_01.STATION_1.PART_A.STATUS.PART_REJECTED )
      I_Contact( "DB8000_PART_STATUS".UNIT_01.STATION_1.PART_A.STATUS.QUALITY_PART )
      { S7_GenerateENO := "TRUE" } Move(in := 1, out1 => "DB8000_PART_STATUS".UNIT_01.STATION_1.PART_A.STATUS.PART_MAIN_STATUS_COLOR, out2 => "DB2401_DBB_DEFINE".PART_STATUS.DBB_1048)
   END_RUNG
   RUNG wire#w2
      Contact( "DB8000_PART_STATUS".UNIT_01.STATION_1.PART_A.STATUS.PART_REJECTED )
      { S7_GenerateENO := "TRUE" } Move(in := 2, out1 => "DB8000_PART_STATUS".UNIT_01.STATION_1.PART_A.STATUS.PART_MAIN_STATUS_COLOR, out2 => "DB2401_DBB_DEFINE".PART_STATUS.DBB_1048)
   END_RUNG
   RUNG wire#w2
      Contact( "DB8000_PART_STATUS".UNIT_01.STATION_1.PART_A.STATUS.QUALITY_PART )
      I_Contact( "DB8000_PART_STATUS".UNIT_01.STATION_1.PART_A.STATUS.PART_REJECTED )
      { S7_GenerateENO := "TRUE" } Move(in := 3, out1 => "DB8000_PART_STATUS".UNIT_01.STATION_1.PART_A.STATUS.PART_MAIN_STATUS_COLOR, out2 => "DB2401_DBB_DEFINE".PART_STATUS.DBB_1048)
   END_RUNG
   RUNG wire#w1
      Contact( "DB8000_PART_STATUS".UNIT_01.STATION_1.PART_A.STATUS.PRESENT )
      wire#w3
      Contact( "DB8000_PART_STATUS".UNIT_01.STATION_1.PART_A.STATUS.CELL_STATUS.NEW_IN_TRANSIT )
      { S7_GenerateENO := "TRUE" } Move(in := 1, out1 => "DB8000_PART_STATUS".UNIT_01.STATION_1.PART_A.STATUS.PART_CELL_STATUS_COLOR, out2 => "DB2401_DBB_DEFINE".PART_STATUS.DBB_1049)
   END_RUNG
   RUNG wire#w3
      Contact( "DB8000_PART_STATUS".UNIT_01.STATION_1.PART_A.STATUS.UNIT_01_STATUS.FACE_N_STATION_3_DONE )
      { S7_GenerateENO := "TRUE" } Move(in := 2, out1 => "DB8000_PART_STATUS".UNIT_01.STATION_1.PART_A.STATUS.PART_CELL_STATUS_COLOR, out2 => "DB2401_DBB_DEFINE".PART_STATUS.DBB_1049)
   END_RUNG
   RUNG wire#w3
      Contact( "DB8000_PART_STATUS".UNIT_01.STATION_1.PART_A.STATUS.UNIT_01_STATUS.FACE_N_STATION_4_DONE )
      { S7_GenerateENO := "TRUE" } Move(in := 3, out1 => "DB8000_PART_STATUS".UNIT_01.STATION_1.PART_A.STATUS.PART_CELL_STATUS_COLOR, out2 => "DB2401_DBB_DEFINE".PART_STATUS.DBB_1049)
   END_RUNG
   RUNG wire#w3
      Contact( "DB8000_PART_STATUS".UNIT_01.STATION_1.PART_A.STATUS.CELL_STATUS.U01_ONE_FACE_DONE_ROTATED )
      { S7_GenerateENO := "TRUE" } Move(in := 4, out1 => "DB8000_PART_STATUS".UNIT_01.STATION_1.PART_A.STATUS.PART_CELL_STATUS_COLOR, out2 => "DB2401_DBB_DEFINE".PART_STATUS.DBB_1049)
   END_RUNG
   RUNG wire#w3
      Contact( "DB8000_PART_STATUS".UNIT_01.STATION_1.PART_A.STATUS.UNIT_01_STATUS.FACE_R_STATION_3_DONE )
      { S7_GenerateENO := "TRUE" } Move(in := 5, out1 => "DB8000_PART_STATUS".UNIT_01.STATION_1.PART_A.STATUS.PART_CELL_STATUS_COLOR, out2 => "DB2401_DBB_DEFINE".PART_STATUS.DBB_1049)
   END_RUNG
   RUNG wire#w3
      Contact( "DB8000_PART_STATUS".UNIT_01.STATION_1.PART_A.STATUS.UNIT_01_STATUS.FACE_R_STATION_4_DONE )
      { S7_GenerateENO := "TRUE" } Move(in := 6, out1 => "DB8000_PART_STATUS".UNIT_01.STATION_1.PART_A.STATUS.PART_CELL_STATUS_COLOR, out2 => "DB2401_DBB_DEFINE".PART_STATUS.DBB_1049)
   END_RUNG
   RUNG wire#w3
      Contact( "DB8000_PART_STATUS".UNIT_01.STATION_1.PART_A.STATUS.CELL_STATUS.U01_DONE_IN_TRANSIT )
      { S7_GenerateENO := "TRUE" } Move(in := 7, out1 => "DB8000_PART_STATUS".UNIT_01.STATION_1.PART_A.STATUS.PART_CELL_STATUS_COLOR, out2 => "DB2401_DBB_DEFINE".PART_STATUS.DBB_1049)
   END_RUNG
   RUNG wire#w3
      Contact( "DB8000_PART_STATUS".UNIT_01.STATION_1.PART_A.STATUS.UNIT_02_STATUS.FACE_N_STATION_2_DONE )
      { S7_GenerateENO := "TRUE" } Move(in := 8, out1 => "DB8000_PART_STATUS".UNIT_01.STATION_1.PART_A.STATUS.PART_CELL_STATUS_COLOR, out2 => "DB2401_DBB_DEFINE".PART_STATUS.DBB_1049)
   END_RUNG
   RUNG wire#w3
      Contact( "DB8000_PART_STATUS".UNIT_01.STATION_1.PART_A.STATUS.UNIT_02_STATUS.FACE_N_STATION_3_DONE )
      Move(in := 9, out1 => "DB8000_PART_STATUS".UNIT_01.STATION_1.PART_A.STATUS.PART_CELL_STATUS_COLOR, out2 => "DB2401_DBB_DEFINE".PART_STATUS.DBB_1049)
   END_RUNG
   RUNG wire#w3
      Contact( "DB8000_PART_STATUS".UNIT_01.STATION_1.PART_A.STATUS.UNIT_02_STATUS.FACE_N_STATION_4_DONE )
      Move(in := 10, out1 => "DB8000_PART_STATUS".UNIT_01.STATION_1.PART_A.STATUS.PART_CELL_STATUS_COLOR, out2 => "DB2401_DBB_DEFINE".PART_STATUS.DBB_1049)
   END_RUNG
   RUNG wire#w3
      Contact( "DB8000_PART_STATUS".UNIT_01.STATION_1.PART_A.STATUS.CELL_STATUS.U02_ONE_FACE_DONE_ROTATED )
      Move(in := 11, out1 => "DB8000_PART_STATUS".UNIT_01.STATION_1.PART_A.STATUS.PART_CELL_STATUS_COLOR, out2 => "DB2401_DBB_DEFINE".PART_STATUS.DBB_1049)
   END_RUNG
   RUNG wire#w3
      Contact( "DB8000_PART_STATUS".UNIT_01.STATION_1.PART_A.STATUS.UNIT_02_STATUS.FACE_R_STATION_2_DONE )
      Move(in := 12, out1 => "DB8000_PART_STATUS".UNIT_01.STATION_1.PART_A.STATUS.PART_CELL_STATUS_COLOR, out2 => "DB2401_DBB_DEFINE".PART_STATUS.DBB_1049)
   END_RUNG
   RUNG wire#w3
      Contact( "DB8000_PART_STATUS".UNIT_01.STATION_1.PART_A.STATUS.UNIT_02_STATUS.FACE_R_STATION_3_DONE )
      Move(in := 13, out1 => "DB8000_PART_STATUS".UNIT_01.STATION_1.PART_A.STATUS.PART_CELL_STATUS_COLOR, out2 => "DB2401_DBB_DEFINE".PART_STATUS.DBB_1049)
   END_RUNG
   RUNG wire#w3
      Contact( "DB8000_PART_STATUS".UNIT_01.STATION_1.PART_A.STATUS.UNIT_02_STATUS.FACE_R_STATION_4_DONE )
      Move(in := 14, out1 => "DB8000_PART_STATUS".UNIT_01.STATION_1.PART_A.STATUS.PART_CELL_STATUS_COLOR, out2 => "DB2401_DBB_DEFINE".PART_STATUS.DBB_1049)
   END_RUNG
   RUNG wire#w3
      Contact( "DB8000_PART_STATUS".UNIT_01.STATION_1.PART_A.STATUS.CELL_STATUS.U02_DONE_IN_TRANSIT )
      Move(in := 15, out1 => "DB8000_PART_STATUS".UNIT_01.STATION_1.PART_A.STATUS.PART_CELL_STATUS_COLOR, out2 => "DB2401_DBB_DEFINE".PART_STATUS.DBB_1049)
   END_RUNG
   RUNG wire#w3
      Contact( "DB8000_PART_STATUS".UNIT_01.STATION_1.PART_A.STATUS.CELL_STATUS.COOLING_DONE )
      Move(in := 16, out1 => "DB8000_PART_STATUS".UNIT_01.STATION_1.PART_A.STATUS.PART_CELL_STATUS_COLOR, out2 => "DB2401_DBB_DEFINE".PART_STATUS.DBB_1049)
   END_RUNG
   RUNG wire#w3
      Contact( "DB8000_PART_STATUS".UNIT_01.STATION_1.PART_A.STATUS.CELL_STATUS.INSPECTION_DONE )
      Move(in := 17, out1 => "DB8000_PART_STATUS".UNIT_01.STATION_1.PART_A.STATUS.PART_CELL_STATUS_COLOR, out2 => "DB2401_DBB_DEFINE".PART_STATUS.DBB_1049)
   END_RUNG
   RUNG wire#w3
      Contact( "DB8000_PART_STATUS".UNIT_01.STATION_1.PART_A.STATUS.MASTER_PART )
      Move(in := 99, out1 => "DB8000_PART_STATUS".UNIT_01.STATION_1.PART_A.STATUS.PART_CELL_STATUS_COLOR, out2 => "DB2401_DBB_DEFINE".PART_STATUS.DBB_1049)
   END_RUNG
   // the same network as SCL:
   // ENO of a box is taken as its EN; it also drops when the box reports an error
   IF "M_ONE" AND NOT "DB8000_PART_STATUS".UNIT_01.STATION_1.PART_A.STATUS.PRESENT THEN
       "DB2401_DBB_DEFINE".PART_STATUS.DBB_1048 := 0;
       "DB2401_DBB_DEFINE".PART_STATUS.DBB_1049 := 0;
       "DB8000_PART_STATUS".UNIT_01.STATION_1.PART_A.STATUS.PART_MAIN_STATUS_COLOR := 0;
       "DB8000_PART_STATUS".UNIT_01.STATION_1.PART_A.STATUS.PART_CELL_STATUS_COLOR := 0;
   END_IF;
   #_w1 := "M_ONE" AND "DB8000_PART_STATUS".UNIT_01.STATION_1.PART_A.STATUS.PRESENT;
   IF #_w1 AND NOT "DB8000_PART_STATUS".UNIT_01.STATION_1.PART_A.STATUS.PART_REJECTED AND NOT "DB8000_PART_STATUS".UNIT_01.STATION_1.PART_A.STATUS.QUALITY_PART THEN
       "DB8000_PART_STATUS".UNIT_01.STATION_1.PART_A.STATUS.PART_MAIN_STATUS_COLOR := 1;
       "DB2401_DBB_DEFINE".PART_STATUS.DBB_1048 := 1;
   END_IF;
   IF #_w1 AND "DB8000_PART_STATUS".UNIT_01.STATION_1.PART_A.STATUS.PART_REJECTED THEN
       "DB8000_PART_STATUS".UNIT_01.STATION_1.PART_A.STATUS.PART_MAIN_STATUS_COLOR := 2;
       "DB2401_DBB_DEFINE".PART_STATUS.DBB_1048 := 2;
   END_IF;
   IF #_w1 AND "DB8000_PART_STATUS".UNIT_01.STATION_1.PART_A.STATUS.QUALITY_PART AND NOT "DB8000_PART_STATUS".UNIT_01.STATION_1.PART_A.STATUS.PART_REJECTED THEN
       "DB8000_PART_STATUS".UNIT_01.STATION_1.PART_A.STATUS.PART_MAIN_STATUS_COLOR := 3;
       "DB2401_DBB_DEFINE".PART_STATUS.DBB_1048 := 3;
   END_IF;
   #_w2 := "M_ONE" AND "DB8000_PART_STATUS".UNIT_01.STATION_1.PART_A.STATUS.PRESENT;
   IF #_w2 AND "DB8000_PART_STATUS".UNIT_01.STATION_1.PART_A.STATUS.CELL_STATUS.NEW_IN_TRANSIT THEN
       "DB8000_PART_STATUS".UNIT_01.STATION_1.PART_A.STATUS.PART_CELL_STATUS_COLOR := 1;
       "DB2401_DBB_DEFINE".PART_STATUS.DBB_1049 := 1;
   END_IF;
   IF #_w2 AND "DB8000_PART_STATUS".UNIT_01.STATION_1.PART_A.STATUS.UNIT_01_STATUS.FACE_N_STATION_3_DONE THEN
       "DB8000_PART_STATUS".UNIT_01.STATION_1.PART_A.STATUS.PART_CELL_STATUS_COLOR := 2;
       "DB2401_DBB_DEFINE".PART_STATUS.DBB_1049 := 2;
   END_IF;
   IF #_w2 AND "DB8000_PART_STATUS".UNIT_01.STATION_1.PART_A.STATUS.UNIT_01_STATUS.FACE_N_STATION_4_DONE THEN
       "DB8000_PART_STATUS".UNIT_01.STATION_1.PART_A.STATUS.PART_CELL_STATUS_COLOR := 3;
       "DB2401_DBB_DEFINE".PART_STATUS.DBB_1049 := 3;
   END_IF;
   IF #_w2 AND "DB8000_PART_STATUS".UNIT_01.STATION_1.PART_A.STATUS.CELL_STATUS.U01_ONE_FACE_DONE_ROTATED THEN
       "DB8000_PART_STATUS".UNIT_01.STATION_1.PART_A.STATUS.PART_CELL_STATUS_COLOR := 4;
       "DB2401_DBB_DEFINE".PART_STATUS.DBB_1049 := 4;
   END_IF;
   IF #_w2 AND "DB8000_PART_STATUS".UNIT_01.STATION_1.PART_A.STATUS.UNIT_01_STATUS.FACE_R_STATION_3_DONE THEN
       "DB8000_PART_STATUS".UNIT_01.STATION_1.PART_A.STATUS.PART_CELL_STATUS_COLOR := 5;
       "DB2401_DBB_DEFINE".PART_STATUS.DBB_1049 := 5;
   END_IF;
   IF #_w2 AND "DB8000_PART_STATUS".UNIT_01.STATION_1.PART_A.STATUS.UNIT_01_STATUS.FACE_R_STATION_4_DONE THEN
       "DB8000_PART_STATUS".UNIT_01.STATION_1.PART_A.STATUS.PART_CELL_STATUS_COLOR := 6;
       "DB2401_DBB_DEFINE".PART_STATUS.DBB_1049 := 6;
   END_IF;
   IF #_w2 AND "DB8000_PART_STATUS".UNIT_01.STATION_1.PART_A.STATUS.CELL_STATUS.U01_DONE_IN_TRANSIT THEN
       "DB8000_PART_STATUS".UNIT_01.STATION_1.PART_A.STATUS.PART_CELL_STATUS_COLOR := 7;
       "DB2401_DBB_DEFINE".PART_STATUS.DBB_1049 := 7;
   END_IF;
   IF #_w2 AND "DB8000_PART_STATUS".UNIT_01.STATION_1.PART_A.STATUS.UNIT_02_STATUS.FACE_N_STATION_2_DONE THEN
       "DB8000_PART_STATUS".UNIT_01.STATION_1.PART_A.STATUS.PART_CELL_STATUS_COLOR := 8;
       "DB2401_DBB_DEFINE".PART_STATUS.DBB_1049 := 8;
   END_IF;
   IF #_w2 AND "DB8000_PART_STATUS".UNIT_01.STATION_1.PART_A.STATUS.UNIT_02_STATUS.FACE_N_STATION_3_DONE THEN
       "DB8000_PART_STATUS".UNIT_01.STATION_1.PART_A.STATUS.PART_CELL_STATUS_COLOR := 9;
       "DB2401_DBB_DEFINE".PART_STATUS.DBB_1049 := 9;
   END_IF;
   IF #_w2 AND "DB8000_PART_STATUS".UNIT_01.STATION_1.PART_A.STATUS.UNIT_02_STATUS.FACE_N_STATION_4_DONE THEN
       "DB8000_PART_STATUS".UNIT_01.STATION_1.PART_A.STATUS.PART_CELL_STATUS_COLOR := 10;
       "DB2401_DBB_DEFINE".PART_STATUS.DBB_1049 := 10;
   END_IF;
   IF #_w2 AND "DB8000_PART_STATUS".UNIT_01.STATION_1.PART_A.STATUS.CELL_STATUS.U02_ONE_FACE_DONE_ROTATED THEN
       "DB8000_PART_STATUS".UNIT_01.STATION_1.PART_A.STATUS.PART_CELL_STATUS_COLOR := 11;
       "DB2401_DBB_DEFINE".PART_STATUS.DBB_1049 := 11;
   END_IF;
   IF #_w2 AND "DB8000_PART_STATUS".UNIT_01.STATION_1.PART_A.STATUS.UNIT_02_STATUS.FACE_R_STATION_2_DONE THEN
       "DB8000_PART_STATUS".UNIT_01.STATION_1.PART_A.STATUS.PART_CELL_STATUS_COLOR := 12;
       "DB2401_DBB_DEFINE".PART_STATUS.DBB_1049 := 12;
   END_IF;
   IF #_w2 AND "DB8000_PART_STATUS".UNIT_01.STATION_1.PART_A.STATUS.UNIT_02_STATUS.FACE_R_STATION_3_DONE THEN
       "DB8000_PART_STATUS".UNIT_01.STATION_1.PART_A.STATUS.PART_CELL_STATUS_COLOR := 13;
       "DB2401_DBB_DEFINE".PART_STATUS.DBB_1049 := 13;
   END_IF;
   IF #_w2 AND "DB8000_PART_STATUS".UNIT_01.STATION_1.PART_A.STATUS.UNIT_02_STATUS.FACE_R_STATION_4_DONE THEN
       "DB8000_PART_STATUS".UNIT_01.STATION_1.PART_A.STATUS.PART_CELL_STATUS_COLOR := 14;
       "DB2401_DBB_DEFINE".PART_STATUS.DBB_1049 := 14;
   END_IF;
   IF #_w2 AND "DB8000_PART_STATUS".UNIT_01.STATION_1.PART_A.STATUS.CELL_STATUS.U02_DONE_IN_TRANSIT THEN
       "DB8000_PART_STATUS".UNIT_01.STATION_1.PART_A.STATUS.PART_CELL_STATUS_COLOR := 15;
       "DB2401_DBB_DEFINE".PART_STATUS.DBB_1049 := 15;
   END_IF;
   IF #_w2 AND "DB8000_PART_STATUS".UNIT_01.STATION_1.PART_A.STATUS.CELL_STATUS.COOLING_DONE THEN
       "DB8000_PART_STATUS".UNIT_01.STATION_1.PART_A.STATUS.PART_CELL_STATUS_COLOR := 16;
       "DB2401_DBB_DEFINE".PART_STATUS.DBB_1049 := 16;
   END_IF;
   IF #_w2 AND "DB8000_PART_STATUS".UNIT_01.STATION_1.PART_A.STATUS.CELL_STATUS.INSPECTION_DONE THEN
       "DB8000_PART_STATUS".UNIT_01.STATION_1.PART_A.STATUS.PART_CELL_STATUS_COLOR := 17;
       "DB2401_DBB_DEFINE".PART_STATUS.DBB_1049 := 17;
   END_IF;
   IF #_w2 AND "DB8000_PART_STATUS".UNIT_01.STATION_1.PART_A.STATUS.MASTER_PART THEN
       "DB8000_PART_STATUS".UNIT_01.STATION_1.PART_A.STATUS.PART_CELL_STATUS_COLOR := 99;
       "DB2401_DBB_DEFINE".PART_STATUS.DBB_1049 := 99;
   END_IF;
END_REGION

